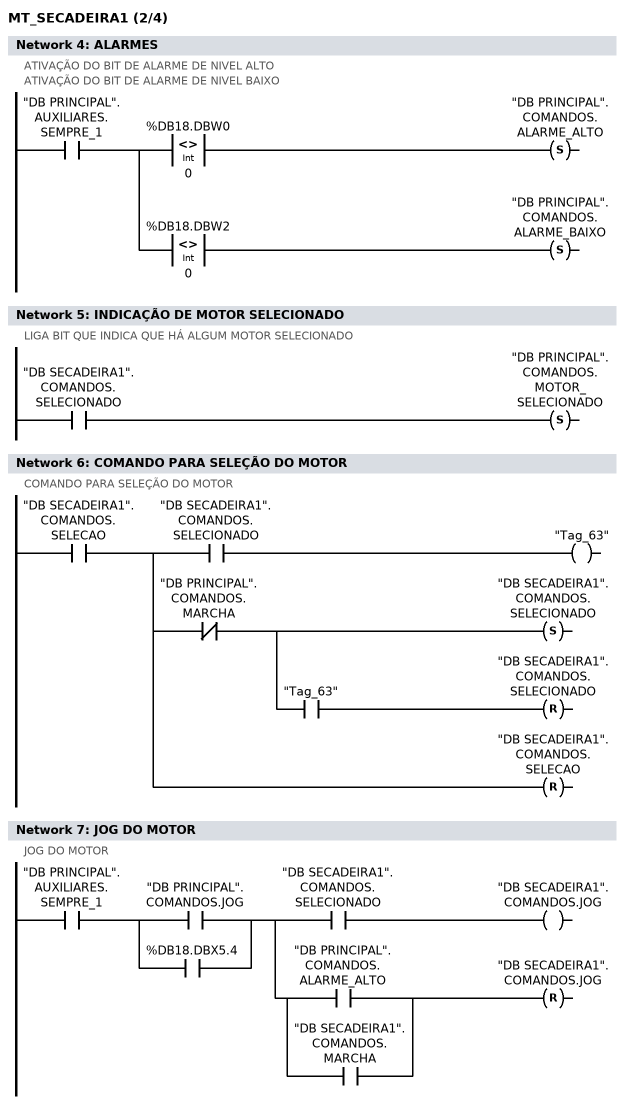
   RUNG wire#powerrail
      Contact( "DB PRINCIPAL".AUXILIARES.SEMPRE_1 )
      wire#w1
      { S7_Templates := "SrcType := Int" } NE_Contact(in1 := %DB18.DBW0, in2 := 0)
      S_Coil( "DB PRINCIPAL".COMANDOS.ALARME_ALTO )
   END_RUNG
   RUNG wire#w1
      { S7_Templates := "SrcType := Int" } NE_Contact(in1 := %DB18.DBW2, in2 := 0)
      S_Coil( "DB PRINCIPAL".COMANDOS.ALARME_BAIXO )
   END_RUNG
   // the same network as SCL:
   IF "DB PRINCIPAL".AUXILIARES.SEMPRE_1 AND (%DB18.DBW0 <> 0) THEN
       "DB PRINCIPAL".COMANDOS.ALARME_ALTO := TRUE;
   END_IF;
   IF "DB PRINCIPAL".AUXILIARES.SEMPRE_1 AND (%DB18.DBW2 <> 0) THEN
       "DB PRINCIPAL".COMANDOS.ALARME_BAIXO := TRUE;
   END_IF;
END_REGION

REGION Network 5: INDICAÇÃO DE MOTOR SELECIONADO
   // LIGA BIT QUE INDICA QUE HÁ ALGUM MOTOR SELECIONADO
   RUNG wire#powerrail
      Contact( "DB SECADEIRA1".COMANDOS.SELECIONADO )
      S_Coil( "DB PRINCIPAL".COMANDOS.MOTOR_SELECIONADO )
   END_RUNG
   // the same network as SCL:
   IF "DB SECADEIRA1".COMANDOS.SELECIONADO THEN "DB PRINCIPAL".COMANDOS.MOTOR_SELECIONADO := TRUE; END_IF;
END_REGION

REGION Network 6: COMANDO PARA SELEÇÃO DO MOTOR
   // COMANDO PARA SELEÇÃO DO MOTOR
   RUNG wire#powerrail
      Contact( "DB SECADEIRA1".COMANDOS.SELECAO )
      wire#w1
      Contact( "DB SECADEIRA1".COMANDOS.SELECIONADO )
      Coil( "Tag_63" )
   END_RUNG
   RUNG wire#w1
      I_Contact( "DB PRINCIPAL".COMANDOS.MARCHA )
      wire#w2
      S_Coil( "DB SECADEIRA1".COMANDOS.SELECIONADO )
   END_RUNG
   RUNG wire#w2
      Contact( "Tag_63" )
      R_Coil( "DB SECADEIRA1".COMANDOS.SELECIONADO )
   END_RUNG
   RUNG wire#w1
      R_Coil( "DB SECADEIRA1".COMANDOS.SELECAO )
   END_RUNG
   // the same network as SCL:
   "Tag_63" := "DB SECADEIRA1".COMANDOS.SELECAO AND "DB SECADEIRA1".COMANDOS.SELECIONADO;
   #_w1 := "DB SECADEIRA1".COMANDOS.SELECAO AND NOT "DB PRINCIPAL".COMANDOS.MARCHA;
   IF #_w1 THEN "DB SECADEIRA1".COMANDOS.SELECIONADO := TRUE; END_IF;
   IF #_w1 AND "Tag_63" THEN "DB SECADEIRA1".COMANDOS.SELECIONADO := FALSE; END_IF;
   IF "DB SECADEIRA1".COMANDOS.SELECAO THEN "DB SECADEIRA1".COMANDOS.SELECAO := FALSE; END_IF;
END_REGION

REGION Network 7: JOG DO MOTOR
   // JOG DO MOTOR
   RUNG wire#powerrail
      Contact( "DB PRINCIPAL".AUXILIARES.SEMPRE_1 )
      wire#w1
      Contact( "DB PRINCIPAL".COMANDOS.JOG )
      wire#w2
      Contact( "DB SECADEIRA1".COMANDOS.SELECIONADO )
      Coil( "DB SECADEIRA1".COMANDOS.JOG )
   END_RUNG
   RUNG wire#w1
      Contact( %DB18.DBX5.4 )
   END_RUNG wire#w2
   RUNG wire#w2
      Contact( "DB PRINCIPAL".COMANDOS.ALARME_ALTO )
      wire#w3
      R_Coil( "DB SECADEIRA1".COMANDOS.JOG )
   END_RUNG
   RUNG wire#w2
      Contact( "DB SECADEIRA1".COMANDOS.MARCHA )
   END_RUNG wire#w3
   // the same network as SCL:
   #_w1 := "DB PRINCIPAL".AUXILIARES.SEMPRE_1 AND ("DB PRINCIPAL".COMANDOS.JOG OR %DB18.DBX5.4);
   "DB SECADEIRA1".COMANDOS.JOG := #_w1 AND "DB SECADEIRA1".COMANDOS.SELECIONADO;
   IF #_w1 AND ("DB PRINCIPAL".COMANDOS.ALARME_ALTO OR "DB SECADEIRA1".COMANDOS.MARCHA) THEN
       "DB SECADEIRA1".COMANDOS.JOG := FALSE;
   END_IF;
END_REGION

REGION Network 8: COMANDO PARA LIBERAÇÃO DO MOTOR
   // COMANDO PARA LIBERAÇÃO DO MOTOR
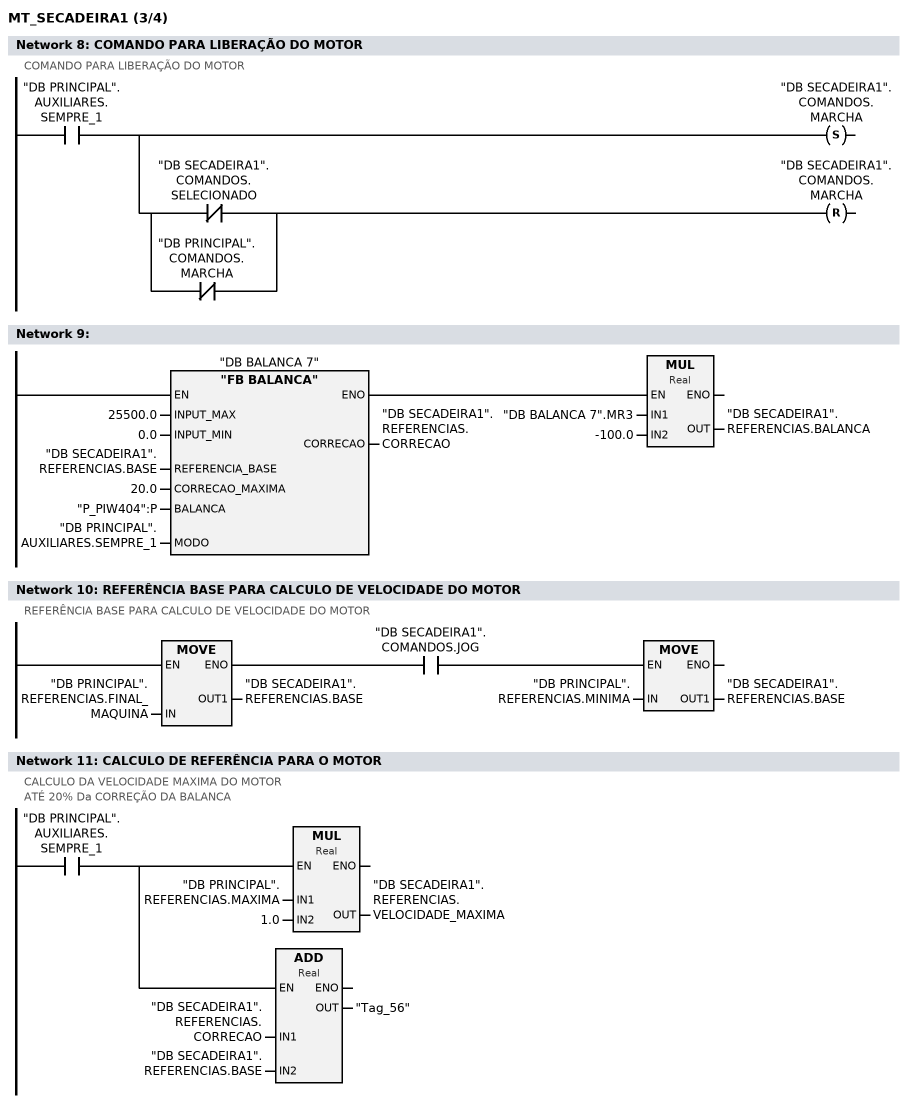
   RUNG wire#powerrail
      Contact( "DB PRINCIPAL".AUXILIARES.SEMPRE_1 )
      wire#w1
      S_Coil( "DB SECADEIRA1".COMANDOS.MARCHA )
   END_RUNG
   RUNG wire#w1
      I_Contact( "DB SECADEIRA1".COMANDOS.SELECIONADO )
      wire#w2
      R_Coil( "DB SECADEIRA1".COMANDOS.MARCHA )
   END_RUNG
   RUNG wire#w1
      I_Contact( "DB PRINCIPAL".COMANDOS.MARCHA )
   END_RUNG wire#w2
   // the same network as SCL:
   IF "DB PRINCIPAL".AUXILIARES.SEMPRE_1 THEN "DB SECADEIRA1".COMANDOS.MARCHA := TRUE; END_IF;
   IF "DB PRINCIPAL".AUXILIARES.SEMPRE_1 AND (NOT "DB SECADEIRA1".COMANDOS.SELECIONADO OR NOT "DB PRINCIPAL".COMANDOS.MARCHA) THEN
       "DB SECADEIRA1".COMANDOS.MARCHA := FALSE;
   END_IF;
END_REGION

REGION Network 9
   RUNG wire#powerrail
      "DB BALANCA 7"(INPUT_MAX := 25500.0, INPUT_MIN := 0.0, REFERENCIA_BASE := "DB SECADEIRA1".REFERENCIAS.BASE, CORRECAO_MAXIMA := 20.0, BALANCA := "P_PIW404":P, MODO := "DB PRINCIPAL".AUXILIARES.SEMPRE_1, CORRECAO => "DB SECADEIRA1".REFERENCIAS.CORRECAO)
      { S7_Templates := "SrcType := Real"; S7_GenerateENO := "TRUE" } Mul(in1 := "DB BALANCA 7".MR3, in2 := -100.0, out => "DB SECADEIRA1".REFERENCIAS.BALANCA)
   END_RUNG
   // the same network as SCL:
   "DB BALANCA 7"(INPUT_MAX := 25500.0,   // "FB BALANCA"
                  INPUT_MIN := 0.0,
                  REFERENCIA_BASE := "DB SECADEIRA1".REFERENCIAS.BASE,
                  CORRECAO_MAXIMA := 20.0,
                  BALANCA := "P_PIW404":P,
                  MODO := "DB PRINCIPAL".AUXILIARES.SEMPRE_1,
                  CORRECAO => "DB SECADEIRA1".REFERENCIAS.CORRECAO,
                  ENO => #_w1);
   IF #_w1 THEN "DB SECADEIRA1".REFERENCIAS.BALANCA := "DB BALANCA 7".MR3 * (-100.0); END_IF;
END_REGION

REGION Network 10: REFERÊNCIA BASE PARA CALCULO DE VELOCIDADE DO MOTOR
   // REFERÊNCIA BASE PARA CALCULO DE VELOCIDADE DO MOTOR
   RUNG wire#powerrail
      { S7_GenerateENO := "TRUE" } Move(in := "DB PRINCIPAL".REFERENCIAS.FINAL_MAQUINA, out1 => "DB SECADEIRA1".REFERENCIAS.BASE)
      Contact( "DB SECADEIRA1".COMANDOS.JOG )
      { S7_GenerateENO := "TRUE" } Move(in := "DB PRINCIPAL".REFERENCIAS.MINIMA, out1 => "DB SECADEIRA1".REFERENCIAS.BASE)
   END_RUNG
   // the same network as SCL:
   // ENO of a box is taken as its EN; it also drops when the box reports an error
   "DB SECADEIRA1".REFERENCIAS.BASE := "DB PRINCIPAL".REFERENCIAS.FINAL_MAQUINA;
   IF "DB SECADEIRA1".COMANDOS.JOG THEN
       "DB SECADEIRA1".REFERENCIAS.BASE := "DB PRINCIPAL".REFERENCIAS.MINIMA;
   END_IF;
END_REGION

REGION Network 11: CALCULO DE REFERÊNCIA PARA O MOTOR
   // CALCULO DA VELOCIDADE MAXIMA DO MOTOR
   // ATÉ 20% Da CORREÇÃO DA BALANCA
   RUNG wire#powerrail
      Contact( "DB PRINCIPAL".AUXILIARES.SEMPRE_1 )
      wire#w1
      { S7_Templates := "SrcType := Real"; S7_GenerateENO := "TRUE" } Mul(in1 := "DB PRINCIPAL".REFERENCIAS.MAXIMA, in2 := 1.0, out => "DB SECADEIRA1".REFERENCIAS.VELOCIDADE_MAXIMA)
   END_RUNG
   RUNG wire#w1
      { S7_Templates := "SrcType := Real"; S7_GenerateENO := "TRUE" } Add(in1 := "DB SECADEIRA1".REFERENCIAS.CORRECAO, in2 := "DB SECADEIRA1".REFERENCIAS.BASE, out => "Tag_56")
   END_RUNG
   // the same network as SCL:
   IF "DB PRINCIPAL".AUXILIARES.SEMPRE_1 THEN
       "DB SECADEIRA1".REFERENCIAS.VELOCIDADE_MAXIMA := "DB PRINCIPAL".REFERENCIAS.MAXIMA * 1.0;
       "Tag_56" := "DB SECADEIRA1".REFERENCIAS.CORRECAO + "DB SECADEIRA1".REFERENCIAS.BASE;
   END_IF;
END_REGION

REGION Network 12: ACC/DEC DA REFERÊNCIA DO MOTOR
   // ACC/DEC DA REFERÊNCIA DO MOTOR
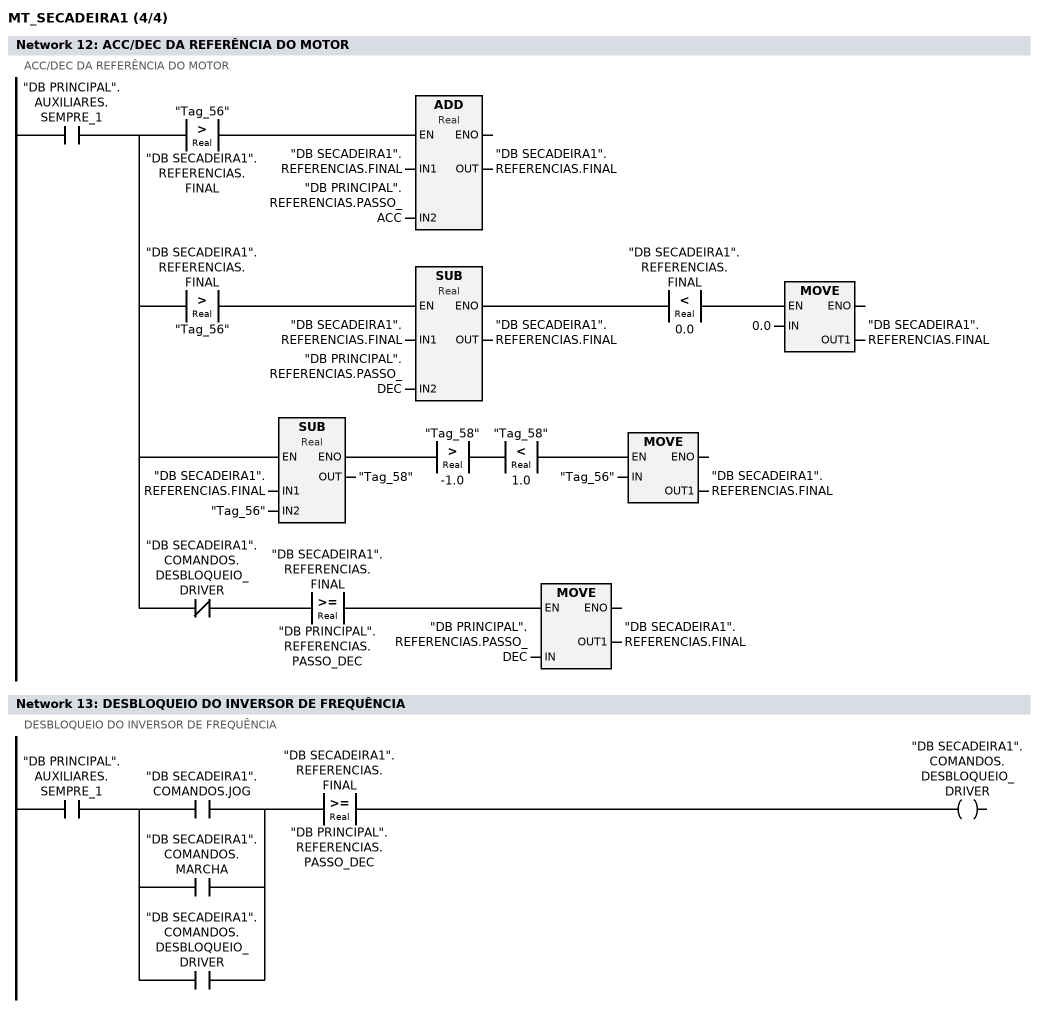
   RUNG wire#powerrail
      Contact( "DB PRINCIPAL".AUXILIARES.SEMPRE_1 )
      wire#w1
      { S7_Templates := "SrcType := Real" } GT_Contact(in1 := "Tag_56", in2 := "DB SECADEIRA1".REFERENCIAS.FINAL)
      { S7_Templates := "SrcType := Real"; S7_GenerateENO := "TRUE" } Add(in1 := "DB SECADEIRA1".REFERENCIAS.FINAL, in2 := "DB PRINCIPAL".REFERENCIAS.PASSO_ACC, out => "DB SECADEIRA1".REFERENCIAS.FINAL)
   END_RUNG
   RUNG wire#w1
      { S7_Templates := "SrcType := Real" } GT_Contact(in1 := "DB SECADEIRA1".REFERENCIAS.FINAL, in2 := "Tag_56")
      { S7_Templates := "SrcType := Real"; S7_GenerateENO := "TRUE" } Sub(in1 := "DB SECADEIRA1".REFERENCIAS.FINAL, in2 := "DB PRINCIPAL".REFERENCIAS.PASSO_DEC, out => "DB SECADEIRA1".REFERENCIAS.FINAL)
      { S7_Templates := "SrcType := Real" } LT_Contact(in1 := "DB SECADEIRA1".REFERENCIAS.FINAL, in2 := 0.0)
      { S7_GenerateENO := "TRUE" } Move(in := 0.0, out1 => "DB SECADEIRA1".REFERENCIAS.FINAL)
   END_RUNG
   RUNG wire#w1
      { S7_Templates := "SrcType := Real"; S7_GenerateENO := "TRUE" } Sub(in1 := "DB SECADEIRA1".REFERENCIAS.FINAL, in2 := "Tag_56", out => "Tag_58")
      { S7_Templates := "SrcType := Real" } GT_Contact(in1 := "Tag_58", in2 := -1.0)
      { S7_Templates := "SrcType := Real" } LT_Contact(in1 := "Tag_58", in2 := 1.0)
      { S7_GenerateENO := "TRUE" } Move(in := "Tag_56", out1 => "DB SECADEIRA1".REFERENCIAS.FINAL)
   END_RUNG
   RUNG wire#w1
      I_Contact( "DB SECADEIRA1".COMANDOS.DESBLOQUEIO_DRIVER )
      { S7_Templates := "SrcType := Real" } GE_Contact(in1 := "DB SECADEIRA1".REFERENCIAS.FINAL, in2 := "DB PRINCIPAL".REFERENCIAS.PASSO_DEC)
      { S7_GenerateENO := "TRUE" } Move(in := "DB PRINCIPAL".REFERENCIAS.PASSO_DEC, out1 => "DB SECADEIRA1".REFERENCIAS.FINAL)
   END_RUNG
   // the same network as SCL:
   // ENO of a box is taken as its EN; it also drops when the box reports an error
   IF "DB PRINCIPAL".AUXILIARES.SEMPRE_1 AND ("Tag_56" > "DB SECADEIRA1".REFERENCIAS.FINAL) THEN
       "DB SECADEIRA1".REFERENCIAS.FINAL := "DB SECADEIRA1".REFERENCIAS.FINAL + "DB PRINCIPAL".REFERENCIAS.PASSO_ACC;
   END_IF;
   #_w1 := "DB PRINCIPAL".AUXILIARES.SEMPRE_1 AND ("DB SECADEIRA1".REFERENCIAS.FINAL > "Tag_56");
   IF #_w1 THEN
       "DB SECADEIRA1".REFERENCIAS.FINAL := "DB SECADEIRA1".REFERENCIAS.FINAL - "DB PRINCIPAL".REFERENCIAS.PASSO_DEC;
   END_IF;
   IF #_w1 AND ("DB SECADEIRA1".REFERENCIAS.FINAL < 0.0) THEN
       "DB SECADEIRA1".REFERENCIAS.FINAL := 0.0;
   END_IF;
   IF "DB PRINCIPAL".AUXILIARES.SEMPRE_1 THEN
       "Tag_58" := "DB SECADEIRA1".REFERENCIAS.FINAL - "Tag_56";
   END_IF;
   IF "DB PRINCIPAL".AUXILIARES.SEMPRE_1 AND ("Tag_58" > (-1.0)) AND ("Tag_58" < 1.0) THEN
       "DB SECADEIRA1".REFERENCIAS.FINAL := "Tag_56";
   END_IF;
   IF "DB PRINCIPAL".AUXILIARES.SEMPRE_1 AND NOT "DB SECADEIRA1".COMANDOS.DESBLOQUEIO_DRIVER AND ("DB SECADEIRA1".REFERENCIAS.FINAL >= "DB PRINCIPAL".REFERENCIAS.PASSO_DEC) THEN
       "DB SECADEIRA1".REFERENCIAS.FINAL := "DB PRINCIPAL".REFERENCIAS.PASSO_DEC;
   END_IF;
END_REGION

REGION Network 13: DESBLOQUEIO DO INVERSOR DE FREQUÊNCIA
   // DESBLOQUEIO DO INVERSOR DE FREQUÊNCIA
   RUNG wire#powerrail
      Contact( "DB PRINCIPAL".AUXILIARES.SEMPRE_1 )
      wire#w1
      Contact( "DB SECADEIRA1".COMANDOS.JOG )
      wire#w2
      { S7_Templates := "SrcType := Real" } GE_Contact(in1 := "DB SECADEIRA1".REFERENCIAS.FINAL, in2 := "DB PRINCIPAL".REFERENCIAS.PASSO_DEC)
      Coil( "DB SECADEIRA1".COMANDOS.DESBLOQUEIO_DRIVER )
   END_RUNG
   RUNG wire#w1
      Contact( "DB SECADEIRA1".COMANDOS.MARCHA )
   END_RUNG wire#w2
   RUNG wire#w1
      Contact( "DB SECADEIRA1".COMANDOS.DESBLOQUEIO_DRIVER )
   END_RUNG wire#w2
   // the same network as SCL:
   "DB SECADEIRA1".COMANDOS.DESBLOQUEIO_DRIVER := "DB PRINCIPAL".AUXILIARES.SEMPRE_1 AND ("DB SECADEIRA1".COMANDOS.JOG OR "DB SECADEIRA1".COMANDOS.MARCHA OR "DB SECADEIRA1".COMANDOS.DESBLOQUEIO_DRIVER) AND ("DB SECADEIRA1".REFERENCIAS.FINAL >= "DB PRINCIPAL".REFERENCIAS.PASSO_DEC);
END_REGION

REGION Network 14 (STL): STATUS / CONTROLE - INVERSOR DE FREQUÊNCIA
   // DANFOSS FC300 PROFIBUS - TEX24626INV001
   // STATUS DO INVERSOR DE FREQUÊNCIA
         L     "Tag_27":P;
         T     "Tag_1";
         AN    "Tag_59";
         =     "DB SECADEIRA1".COMANDOS.STATUS_DRIVER;

   // CONTROLE DO INVERSOR DE FREQUÊNCIA
         L     1150;
         T     "Tag_1";
         A     "DB SECADEIRA1".COMANDOS.DESBLOQUEIO_DRIVER;
         =     "Tag_60";
         A     "T2";
         AN    "DB SECADEIRA1".COMANDOS.STATUS_DRIVER;
         =     "Tag_61";
         L     "Tag_1";
         T     "Tag_28":P;

   // REFERÊNCIA PARA O INVERSOR DE FREQUÊNCIA
         L     "DB SECADEIRA1".REFERENCIAS.FINAL;
         L     16384.0;
         *R;

         L     "DB SECADEIRA1".REFERENCIAS.VELOCIDADE_MAXIMA;
         /R;
         RND;
         T     "Tag_62";
         L     "Tag_62";
         T     "Tag_29":P;
END_REGION

REGION Network 15 (STL): INVERSOR RESERVA
         A     "DB PRINCIPAL".AUXILIARES.SEMPRE_1;
         =     %L24.0;
         A     %L24.0;
         A(;
         L     "DB PRINCIPAL".AUXILIARES1.INVERSOR_RESERVA1;
         L     9;
         ==I;
         );
         =     %L24.1;
         A     %L24.1;
         JNB   M00c;
         L     "DB SECADEIRA1".REFERENCIAS.FINAL;
         L     3.456;
         *R;
         T     #AUX_R;
         RND;
         T     "P_QW100":P;
   M00c: NOP   0;
         A     %L24.1;
         A     "I130";
         S     "DB PRINCIPAL".ALARME.INV_RESERVA1;
         A     %L24.1;
         A     "DB SECADEIRA1".COMANDOS.DESBLOQUEIO_DRIVER;
         S     "Q134";
         A     %L24.1;
         AN    "DB SECADEIRA1".COMANDOS.DESBLOQUEIO_DRIVER;
         R     "Q134";
         A     %L24.0;
         A(;
         L     "DB PRINCIPAL".AUXILIARES1.INVERSOR_RESERVA2;
         L     9;
         ==I;
         );
         =     %L24.1;
         A     %L24.1;
         JNB   M00d;
         L     "DB SECADEIRA1".REFERENCIAS.FINAL;
         L     3.456;
         *R;
         T     #AUX_R;
         RND;
         T     "P_QW102":P;
   M00d: NOP   0;
         A     %L24.1;
         A     "I132";
         S     "DB PRINCIPAL".ALARME.INV_RESERVA2;
         A     %L24.1;
         A     "DB SECADEIRA1".COMANDOS.DESBLOQUEIO_DRIVER;
         S     "Q135";
         A     %L24.1;
         AN    "DB SECADEIRA1".COMANDOS.DESBLOQUEIO_DRIVER;
         R     "Q135";
END_REGION
END_FUNCTION

FUNCTION "MT_FOULARD" : Void   // FC19, LAD
TITLE = MÓDULO DE CONTROLE DO FOULARD
{ S7_Optimized_Access := 'FALSE' }
AUTHOR : THALLES
FAMILY : TRAÇÃO
NAME : LINHA1
VERSION : 0.1
// DATA BLOCK DE CONTROLE // DB19
// Automation Pack Automação Indl. e Com. Ltda.
// Cliente: Texima S/A Ind. de Máquinas
// Cliente Final: Cia. Fiação e Tecidos Santo Antonio.
// Máquina: LINHA 1 DENIN - O.S.: 24.626
   VAR_TEMP
      AUX_R : Real;
   END_VAR
   VAR_TEMP   // added for the SCL form of the ladder/FBD networks
      _w1 : Bool;
   END_VAR
BEGIN

REGION Network 1: ALARMES
   // RESET DOS ALARMES
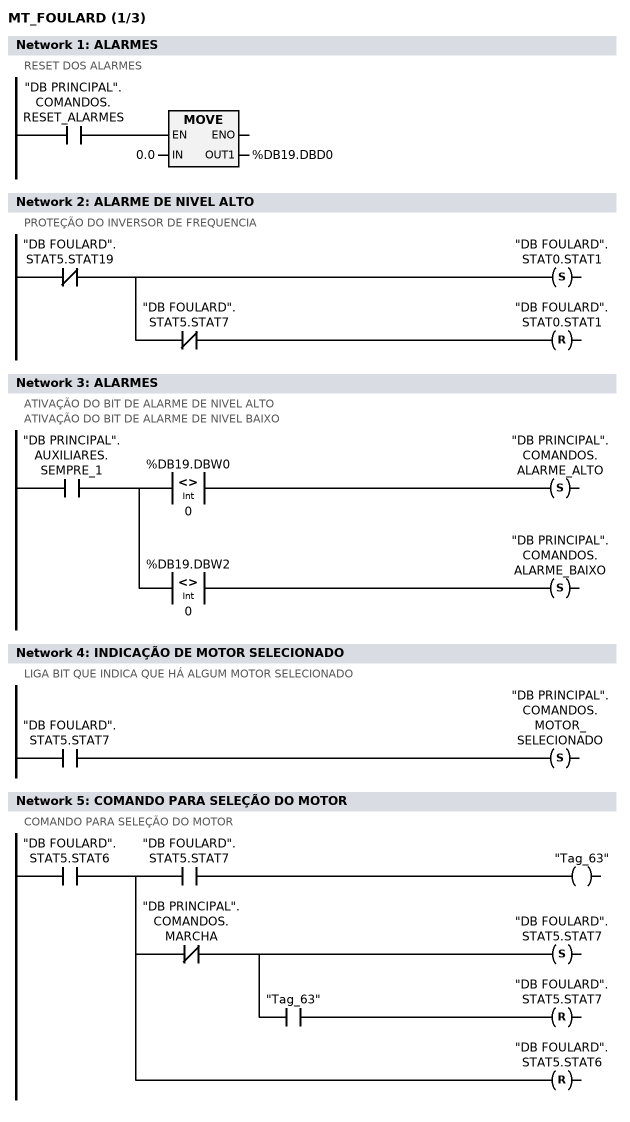
   RUNG wire#powerrail
      Contact( "DB PRINCIPAL".COMANDOS.RESET_ALARMES )
      { S7_GenerateENO := "TRUE" } Move(in := 0.0, out1 => %DB19.DBD0)
   END_RUNG
   // the same network as SCL:
   IF "DB PRINCIPAL".COMANDOS.RESET_ALARMES THEN %DB19.DBD0 := 0.0; END_IF;
END_REGION

REGION Network 2: ALARME DE NIVEL ALTO
   // PROTEÇÃO DO INVERSOR DE FREQUENCIA
   RUNG wire#powerrail
      I_Contact( "DB FOULARD".STAT5.STAT19 )
      wire#w1
      S_Coil( "DB FOULARD".STAT0.STAT1 )
   END_RUNG
   RUNG wire#w1
      I_Contact( "DB FOULARD".STAT5.STAT7 )
      R_Coil( "DB FOULARD".STAT0.STAT1 )
   END_RUNG
   // the same network as SCL:
   #_w1 := NOT "DB FOULARD".STAT5.STAT19;
   IF #_w1 THEN "DB FOULARD".STAT0.STAT1 := TRUE; END_IF;
   IF #_w1 AND NOT "DB FOULARD".STAT5.STAT7 THEN "DB FOULARD".STAT0.STAT1 := FALSE; END_IF;
END_REGION

REGION Network 3: ALARMES
   // ATIVAÇÃO DO BIT DE ALARME DE NIVEL ALTO
   // ATIVAÇÃO DO BIT DE ALARME DE NIVEL BAIXO
   RUNG wire#powerrail
      Contact( "DB PRINCIPAL".AUXILIARES.SEMPRE_1 )
      wire#w1
      { S7_Templates := "SrcType := Int" } NE_Contact(in1 := %DB19.DBW0, in2 := 0)
      S_Coil( "DB PRINCIPAL".COMANDOS.ALARME_ALTO )
   END_RUNG
   RUNG wire#w1
      { S7_Templates := "SrcType := Int" } NE_Contact(in1 := %DB19.DBW2, in2 := 0)
      S_Coil( "DB PRINCIPAL".COMANDOS.ALARME_BAIXO )
   END_RUNG
   // the same network as SCL:
   IF "DB PRINCIPAL".AUXILIARES.SEMPRE_1 AND (%DB19.DBW0 <> 0) THEN
       "DB PRINCIPAL".COMANDOS.ALARME_ALTO := TRUE;
   END_IF;
   IF "DB PRINCIPAL".AUXILIARES.SEMPRE_1 AND (%DB19.DBW2 <> 0) THEN
       "DB PRINCIPAL".COMANDOS.ALARME_BAIXO := TRUE;
   END_IF;
END_REGION

REGION Network 4: INDICAÇÃO DE MOTOR SELECIONADO
   // LIGA BIT QUE INDICA QUE HÁ ALGUM MOTOR SELECIONADO
   RUNG wire#powerrail
      Contact( "DB FOULARD".STAT5.STAT7 )
      S_Coil( "DB PRINCIPAL".COMANDOS.MOTOR_SELECIONADO )
   END_RUNG
   // the same network as SCL:
   IF "DB FOULARD".STAT5.STAT7 THEN "DB PRINCIPAL".COMANDOS.MOTOR_SELECIONADO := TRUE; END_IF;
END_REGION

REGION Network 5: COMANDO PARA SELEÇÃO DO MOTOR
   // COMANDO PARA SELEÇÃO DO MOTOR
   RUNG wire#powerrail
      Contact( "DB FOULARD".STAT5.STAT6 )
      wire#w1
      Contact( "DB FOULARD".STAT5.STAT7 )
      Coil( "Tag_63" )
   END_RUNG
   RUNG wire#w1
      I_Contact( "DB PRINCIPAL".COMANDOS.MARCHA )
      wire#w2
      S_Coil( "DB FOULARD".STAT5.STAT7 )
   END_RUNG
   RUNG wire#w2
      Contact( "Tag_63" )
      R_Coil( "DB FOULARD".STAT5.STAT7 )
   END_RUNG
   RUNG wire#w1
      R_Coil( "DB FOULARD".STAT5.STAT6 )
   END_RUNG
   // the same network as SCL:
   "Tag_63" := "DB FOULARD".STAT5.STAT6 AND "DB FOULARD".STAT5.STAT7;
   #_w1 := "DB FOULARD".STAT5.STAT6 AND NOT "DB PRINCIPAL".COMANDOS.MARCHA;
   IF #_w1 THEN "DB FOULARD".STAT5.STAT7 := TRUE; END_IF;
   IF #_w1 AND "Tag_63" THEN "DB FOULARD".STAT5.STAT7 := FALSE; END_IF;
   IF "DB FOULARD".STAT5.STAT6 THEN "DB FOULARD".STAT5.STAT6 := FALSE; END_IF;
END_REGION

REGION Network 6: JOG DO MOTOR
   // JOG DO MOTOR
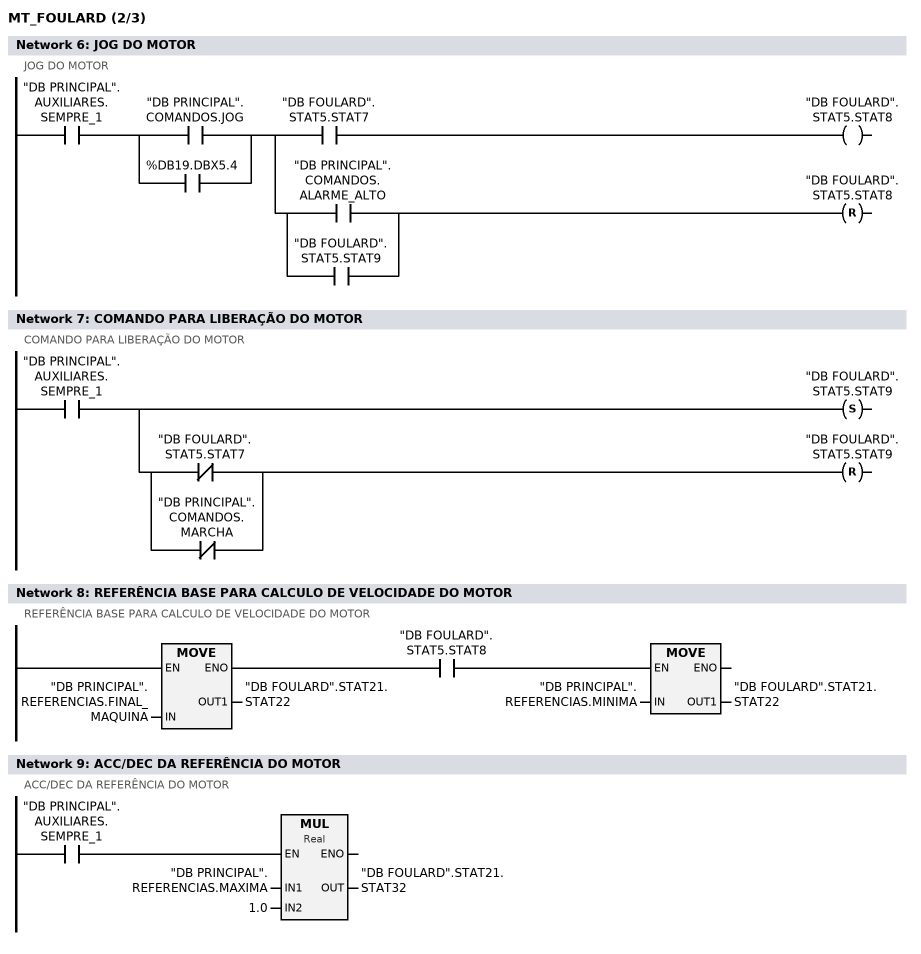
   RUNG wire#powerrail
      Contact( "DB PRINCIPAL".AUXILIARES.SEMPRE_1 )
      wire#w1
      Contact( "DB PRINCIPAL".COMANDOS.JOG )
      wire#w2
      Contact( "DB FOULARD".STAT5.STAT7 )
      Coil( "DB FOULARD".STAT5.STAT8 )
   END_RUNG
   RUNG wire#w1
      Contact( %DB19.DBX5.4 )
   END_RUNG wire#w2
   RUNG wire#w2
      Contact( "DB PRINCIPAL".COMANDOS.ALARME_ALTO )
      wire#w3
      R_Coil( "DB FOULARD".STAT5.STAT8 )
   END_RUNG
   RUNG wire#w2
      Contact( "DB FOULARD".STAT5.STAT9 )
   END_RUNG wire#w3
   // the same network as SCL:
   #_w1 := "DB PRINCIPAL".AUXILIARES.SEMPRE_1 AND ("DB PRINCIPAL".COMANDOS.JOG OR %DB19.DBX5.4);
   "DB FOULARD".STAT5.STAT8 := #_w1 AND "DB FOULARD".STAT5.STAT7;
   IF #_w1 AND ("DB PRINCIPAL".COMANDOS.ALARME_ALTO OR "DB FOULARD".STAT5.STAT9) THEN
       "DB FOULARD".STAT5.STAT8 := FALSE;
   END_IF;
END_REGION

REGION Network 7: COMANDO PARA LIBERAÇÃO DO MOTOR
   // COMANDO PARA LIBERAÇÃO DO MOTOR
   RUNG wire#powerrail
      Contact( "DB PRINCIPAL".AUXILIARES.SEMPRE_1 )
      wire#w1
      S_Coil( "DB FOULARD".STAT5.STAT9 )
   END_RUNG
   RUNG wire#w1
      I_Contact( "DB FOULARD".STAT5.STAT7 )
      wire#w2
      R_Coil( "DB FOULARD".STAT5.STAT9 )
   END_RUNG
   RUNG wire#w1
      I_Contact( "DB PRINCIPAL".COMANDOS.MARCHA )
   END_RUNG wire#w2
   // the same network as SCL:
   IF "DB PRINCIPAL".AUXILIARES.SEMPRE_1 THEN "DB FOULARD".STAT5.STAT9 := TRUE; END_IF;
   IF "DB PRINCIPAL".AUXILIARES.SEMPRE_1 AND (NOT "DB FOULARD".STAT5.STAT7 OR NOT "DB PRINCIPAL".COMANDOS.MARCHA) THEN
       "DB FOULARD".STAT5.STAT9 := FALSE;
   END_IF;
END_REGION

REGION Network 8: REFERÊNCIA BASE PARA CALCULO DE VELOCIDADE DO MOTOR
   // REFERÊNCIA BASE PARA CALCULO DE VELOCIDADE DO MOTOR
   RUNG wire#powerrail
      { S7_GenerateENO := "TRUE" } Move(in := "DB PRINCIPAL".REFERENCIAS.FINAL_MAQUINA, out1 => "DB FOULARD".STAT21.STAT22)
      Contact( "DB FOULARD".STAT5.STAT8 )
      { S7_GenerateENO := "TRUE" } Move(in := "DB PRINCIPAL".REFERENCIAS.MINIMA, out1 => "DB FOULARD".STAT21.STAT22)
   END_RUNG
   // the same network as SCL:
   // ENO of a box is taken as its EN; it also drops when the box reports an error
   "DB FOULARD".STAT21.STAT22 := "DB PRINCIPAL".REFERENCIAS.FINAL_MAQUINA;
   IF "DB FOULARD".STAT5.STAT8 THEN "DB FOULARD".STAT21.STAT22 := "DB PRINCIPAL".REFERENCIAS.MINIMA; END_IF;
END_REGION

REGION Network 9: ACC/DEC DA REFERÊNCIA DO MOTOR
   // ACC/DEC DA REFERÊNCIA DO MOTOR
   RUNG wire#powerrail
      Contact( "DB PRINCIPAL".AUXILIARES.SEMPRE_1 )
      { S7_Templates := "SrcType := Real"; S7_GenerateENO := "TRUE" } Mul(in1 := "DB PRINCIPAL".REFERENCIAS.MAXIMA, in2 := 1.0, out => "DB FOULARD".STAT21.STAT32)
   END_RUNG
   // the same network as SCL:
   IF "DB PRINCIPAL".AUXILIARES.SEMPRE_1 THEN
       "DB FOULARD".STAT21.STAT32 := "DB PRINCIPAL".REFERENCIAS.MAXIMA * 1.0;
   END_IF;
END_REGION

REGION Network 10: DESBLOQUEIO DO INVERSOR DE FREQUÊNCIA
   // DESBLOQUEIO DO INVERSOR DE FREQUÊNCIA
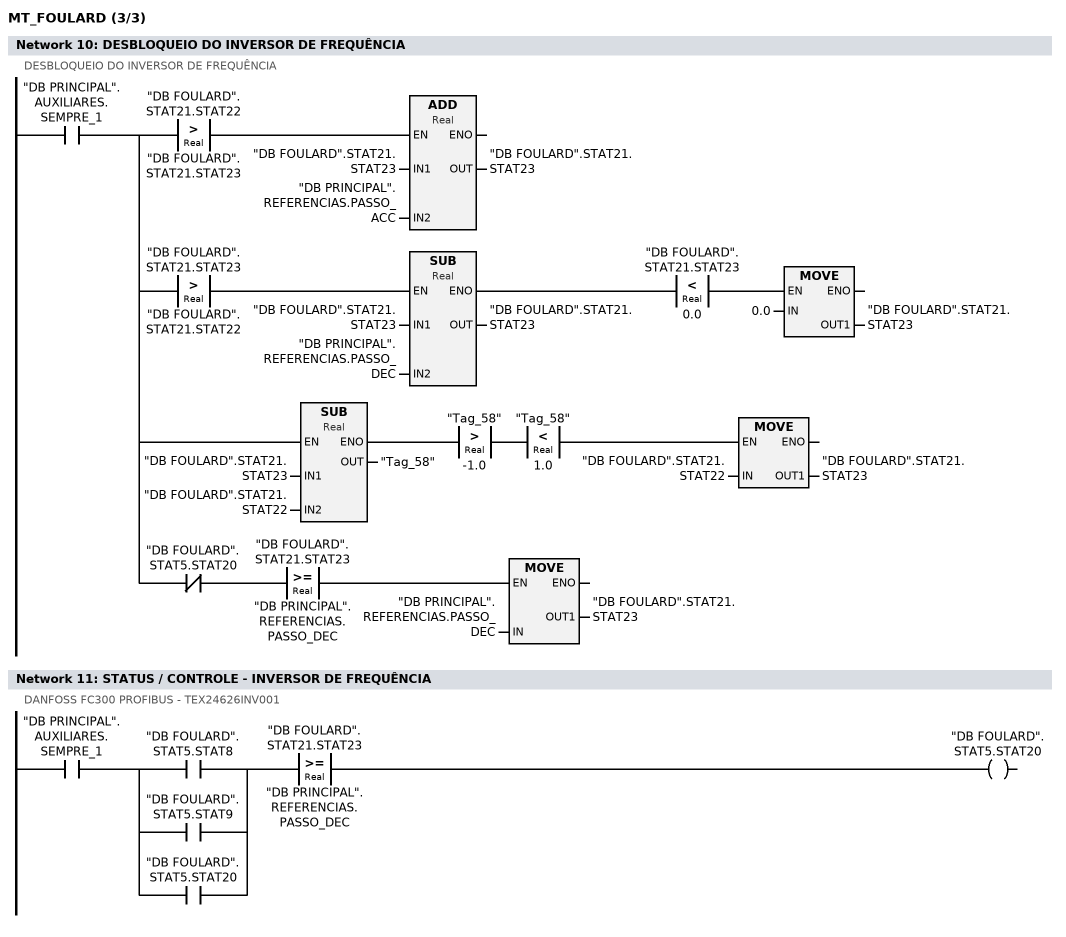
   RUNG wire#powerrail
      Contact( "DB PRINCIPAL".AUXILIARES.SEMPRE_1 )
      wire#w1
      { S7_Templates := "SrcType := Real" } GT_Contact(in1 := "DB FOULARD".STAT21.STAT22, in2 := "DB FOULARD".STAT21.STAT23)
      { S7_Templates := "SrcType := Real"; S7_GenerateENO := "TRUE" } Add(in1 := "DB FOULARD".STAT21.STAT23, in2 := "DB PRINCIPAL".REFERENCIAS.PASSO_ACC, out => "DB FOULARD".STAT21.STAT23)
   END_RUNG
   RUNG wire#w1
      { S7_Templates := "SrcType := Real" } GT_Contact(in1 := "DB FOULARD".STAT21.STAT23, in2 := "DB FOULARD".STAT21.STAT22)
      { S7_Templates := "SrcType := Real"; S7_GenerateENO := "TRUE" } Sub(in1 := "DB FOULARD".STAT21.STAT23, in2 := "DB PRINCIPAL".REFERENCIAS.PASSO_DEC, out => "DB FOULARD".STAT21.STAT23)
      { S7_Templates := "SrcType := Real" } LT_Contact(in1 := "DB FOULARD".STAT21.STAT23, in2 := 0.0)
      { S7_GenerateENO := "TRUE" } Move(in := 0.0, out1 => "DB FOULARD".STAT21.STAT23)
   END_RUNG
   RUNG wire#w1
      { S7_Templates := "SrcType := Real"; S7_GenerateENO := "TRUE" } Sub(in1 := "DB FOULARD".STAT21.STAT23, in2 := "DB FOULARD".STAT21.STAT22, out => "Tag_58")
      { S7_Templates := "SrcType := Real" } GT_Contact(in1 := "Tag_58", in2 := -1.0)
      { S7_Templates := "SrcType := Real" } LT_Contact(in1 := "Tag_58", in2 := 1.0)
      { S7_GenerateENO := "TRUE" } Move(in := "DB FOULARD".STAT21.STAT22, out1 => "DB FOULARD".STAT21.STAT23)
   END_RUNG
   RUNG wire#w1
      I_Contact( "DB FOULARD".STAT5.STAT20 )
      { S7_Templates := "SrcType := Real" } GE_Contact(in1 := "DB FOULARD".STAT21.STAT23, in2 := "DB PRINCIPAL".REFERENCIAS.PASSO_DEC)
      { S7_GenerateENO := "TRUE" } Move(in := "DB PRINCIPAL".REFERENCIAS.PASSO_DEC, out1 => "DB FOULARD".STAT21.STAT23)
   END_RUNG
   // the same network as SCL:
   // ENO of a box is taken as its EN; it also drops when the box reports an error
   IF "DB PRINCIPAL".AUXILIARES.SEMPRE_1 AND ("DB FOULARD".STAT21.STAT22 > "DB FOULARD".STAT21.STAT23) THEN
       "DB FOULARD".STAT21.STAT23 := "DB FOULARD".STAT21.STAT23 + "DB PRINCIPAL".REFERENCIAS.PASSO_ACC;
   END_IF;
   #_w1 := "DB PRINCIPAL".AUXILIARES.SEMPRE_1 AND ("DB FOULARD".STAT21.STAT23 > "DB FOULARD".STAT21.STAT22);
   IF #_w1 THEN
       "DB FOULARD".STAT21.STAT23 := "DB FOULARD".STAT21.STAT23 - "DB PRINCIPAL".REFERENCIAS.PASSO_DEC;
   END_IF;
   IF #_w1 AND ("DB FOULARD".STAT21.STAT23 < 0.0) THEN "DB FOULARD".STAT21.STAT23 := 0.0; END_IF;
   IF "DB PRINCIPAL".AUXILIARES.SEMPRE_1 THEN
       "Tag_58" := "DB FOULARD".STAT21.STAT23 - "DB FOULARD".STAT21.STAT22;
   END_IF;
   IF "DB PRINCIPAL".AUXILIARES.SEMPRE_1 AND ("Tag_58" > (-1.0)) AND ("Tag_58" < 1.0) THEN
       "DB FOULARD".STAT21.STAT23 := "DB FOULARD".STAT21.STAT22;
   END_IF;
   IF "DB PRINCIPAL".AUXILIARES.SEMPRE_1 AND NOT "DB FOULARD".STAT5.STAT20 AND ("DB FOULARD".STAT21.STAT23 >= "DB PRINCIPAL".REFERENCIAS.PASSO_DEC) THEN
       "DB FOULARD".STAT21.STAT23 := "DB PRINCIPAL".REFERENCIAS.PASSO_DEC;
   END_IF;
END_REGION

REGION Network 11: STATUS / CONTROLE - INVERSOR DE FREQUÊNCIA
   // DANFOSS FC300 PROFIBUS - TEX24626INV001
   RUNG wire#powerrail
      Contact( "DB PRINCIPAL".AUXILIARES.SEMPRE_1 )
      wire#w1
      Contact( "DB FOULARD".STAT5.STAT8 )
      wire#w2
      { S7_Templates := "SrcType := Real" } GE_Contact(in1 := "DB FOULARD".STAT21.STAT23, in2 := "DB PRINCIPAL".REFERENCIAS.PASSO_DEC)
      Coil( "DB FOULARD".STAT5.STAT20 )
   END_RUNG
   RUNG wire#w1
      Contact( "DB FOULARD".STAT5.STAT9 )
   END_RUNG wire#w2
   RUNG wire#w1
      Contact( "DB FOULARD".STAT5.STAT20 )
   END_RUNG wire#w2
   // the same network as SCL:
   "DB FOULARD".STAT5.STAT20 := "DB PRINCIPAL".AUXILIARES.SEMPRE_1 AND ("DB FOULARD".STAT5.STAT8 OR "DB FOULARD".STAT5.STAT9 OR "DB FOULARD".STAT5.STAT20) AND ("DB FOULARD".STAT21.STAT23 >= "DB PRINCIPAL".REFERENCIAS.PASSO_DEC);
END_REGION

REGION Network 12 (STL): INVERSOR RESERVA
         L     "Tag_30":P;
         T     "Tag_1";
         AN    "Tag_59";
         =     "DB FOULARD".STAT5.STAT19;
         L     1150;
         T     "Tag_1";
         A     "DB FOULARD".STAT5.STAT20;
         =     "Tag_60";
         A     "T2";
         AN    "DB FOULARD".STAT5.STAT19;
         =     "Tag_61";
         L     "Tag_1";
         T     "Tag_31":P;
         L     "DB FOULARD".STAT21.STAT23;
         L     16384.0;
         *R;
         L     "DB FOULARD".STAT21.STAT32;
         /R;
         RND;
         T     "Tag_62";
         L     "Tag_62";
         T     "Tag_32":P;
END_REGION

REGION Network 13 (STL)
         A     "DB PRINCIPAL".AUXILIARES.SEMPRE_1;
         =     %L24.0;
         A     %L24.0;
         A(;
         L     "DB PRINCIPAL".AUXILIARES1.INVERSOR_RESERVA1;
         L     10;
         ==I;
         );
         =     %L24.1;
         A     %L24.1;
         JNB   M003;
         L     "DB FOULARD".STAT21.STAT23;
         L     3.456;
         *R;
         T     #AUX_R;
         RND;
         T     "P_QW100":P;
   M003: NOP   0;
         A     %L24.1;
         A     "I130";
         S     "DB PRINCIPAL".ALARME.INV_RESERVA1;
         A     %L24.1;
         A     "DB FOULARD".STAT5.STAT20;
         S     "Q134";
         A     %L24.1;
         AN    "DB FOULARD".STAT5.STAT20;
         R     "Q134";
         A     %L24.0;
         A(;
         L     "DB PRINCIPAL".AUXILIARES1.INVERSOR_RESERVA2;
         L     10;
         ==I;
         );
         =     %L24.1;
         A     %L24.1;
         JNB   M004;
         L     "DB FOULARD".STAT21.STAT23;
         L     3.456;
         *R;
         T     #AUX_R;
         RND;
         T     "P_QW102":P;
   M004: NOP   0;
         A     %L24.1;
         A     "I132";
         S     "DB PRINCIPAL".ALARME.INV_RESERVA2;
         A     %L24.1;
         A     "DB FOULARD".STAT5.STAT20;
         S     "Q135";
         A     %L24.1;
         AN    "DB FOULARD".STAT5.STAT20;
         R     "Q135";
END_REGION
END_FUNCTION

FUNCTION "MT_ESTICADOR" : Void   // FC20, LAD
TITLE = MÓDULO DE CONTROLE DO ESTICADOR
{ S7_Optimized_Access := 'FALSE' }
AUTHOR : THALLES
FAMILY : TRAÇÃO
NAME : LINHA1
VERSION : 0.1
// DATA BLOCK DE CONTROLE // DB20
// Automation Pack Automação Indl. e Com. Ltda.
// Cliente: Texima S/A Ind. de Máquinas
// Cliente Final: Cia. Fiação e Tecidos Santo Antonio.
// Máquina: LINHA 1 DENIN - O.S.: 24.626
   VAR_TEMP
      AUX_R : Real;
   END_VAR
   VAR_TEMP   // added for the SCL form of the ladder/FBD networks
      _w1 : Bool;
   END_VAR
BEGIN

REGION Network 1: ALARMES
   // RESET DOS ALARMES
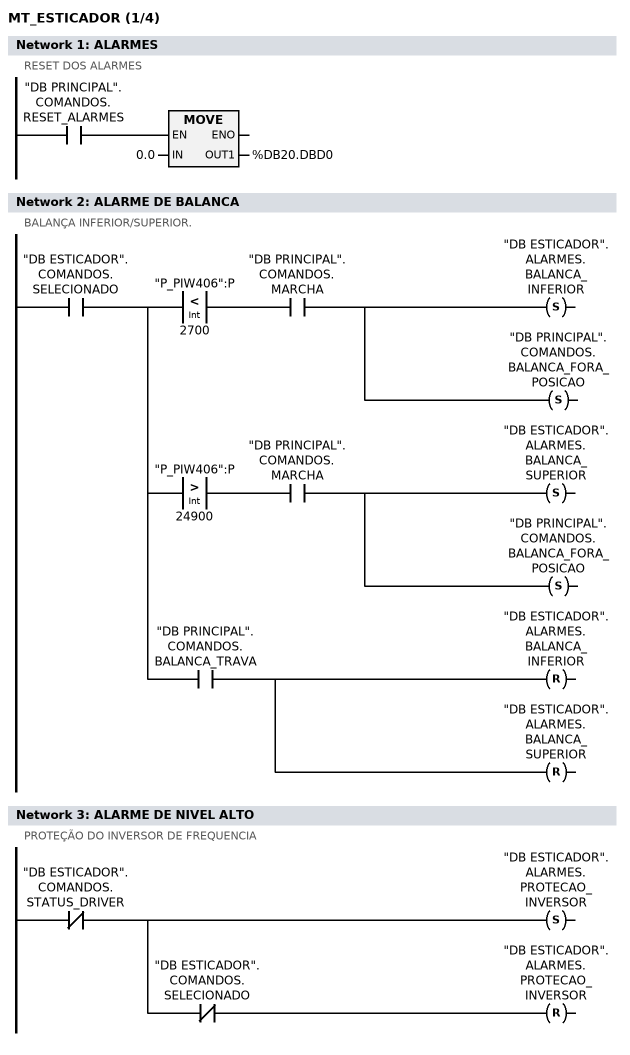
   RUNG wire#powerrail
      Contact( "DB PRINCIPAL".COMANDOS.RESET_ALARMES )
      { S7_GenerateENO := "TRUE" } Move(in := 0.0, out1 => %DB20.DBD0)
   END_RUNG
   // the same network as SCL:
   IF "DB PRINCIPAL".COMANDOS.RESET_ALARMES THEN %DB20.DBD0 := 0.0; END_IF;
END_REGION

REGION Network 2: ALARME DE BALANCA
   // BALANÇA INFERIOR/SUPERIOR.
   RUNG wire#powerrail
      Contact( "DB ESTICADOR".COMANDOS.SELECIONADO )
      wire#w1
      { S7_Templates := "SrcType := Int" } LT_Contact(in1 := "P_PIW406":P, in2 := 2700)
      Contact( "DB PRINCIPAL".COMANDOS.MARCHA )
      wire#w2
      S_Coil( "DB ESTICADOR".ALARMES.BALANCA_INFERIOR )
   END_RUNG
   RUNG wire#w2
      S_Coil( "DB PRINCIPAL".COMANDOS.BALANCA_FORA_POSICAO )
   END_RUNG
   RUNG wire#w1
      { S7_Templates := "SrcType := Int" } GT_Contact(in1 := "P_PIW406":P, in2 := 24900)
      Contact( "DB PRINCIPAL".COMANDOS.MARCHA )
      wire#w3
      S_Coil( "DB ESTICADOR".ALARMES.BALANCA_SUPERIOR )
   END_RUNG
   RUNG wire#w3
      S_Coil( "DB PRINCIPAL".COMANDOS.BALANCA_FORA_POSICAO )
   END_RUNG
   RUNG wire#w1
      Contact( "DB PRINCIPAL".COMANDOS.BALANCA_TRAVA )
      wire#w4
      R_Coil( "DB ESTICADOR".ALARMES.BALANCA_INFERIOR )
   END_RUNG
   RUNG wire#w4
      R_Coil( "DB ESTICADOR".ALARMES.BALANCA_SUPERIOR )
   END_RUNG
   // the same network as SCL:
   IF "DB ESTICADOR".COMANDOS.SELECIONADO AND ("P_PIW406":P < 2700) AND "DB PRINCIPAL".COMANDOS.MARCHA THEN
       "DB ESTICADOR".ALARMES.BALANCA_INFERIOR := TRUE;
       "DB PRINCIPAL".COMANDOS.BALANCA_FORA_POSICAO := TRUE;
   END_IF;
   IF "DB ESTICADOR".COMANDOS.SELECIONADO AND ("P_PIW406":P > 24900) AND "DB PRINCIPAL".COMANDOS.MARCHA THEN
       "DB ESTICADOR".ALARMES.BALANCA_SUPERIOR := TRUE;
       "DB PRINCIPAL".COMANDOS.BALANCA_FORA_POSICAO := TRUE;
   END_IF;
   IF "DB ESTICADOR".COMANDOS.SELECIONADO AND "DB PRINCIPAL".COMANDOS.BALANCA_TRAVA THEN
       "DB ESTICADOR".ALARMES.BALANCA_INFERIOR := FALSE;
       "DB ESTICADOR".ALARMES.BALANCA_SUPERIOR := FALSE;
   END_IF;
END_REGION

REGION Network 3: ALARME DE NIVEL ALTO
   // PROTEÇÃO DO INVERSOR DE FREQUENCIA
   RUNG wire#powerrail
      I_Contact( "DB ESTICADOR".COMANDOS.STATUS_DRIVER )
      wire#w1
      S_Coil( "DB ESTICADOR".ALARMES.PROTECAO_INVERSOR )
   END_RUNG
   RUNG wire#w1
      I_Contact( "DB ESTICADOR".COMANDOS.SELECIONADO )
      R_Coil( "DB ESTICADOR".ALARMES.PROTECAO_INVERSOR )
   END_RUNG
   // the same network as SCL:
   #_w1 := NOT "DB ESTICADOR".COMANDOS.STATUS_DRIVER;
   IF #_w1 THEN "DB ESTICADOR".ALARMES.PROTECAO_INVERSOR := TRUE; END_IF;
   IF #_w1 AND NOT "DB ESTICADOR".COMANDOS.SELECIONADO THEN
       "DB ESTICADOR".ALARMES.PROTECAO_INVERSOR := FALSE;
   END_IF;
END_REGION

REGION Network 4: ALARMES
   // ATIVAÇÃO DO BIT DE ALARME DE NIVEL ALTO
   // ATIVAÇÃO DO BIT DE ALARME DE NIVEL BAIXO
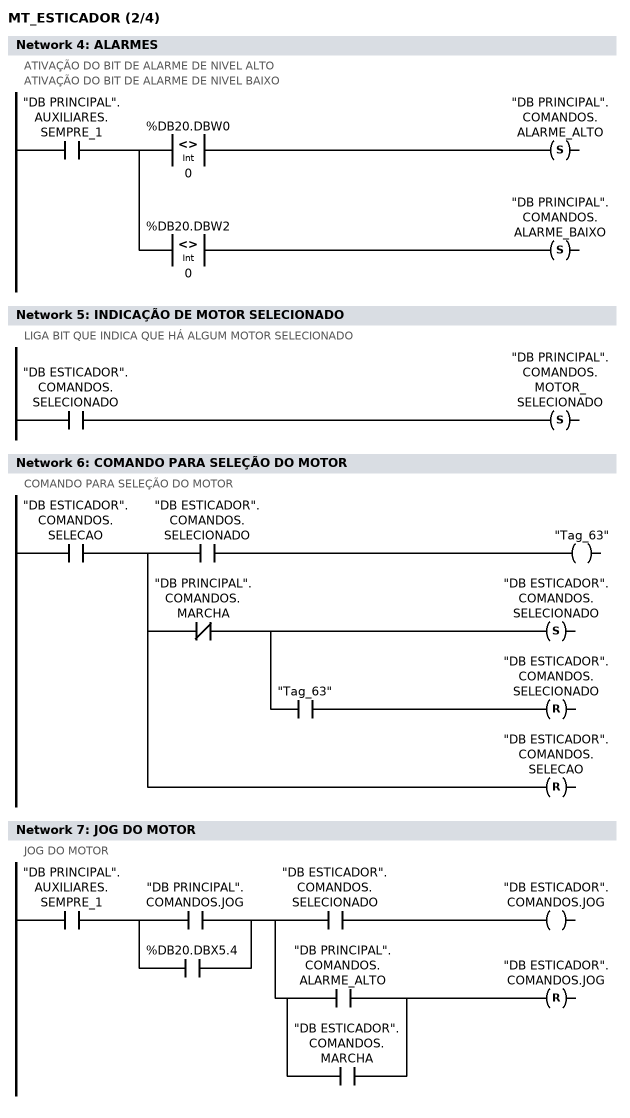
   RUNG wire#powerrail
      Contact( "DB PRINCIPAL".AUXILIARES.SEMPRE_1 )
      wire#w1
      { S7_Templates := "SrcType := Int" } NE_Contact(in1 := %DB20.DBW0, in2 := 0)
      S_Coil( "DB PRINCIPAL".COMANDOS.ALARME_ALTO )
   END_RUNG
   RUNG wire#w1
      { S7_Templates := "SrcType := Int" } NE_Contact(in1 := %DB20.DBW2, in2 := 0)
      S_Coil( "DB PRINCIPAL".COMANDOS.ALARME_BAIXO )
   END_RUNG
   // the same network as SCL:
   IF "DB PRINCIPAL".AUXILIARES.SEMPRE_1 AND (%DB20.DBW0 <> 0) THEN
       "DB PRINCIPAL".COMANDOS.ALARME_ALTO := TRUE;
   END_IF;
   IF "DB PRINCIPAL".AUXILIARES.SEMPRE_1 AND (%DB20.DBW2 <> 0) THEN
       "DB PRINCIPAL".COMANDOS.ALARME_BAIXO := TRUE;
   END_IF;
END_REGION

REGION Network 5: INDICAÇÃO DE MOTOR SELECIONADO
   // LIGA BIT QUE INDICA QUE HÁ ALGUM MOTOR SELECIONADO
   RUNG wire#powerrail
      Contact( "DB ESTICADOR".COMANDOS.SELECIONADO )
      S_Coil( "DB PRINCIPAL".COMANDOS.MOTOR_SELECIONADO )
   END_RUNG
   // the same network as SCL:
   IF "DB ESTICADOR".COMANDOS.SELECIONADO THEN "DB PRINCIPAL".COMANDOS.MOTOR_SELECIONADO := TRUE; END_IF;
END_REGION

REGION Network 6: COMANDO PARA SELEÇÃO DO MOTOR
   // COMANDO PARA SELEÇÃO DO MOTOR
   RUNG wire#powerrail
      Contact( "DB ESTICADOR".COMANDOS.SELECAO )
      wire#w1
      Contact( "DB ESTICADOR".COMANDOS.SELECIONADO )
      Coil( "Tag_63" )
   END_RUNG
   RUNG wire#w1
      I_Contact( "DB PRINCIPAL".COMANDOS.MARCHA )
      wire#w2
      S_Coil( "DB ESTICADOR".COMANDOS.SELECIONADO )
   END_RUNG
   RUNG wire#w2
      Contact( "Tag_63" )
      R_Coil( "DB ESTICADOR".COMANDOS.SELECIONADO )
   END_RUNG
   RUNG wire#w1
      R_Coil( "DB ESTICADOR".COMANDOS.SELECAO )
   END_RUNG
   // the same network as SCL:
   "Tag_63" := "DB ESTICADOR".COMANDOS.SELECAO AND "DB ESTICADOR".COMANDOS.SELECIONADO;
   #_w1 := "DB ESTICADOR".COMANDOS.SELECAO AND NOT "DB PRINCIPAL".COMANDOS.MARCHA;
   IF #_w1 THEN "DB ESTICADOR".COMANDOS.SELECIONADO := TRUE; END_IF;
   IF #_w1 AND "Tag_63" THEN "DB ESTICADOR".COMANDOS.SELECIONADO := FALSE; END_IF;
   IF "DB ESTICADOR".COMANDOS.SELECAO THEN "DB ESTICADOR".COMANDOS.SELECAO := FALSE; END_IF;
END_REGION

REGION Network 7: JOG DO MOTOR
   // JOG DO MOTOR
   RUNG wire#powerrail
      Contact( "DB PRINCIPAL".AUXILIARES.SEMPRE_1 )
      wire#w1
      Contact( "DB PRINCIPAL".COMANDOS.JOG )
      wire#w2
      Contact( "DB ESTICADOR".COMANDOS.SELECIONADO )
      Coil( "DB ESTICADOR".COMANDOS.JOG )
   END_RUNG
   RUNG wire#w1
      Contact( %DB20.DBX5.4 )
   END_RUNG wire#w2
   RUNG wire#w2
      Contact( "DB PRINCIPAL".COMANDOS.ALARME_ALTO )
      wire#w3
      R_Coil( "DB ESTICADOR".COMANDOS.JOG )
   END_RUNG
   RUNG wire#w2
      Contact( "DB ESTICADOR".COMANDOS.MARCHA )
   END_RUNG wire#w3
   // the same network as SCL:
   #_w1 := "DB PRINCIPAL".AUXILIARES.SEMPRE_1 AND ("DB PRINCIPAL".COMANDOS.JOG OR %DB20.DBX5.4);
   "DB ESTICADOR".COMANDOS.JOG := #_w1 AND "DB ESTICADOR".COMANDOS.SELECIONADO;
   IF #_w1 AND ("DB PRINCIPAL".COMANDOS.ALARME_ALTO OR "DB ESTICADOR".COMANDOS.MARCHA) THEN
       "DB ESTICADOR".COMANDOS.JOG := FALSE;
   END_IF;
END_REGION

REGION Network 8: COMANDO PARA LIBERAÇÃO DO MOTOR
   // COMANDO PARA LIBERAÇÃO DO MOTOR
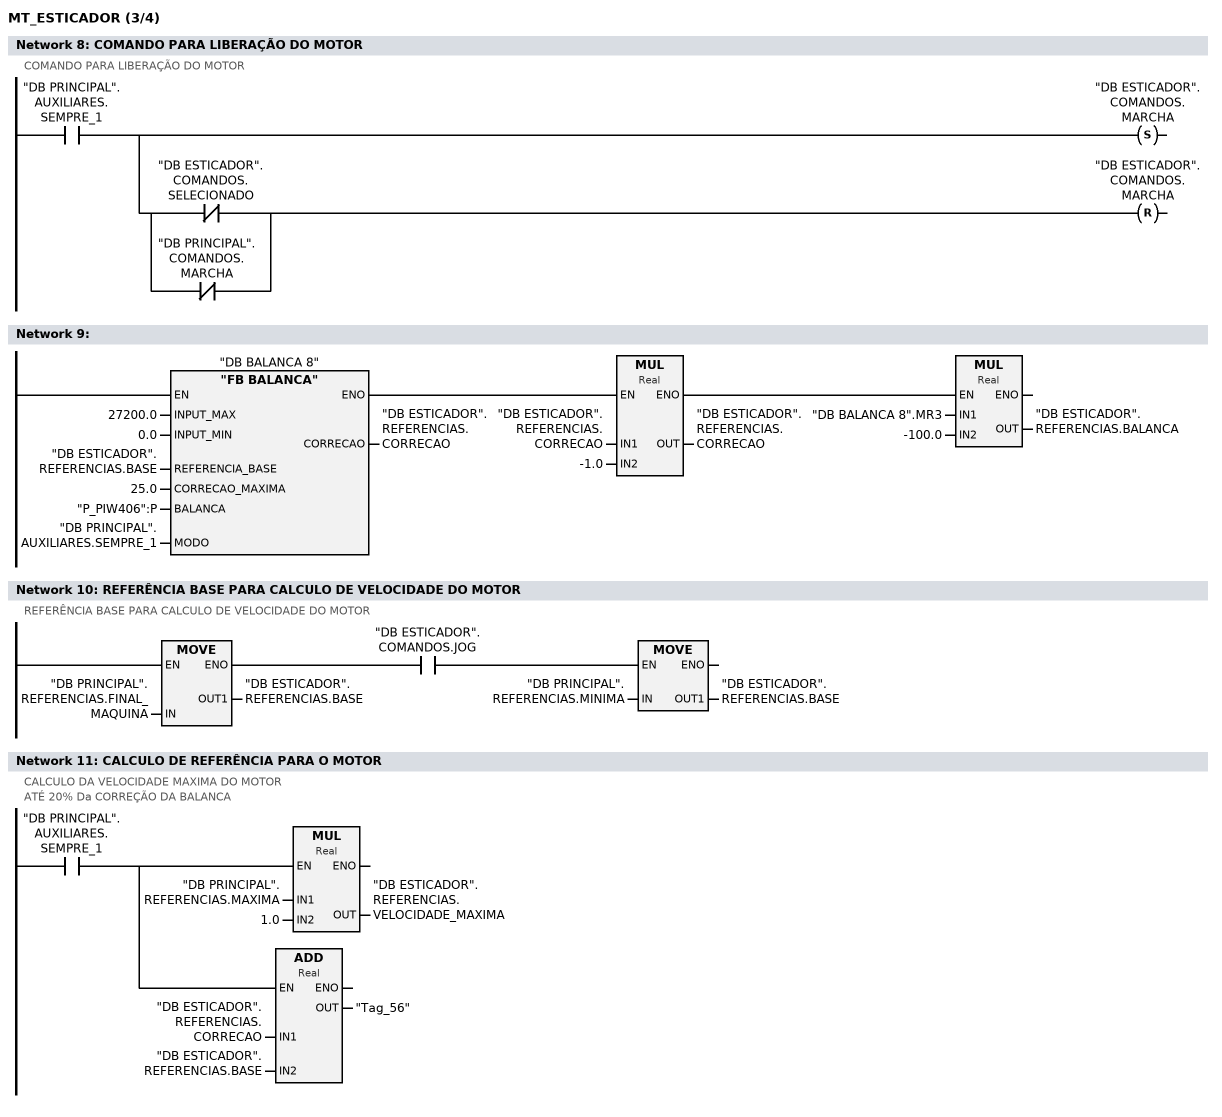
   RUNG wire#powerrail
      Contact( "DB PRINCIPAL".AUXILIARES.SEMPRE_1 )
      wire#w1
      S_Coil( "DB ESTICADOR".COMANDOS.MARCHA )
   END_RUNG
   RUNG wire#w1
      I_Contact( "DB ESTICADOR".COMANDOS.SELECIONADO )
      wire#w2
      R_Coil( "DB ESTICADOR".COMANDOS.MARCHA )
   END_RUNG
   RUNG wire#w1
      I_Contact( "DB PRINCIPAL".COMANDOS.MARCHA )
   END_RUNG wire#w2
   // the same network as SCL:
   IF "DB PRINCIPAL".AUXILIARES.SEMPRE_1 THEN "DB ESTICADOR".COMANDOS.MARCHA := TRUE; END_IF;
   IF "DB PRINCIPAL".AUXILIARES.SEMPRE_1 AND (NOT "DB ESTICADOR".COMANDOS.SELECIONADO OR NOT "DB PRINCIPAL".COMANDOS.MARCHA) THEN
       "DB ESTICADOR".COMANDOS.MARCHA := FALSE;
   END_IF;
END_REGION

REGION Network 9
   RUNG wire#powerrail
      "DB BALANCA 8"(INPUT_MAX := 27200.0, INPUT_MIN := 0.0, REFERENCIA_BASE := "DB ESTICADOR".REFERENCIAS.BASE, CORRECAO_MAXIMA := 25.0, BALANCA := "P_PIW406":P, MODO := "DB PRINCIPAL".AUXILIARES.SEMPRE_1, CORRECAO => "DB ESTICADOR".REFERENCIAS.CORRECAO)
      { S7_Templates := "SrcType := Real"; S7_GenerateENO := "TRUE" } Mul(in1 := "DB ESTICADOR".REFERENCIAS.CORRECAO, in2 := -1.0, out => "DB ESTICADOR".REFERENCIAS.CORRECAO)
      { S7_Templates := "SrcType := Real"; S7_GenerateENO := "TRUE" } Mul(in1 := "DB BALANCA 8".MR3, in2 := -100.0, out => "DB ESTICADOR".REFERENCIAS.BALANCA)
   END_RUNG
   // the same network as SCL:
   // ENO of a box is taken as its EN; it also drops when the box reports an error
   "DB BALANCA 8"(INPUT_MAX := 27200.0,   // "FB BALANCA"
                  INPUT_MIN := 0.0,
                  REFERENCIA_BASE := "DB ESTICADOR".REFERENCIAS.BASE,
                  CORRECAO_MAXIMA := 25.0,
                  BALANCA := "P_PIW406":P,
                  MODO := "DB PRINCIPAL".AUXILIARES.SEMPRE_1,
                  CORRECAO => "DB ESTICADOR".REFERENCIAS.CORRECAO,
                  ENO => #_w1);
   IF #_w1 THEN
       "DB ESTICADOR".REFERENCIAS.CORRECAO := "DB ESTICADOR".REFERENCIAS.CORRECAO * (-1.0);
       "DB ESTICADOR".REFERENCIAS.BALANCA := "DB BALANCA 8".MR3 * (-100.0);
   END_IF;
END_REGION

REGION Network 10: REFERÊNCIA BASE PARA CALCULO DE VELOCIDADE DO MOTOR
   // REFERÊNCIA BASE PARA CALCULO DE VELOCIDADE DO MOTOR
   RUNG wire#powerrail
      { S7_GenerateENO := "TRUE" } Move(in := "DB PRINCIPAL".REFERENCIAS.FINAL_MAQUINA, out1 => "DB ESTICADOR".REFERENCIAS.BASE)
      Contact( "DB ESTICADOR".COMANDOS.JOG )
      { S7_GenerateENO := "TRUE" } Move(in := "DB PRINCIPAL".REFERENCIAS.MINIMA, out1 => "DB ESTICADOR".REFERENCIAS.BASE)
   END_RUNG
   // the same network as SCL:
   // ENO of a box is taken as its EN; it also drops when the box reports an error
   "DB ESTICADOR".REFERENCIAS.BASE := "DB PRINCIPAL".REFERENCIAS.FINAL_MAQUINA;
   IF "DB ESTICADOR".COMANDOS.JOG THEN
       "DB ESTICADOR".REFERENCIAS.BASE := "DB PRINCIPAL".REFERENCIAS.MINIMA;
   END_IF;
END_REGION

REGION Network 11: CALCULO DE REFERÊNCIA PARA O MOTOR
   // CALCULO DA VELOCIDADE MAXIMA DO MOTOR
   // ATÉ 20% Da CORREÇÃO DA BALANCA
   RUNG wire#powerrail
      Contact( "DB PRINCIPAL".AUXILIARES.SEMPRE_1 )
      wire#w1
      { S7_Templates := "SrcType := Real"; S7_GenerateENO := "TRUE" } Mul(in1 := "DB PRINCIPAL".REFERENCIAS.MAXIMA, in2 := 1.0, out => "DB ESTICADOR".REFERENCIAS.VELOCIDADE_MAXIMA)
   END_RUNG
   RUNG wire#w1
      { S7_Templates := "SrcType := Real"; S7_GenerateENO := "TRUE" } Add(in1 := "DB ESTICADOR".REFERENCIAS.CORRECAO, in2 := "DB ESTICADOR".REFERENCIAS.BASE, out => "Tag_56")
   END_RUNG
   // the same network as SCL:
   IF "DB PRINCIPAL".AUXILIARES.SEMPRE_1 THEN
       "DB ESTICADOR".REFERENCIAS.VELOCIDADE_MAXIMA := "DB PRINCIPAL".REFERENCIAS.MAXIMA * 1.0;
       "Tag_56" := "DB ESTICADOR".REFERENCIAS.CORRECAO + "DB ESTICADOR".REFERENCIAS.BASE;
   END_IF;
END_REGION

REGION Network 12: ACC/DEC DA REFERÊNCIA DO MOTOR
   // ACC/DEC DA REFERÊNCIA DO MOTOR
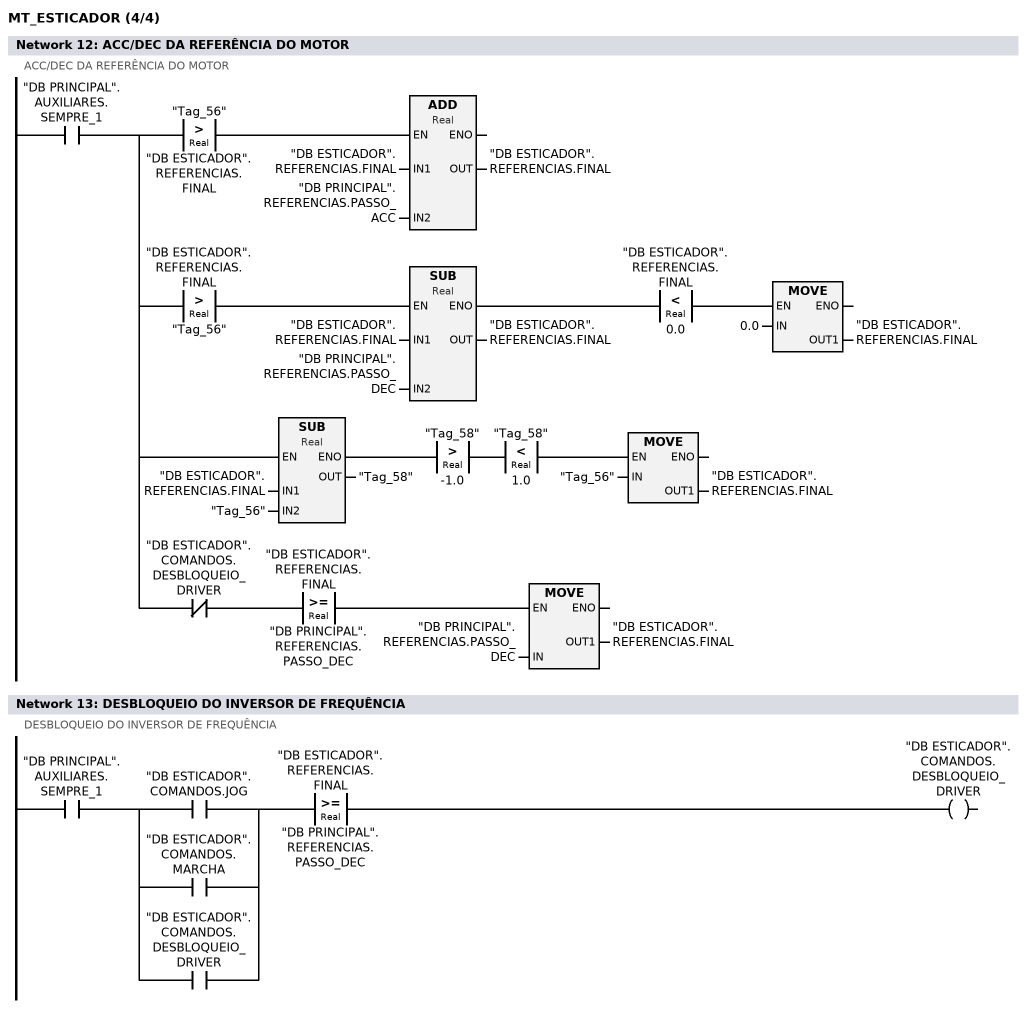
   RUNG wire#powerrail
      Contact( "DB PRINCIPAL".AUXILIARES.SEMPRE_1 )
      wire#w1
      { S7_Templates := "SrcType := Real" } GT_Contact(in1 := "Tag_56", in2 := "DB ESTICADOR".REFERENCIAS.FINAL)
      { S7_Templates := "SrcType := Real"; S7_GenerateENO := "TRUE" } Add(in1 := "DB ESTICADOR".REFERENCIAS.FINAL, in2 := "DB PRINCIPAL".REFERENCIAS.PASSO_ACC, out => "DB ESTICADOR".REFERENCIAS.FINAL)
   END_RUNG
   RUNG wire#w1
      { S7_Templates := "SrcType := Real" } GT_Contact(in1 := "DB ESTICADOR".REFERENCIAS.FINAL, in2 := "Tag_56")
      { S7_Templates := "SrcType := Real"; S7_GenerateENO := "TRUE" } Sub(in1 := "DB ESTICADOR".REFERENCIAS.FINAL, in2 := "DB PRINCIPAL".REFERENCIAS.PASSO_DEC, out => "DB ESTICADOR".REFERENCIAS.FINAL)
      { S7_Templates := "SrcType := Real" } LT_Contact(in1 := "DB ESTICADOR".REFERENCIAS.FINAL, in2 := 0.0)
      { S7_GenerateENO := "TRUE" } Move(in := 0.0, out1 => "DB ESTICADOR".REFERENCIAS.FINAL)
   END_RUNG
   RUNG wire#w1
      { S7_Templates := "SrcType := Real"; S7_GenerateENO := "TRUE" } Sub(in1 := "DB ESTICADOR".REFERENCIAS.FINAL, in2 := "Tag_56", out => "Tag_58")
      { S7_Templates := "SrcType := Real" } GT_Contact(in1 := "Tag_58", in2 := -1.0)
      { S7_Templates := "SrcType := Real" } LT_Contact(in1 := "Tag_58", in2 := 1.0)
      { S7_GenerateENO := "TRUE" } Move(in := "Tag_56", out1 => "DB ESTICADOR".REFERENCIAS.FINAL)
   END_RUNG
   RUNG wire#w1
      I_Contact( "DB ESTICADOR".COMANDOS.DESBLOQUEIO_DRIVER )
      { S7_Templates := "SrcType := Real" } GE_Contact(in1 := "DB ESTICADOR".REFERENCIAS.FINAL, in2 := "DB PRINCIPAL".REFERENCIAS.PASSO_DEC)
      { S7_GenerateENO := "TRUE" } Move(in := "DB PRINCIPAL".REFERENCIAS.PASSO_DEC, out1 => "DB ESTICADOR".REFERENCIAS.FINAL)
   END_RUNG
   // the same network as SCL:
   // ENO of a box is taken as its EN; it also drops when the box reports an error
   IF "DB PRINCIPAL".AUXILIARES.SEMPRE_1 AND ("Tag_56" > "DB ESTICADOR".REFERENCIAS.FINAL) THEN
       "DB ESTICADOR".REFERENCIAS.FINAL := "DB ESTICADOR".REFERENCIAS.FINAL + "DB PRINCIPAL".REFERENCIAS.PASSO_ACC;
   END_IF;
   #_w1 := "DB PRINCIPAL".AUXILIARES.SEMPRE_1 AND ("DB ESTICADOR".REFERENCIAS.FINAL > "Tag_56");
   IF #_w1 THEN
       "DB ESTICADOR".REFERENCIAS.FINAL := "DB ESTICADOR".REFERENCIAS.FINAL - "DB PRINCIPAL".REFERENCIAS.PASSO_DEC;
   END_IF;
   IF #_w1 AND ("DB ESTICADOR".REFERENCIAS.FINAL < 0.0) THEN "DB ESTICADOR".REFERENCIAS.FINAL := 0.0; END_IF;
   IF "DB PRINCIPAL".AUXILIARES.SEMPRE_1 THEN
       "Tag_58" := "DB ESTICADOR".REFERENCIAS.FINAL - "Tag_56";
   END_IF;
   IF "DB PRINCIPAL".AUXILIARES.SEMPRE_1 AND ("Tag_58" > (-1.0)) AND ("Tag_58" < 1.0) THEN
       "DB ESTICADOR".REFERENCIAS.FINAL := "Tag_56";
   END_IF;
   IF "DB PRINCIPAL".AUXILIARES.SEMPRE_1 AND NOT "DB ESTICADOR".COMANDOS.DESBLOQUEIO_DRIVER AND ("DB ESTICADOR".REFERENCIAS.FINAL >= "DB PRINCIPAL".REFERENCIAS.PASSO_DEC) THEN
       "DB ESTICADOR".REFERENCIAS.FINAL := "DB PRINCIPAL".REFERENCIAS.PASSO_DEC;
   END_IF;
END_REGION

REGION Network 13: DESBLOQUEIO DO INVERSOR DE FREQUÊNCIA
   // DESBLOQUEIO DO INVERSOR DE FREQUÊNCIA
   RUNG wire#powerrail
      Contact( "DB PRINCIPAL".AUXILIARES.SEMPRE_1 )
      wire#w1
      Contact( "DB ESTICADOR".COMANDOS.JOG )
      wire#w2
      { S7_Templates := "SrcType := Real" } GE_Contact(in1 := "DB ESTICADOR".REFERENCIAS.FINAL, in2 := "DB PRINCIPAL".REFERENCIAS.PASSO_DEC)
      Coil( "DB ESTICADOR".COMANDOS.DESBLOQUEIO_DRIVER )
   END_RUNG
   RUNG wire#w1
      Contact( "DB ESTICADOR".COMANDOS.MARCHA )
   END_RUNG wire#w2
   RUNG wire#w1
      Contact( "DB ESTICADOR".COMANDOS.DESBLOQUEIO_DRIVER )
   END_RUNG wire#w2
   // the same network as SCL:
   "DB ESTICADOR".COMANDOS.DESBLOQUEIO_DRIVER := "DB PRINCIPAL".AUXILIARES.SEMPRE_1 AND ("DB ESTICADOR".COMANDOS.JOG OR "DB ESTICADOR".COMANDOS.MARCHA OR "DB ESTICADOR".COMANDOS.DESBLOQUEIO_DRIVER) AND ("DB ESTICADOR".REFERENCIAS.FINAL >= "DB PRINCIPAL".REFERENCIAS.PASSO_DEC);
END_REGION

REGION Network 14 (STL): STATUS / CONTROLE - INVERSOR DE FREQUÊNCIA
   // DANFOSS FC300 PROFIBUS - TEX24626INV001
   // STATUS DO INVERSOR DE FREQUÊNCIA
         L     "Tag_33":P;
         T     "Tag_1";
         AN    "Tag_59";
         =     "DB ESTICADOR".COMANDOS.STATUS_DRIVER;

   // CONTROLE DO INVERSOR DE FREQUÊNCIA
         L     1150;
         T     "Tag_1";
         A     "DB ESTICADOR".COMANDOS.DESBLOQUEIO_DRIVER;
         =     "Tag_60";
         A     "T2";
         AN    "DB ESTICADOR".COMANDOS.STATUS_DRIVER;
         =     "Tag_61";
         L     "Tag_1";
         T     "Tag_34":P;

   // REFERÊNCIA PARA O INVERSOR DE FREQUÊNCIA
         L     "DB ESTICADOR".REFERENCIAS.FINAL;
         L     16384.0;
         *R;

         L     "DB ESTICADOR".REFERENCIAS.VELOCIDADE_MAXIMA;
         /R;
         RND;
         T     "Tag_62";
         L     "Tag_62";
         T     "Tag_35":P;
END_REGION

REGION Network 15 (STL): INVERSOR RESERVA
         A     "DB PRINCIPAL".AUXILIARES.SEMPRE_1;
         =     %L24.0;
         A     %L24.0;
         A(;
         L     "DB PRINCIPAL".AUXILIARES1.INVERSOR_RESERVA1;
         L     11;
         ==I;
         );
         =     %L24.1;
         A     %L24.1;
         JNB   M001;
         L     "DB ESTICADOR".REFERENCIAS.FINAL;
         L     3.456;
         *R;
         T     #AUX_R;
         RND;
         T     "P_QW100":P;
   M001: NOP   0;
         A     %L24.1;
         A     "I130";
         S     "DB PRINCIPAL".ALARME.INV_RESERVA1;
         A     %L24.1;
         A     "DB ESTICADOR".COMANDOS.DESBLOQUEIO_DRIVER;
         S     "Q134";
         A     %L24.1;
         AN    "DB ESTICADOR".COMANDOS.DESBLOQUEIO_DRIVER;
         R     "Q134";
         A     %L24.0;
         A(;
         L     "DB PRINCIPAL".AUXILIARES1.INVERSOR_RESERVA2;
         L     11;
         ==I;
         );
         =     %L24.1;
         A     %L24.1;
         JNB   M002;
         L     "DB ESTICADOR".REFERENCIAS.FINAL;
         L     3.456;
         *R;
         T     #AUX_R;
         RND;
         T     "P_QW102":P;
   M002: NOP   0;
         A     %L24.1;
         A     "I132";
         S     "DB PRINCIPAL".ALARME.INV_RESERVA2;
         A     %L24.1;
         A     "DB ESTICADOR".COMANDOS.DESBLOQUEIO_DRIVER;
         S     "Q135";
         A     %L24.1;
         AN    "DB ESTICADOR".COMANDOS.DESBLOQUEIO_DRIVER;
         R     "Q135";
END_REGION
END_FUNCTION

FUNCTION "MT_PUXADOR_SECADEIRA2" : Void   // FC21, LAD
TITLE = MÓDULO DE CONTROLE DO PUXADOR DA SECADEIRA 2
{ S7_Optimized_Access := 'FALSE' }
AUTHOR : THALLES
FAMILY : TRAÇÃO
NAME : LINHA1
VERSION : 0.1
// DATA BLOCK DE CONTROLE // DB21
// Automation Pack Automação Indl. e Com. Ltda.
// Cliente: Texima S/A Ind. de Máquinas
// Cliente Final: Cia. Fiação e Tecidos Santo Antonio.
// Máquina: LINHA 1 DENIN - O.S.: 24.626
   VAR_TEMP
      AUX_R : Real;
   END_VAR
   VAR_TEMP   // added for the SCL form of the ladder/FBD networks
      _w1 : Bool;
   END_VAR
BEGIN

REGION Network 1: ALARMES
   // RESET DOS ALARMES
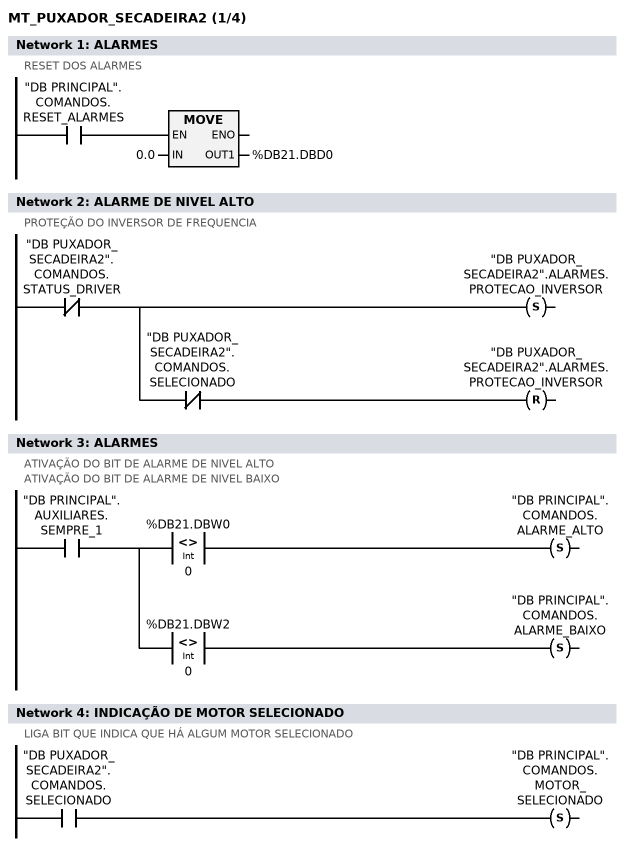
   RUNG wire#powerrail
      Contact( "DB PRINCIPAL".COMANDOS.RESET_ALARMES )
      { S7_GenerateENO := "TRUE" } Move(in := 0.0, out1 => %DB21.DBD0)
   END_RUNG
   // the same network as SCL:
   IF "DB PRINCIPAL".COMANDOS.RESET_ALARMES THEN %DB21.DBD0 := 0.0; END_IF;
END_REGION

REGION Network 2: ALARME DE NIVEL ALTO
   // PROTEÇÃO DO INVERSOR DE FREQUENCIA
   RUNG wire#powerrail
      I_Contact( "DB PUXADOR_SECADEIRA2".COMANDOS.STATUS_DRIVER )
      wire#w1
      S_Coil( "DB PUXADOR_SECADEIRA2".ALARMES.PROTECAO_INVERSOR )
   END_RUNG
   RUNG wire#w1
      I_Contact( "DB PUXADOR_SECADEIRA2".COMANDOS.SELECIONADO )
      R_Coil( "DB PUXADOR_SECADEIRA2".ALARMES.PROTECAO_INVERSOR )
   END_RUNG
   // the same network as SCL:
   #_w1 := NOT "DB PUXADOR_SECADEIRA2".COMANDOS.STATUS_DRIVER;
   IF #_w1 THEN "DB PUXADOR_SECADEIRA2".ALARMES.PROTECAO_INVERSOR := TRUE; END_IF;
   IF #_w1 AND NOT "DB PUXADOR_SECADEIRA2".COMANDOS.SELECIONADO THEN
       "DB PUXADOR_SECADEIRA2".ALARMES.PROTECAO_INVERSOR := FALSE;
   END_IF;
END_REGION

REGION Network 3: ALARMES
   // ATIVAÇÃO DO BIT DE ALARME DE NIVEL ALTO
   // ATIVAÇÃO DO BIT DE ALARME DE NIVEL BAIXO
   RUNG wire#powerrail
      Contact( "DB PRINCIPAL".AUXILIARES.SEMPRE_1 )
      wire#w1
      { S7_Templates := "SrcType := Int" } NE_Contact(in1 := %DB21.DBW0, in2 := 0)
      S_Coil( "DB PRINCIPAL".COMANDOS.ALARME_ALTO )
   END_RUNG
   RUNG wire#w1
      { S7_Templates := "SrcType := Int" } NE_Contact(in1 := %DB21.DBW2, in2 := 0)
      S_Coil( "DB PRINCIPAL".COMANDOS.ALARME_BAIXO )
   END_RUNG
   // the same network as SCL:
   IF "DB PRINCIPAL".AUXILIARES.SEMPRE_1 AND (%DB21.DBW0 <> 0) THEN
       "DB PRINCIPAL".COMANDOS.ALARME_ALTO := TRUE;
   END_IF;
   IF "DB PRINCIPAL".AUXILIARES.SEMPRE_1 AND (%DB21.DBW2 <> 0) THEN
       "DB PRINCIPAL".COMANDOS.ALARME_BAIXO := TRUE;
   END_IF;
END_REGION

REGION Network 4: INDICAÇÃO DE MOTOR SELECIONADO
   // LIGA BIT QUE INDICA QUE HÁ ALGUM MOTOR SELECIONADO
   RUNG wire#powerrail
      Contact( "DB PUXADOR_SECADEIRA2".COMANDOS.SELECIONADO )
      S_Coil( "DB PRINCIPAL".COMANDOS.MOTOR_SELECIONADO )
   END_RUNG
   // the same network as SCL:
   IF "DB PUXADOR_SECADEIRA2".COMANDOS.SELECIONADO THEN
       "DB PRINCIPAL".COMANDOS.MOTOR_SELECIONADO := TRUE;
   END_IF;
END_REGION

REGION Network 5: COMANDO PARA SELEÇÃO DO MOTOR
   // COMANDO PARA SELEÇÃO DO MOTOR
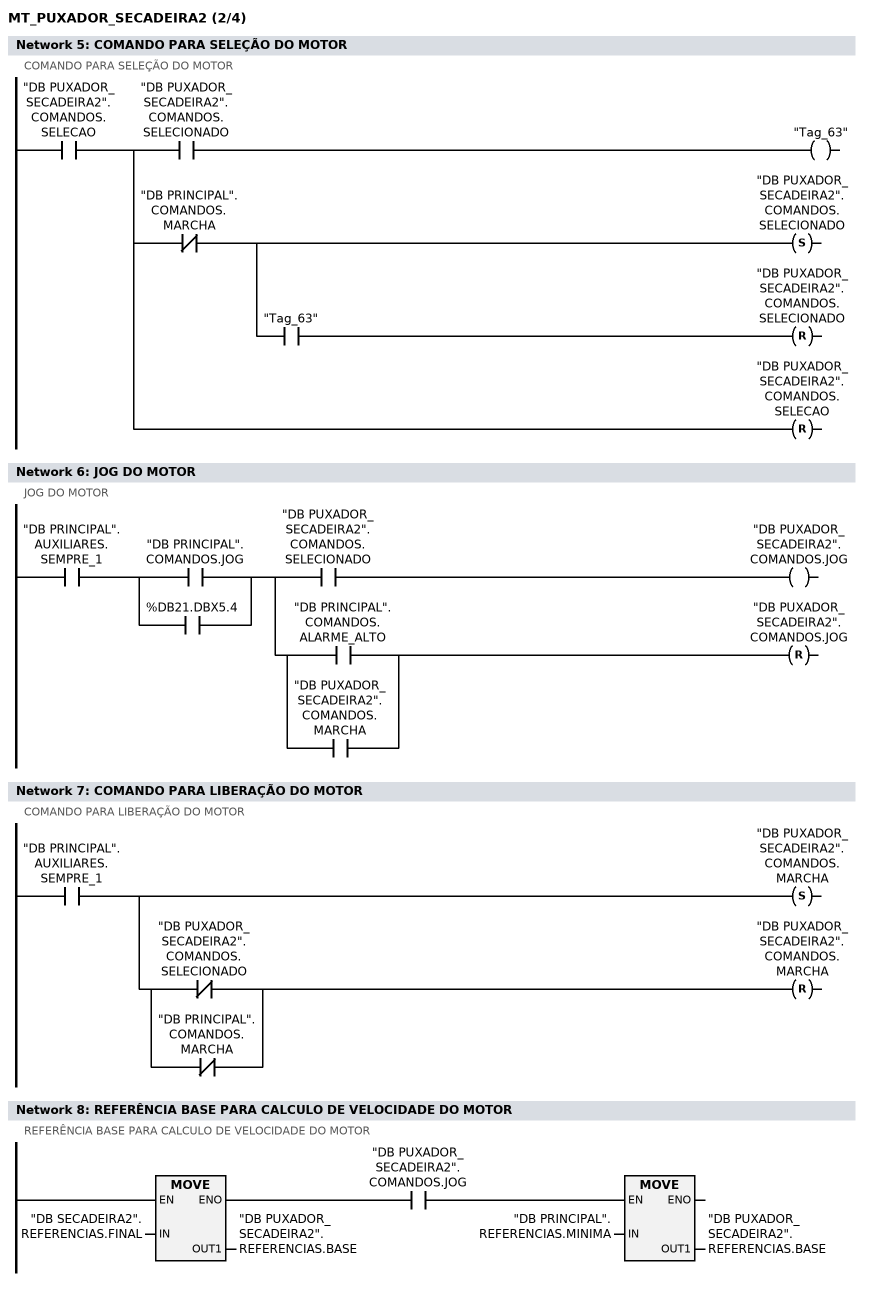
   RUNG wire#powerrail
      Contact( "DB PUXADOR_SECADEIRA2".COMANDOS.SELECAO )
      wire#w1
      Contact( "DB PUXADOR_SECADEIRA2".COMANDOS.SELECIONADO )
      Coil( "Tag_63" )
   END_RUNG
   RUNG wire#w1
      I_Contact( "DB PRINCIPAL".COMANDOS.MARCHA )
      wire#w2
      S_Coil( "DB PUXADOR_SECADEIRA2".COMANDOS.SELECIONADO )
   END_RUNG
   RUNG wire#w2
      Contact( "Tag_63" )
      R_Coil( "DB PUXADOR_SECADEIRA2".COMANDOS.SELECIONADO )
   END_RUNG
   RUNG wire#w1
      R_Coil( "DB PUXADOR_SECADEIRA2".COMANDOS.SELECAO )
   END_RUNG
   // the same network as SCL:
   "Tag_63" := "DB PUXADOR_SECADEIRA2".COMANDOS.SELECAO AND "DB PUXADOR_SECADEIRA2".COMANDOS.SELECIONADO;
   #_w1 := "DB PUXADOR_SECADEIRA2".COMANDOS.SELECAO AND NOT "DB PRINCIPAL".COMANDOS.MARCHA;
   IF #_w1 THEN "DB PUXADOR_SECADEIRA2".COMANDOS.SELECIONADO := TRUE; END_IF;
   IF #_w1 AND "Tag_63" THEN "DB PUXADOR_SECADEIRA2".COMANDOS.SELECIONADO := FALSE; END_IF;
   IF "DB PUXADOR_SECADEIRA2".COMANDOS.SELECAO THEN
       "DB PUXADOR_SECADEIRA2".COMANDOS.SELECAO := FALSE;
   END_IF;
END_REGION

REGION Network 6: JOG DO MOTOR
   // JOG DO MOTOR
   RUNG wire#powerrail
      Contact( "DB PRINCIPAL".AUXILIARES.SEMPRE_1 )
      wire#w1
      Contact( "DB PRINCIPAL".COMANDOS.JOG )
      wire#w2
      Contact( "DB PUXADOR_SECADEIRA2".COMANDOS.SELECIONADO )
      Coil( "DB PUXADOR_SECADEIRA2".COMANDOS.JOG )
   END_RUNG
   RUNG wire#w1
      Contact( %DB21.DBX5.4 )
   END_RUNG wire#w2
   RUNG wire#w2
      Contact( "DB PRINCIPAL".COMANDOS.ALARME_ALTO )
      wire#w3
      R_Coil( "DB PUXADOR_SECADEIRA2".COMANDOS.JOG )
   END_RUNG
   RUNG wire#w2
      Contact( "DB PUXADOR_SECADEIRA2".COMANDOS.MARCHA )
   END_RUNG wire#w3
   // the same network as SCL:
   #_w1 := "DB PRINCIPAL".AUXILIARES.SEMPRE_1 AND ("DB PRINCIPAL".COMANDOS.JOG OR %DB21.DBX5.4);
   "DB PUXADOR_SECADEIRA2".COMANDOS.JOG := #_w1 AND "DB PUXADOR_SECADEIRA2".COMANDOS.SELECIONADO;
   IF #_w1 AND ("DB PRINCIPAL".COMANDOS.ALARME_ALTO OR "DB PUXADOR_SECADEIRA2".COMANDOS.MARCHA) THEN
       "DB PUXADOR_SECADEIRA2".COMANDOS.JOG := FALSE;
   END_IF;
END_REGION

REGION Network 7: COMANDO PARA LIBERAÇÃO DO MOTOR
   // COMANDO PARA LIBERAÇÃO DO MOTOR
   RUNG wire#powerrail
      Contact( "DB PRINCIPAL".AUXILIARES.SEMPRE_1 )
      wire#w1
      S_Coil( "DB PUXADOR_SECADEIRA2".COMANDOS.MARCHA )
   END_RUNG
   RUNG wire#w1
      I_Contact( "DB PUXADOR_SECADEIRA2".COMANDOS.SELECIONADO )
      wire#w2
      R_Coil( "DB PUXADOR_SECADEIRA2".COMANDOS.MARCHA )
   END_RUNG
   RUNG wire#w1
      I_Contact( "DB PRINCIPAL".COMANDOS.MARCHA )
   END_RUNG wire#w2
   // the same network as SCL:
   IF "DB PRINCIPAL".AUXILIARES.SEMPRE_1 THEN "DB PUXADOR_SECADEIRA2".COMANDOS.MARCHA := TRUE; END_IF;
   IF "DB PRINCIPAL".AUXILIARES.SEMPRE_1 AND (NOT "DB PUXADOR_SECADEIRA2".COMANDOS.SELECIONADO OR NOT "DB PRINCIPAL".COMANDOS.MARCHA) THEN
       "DB PUXADOR_SECADEIRA2".COMANDOS.MARCHA := FALSE;
   END_IF;
END_REGION

REGION Network 8: REFERÊNCIA BASE PARA CALCULO DE VELOCIDADE DO MOTOR
   // REFERÊNCIA BASE PARA CALCULO DE VELOCIDADE DO MOTOR
   RUNG wire#powerrail
      { S7_GenerateENO := "TRUE" } Move(in := "DB SECADEIRA2".REFERENCIAS.FINAL, out1 => "DB PUXADOR_SECADEIRA2".REFERENCIAS.BASE)
      Contact( "DB PUXADOR_SECADEIRA2".COMANDOS.JOG )
      { S7_GenerateENO := "TRUE" } Move(in := "DB PRINCIPAL".REFERENCIAS.MINIMA, out1 => "DB PUXADOR_SECADEIRA2".REFERENCIAS.BASE)
   END_RUNG
   // the same network as SCL:
   // ENO of a box is taken as its EN; it also drops when the box reports an error
   "DB PUXADOR_SECADEIRA2".REFERENCIAS.BASE := "DB SECADEIRA2".REFERENCIAS.FINAL;
   IF "DB PUXADOR_SECADEIRA2".COMANDOS.JOG THEN
       "DB PUXADOR_SECADEIRA2".REFERENCIAS.BASE := "DB PRINCIPAL".REFERENCIAS.MINIMA;
   END_IF;
END_REGION

REGION Network 9: CALCULO DE REFERÊNCIA PARA O MOTOR
   // CALCULO DA VELOCIDADE MAXIMA DO MOTOR
   // ATÉ 20% DE TAXA DE AJUSTE
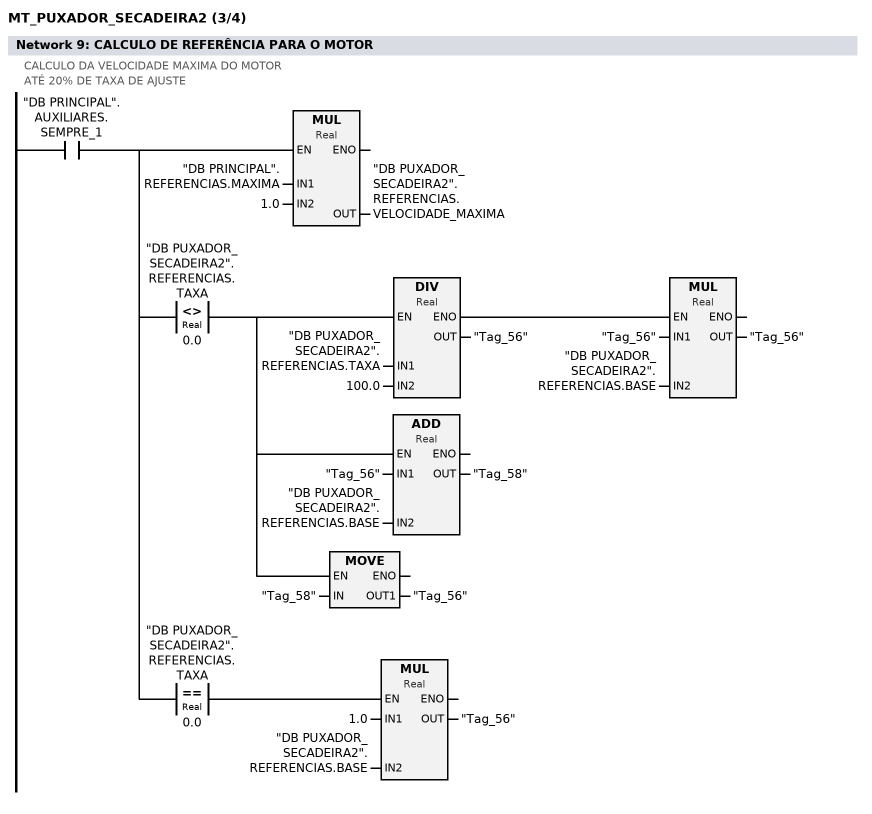
   RUNG wire#powerrail
      Contact( "DB PRINCIPAL".AUXILIARES.SEMPRE_1 )
      wire#w1
      { S7_Templates := "SrcType := Real"; S7_GenerateENO := "TRUE" } Mul(in1 := "DB PRINCIPAL".REFERENCIAS.MAXIMA, in2 := 1.0, out => "DB PUXADOR_SECADEIRA2".REFERENCIAS.VELOCIDADE_MAXIMA)
   END_RUNG
   RUNG wire#w1
      { S7_Templates := "SrcType := Real" } NE_Contact(in1 := "DB PUXADOR_SECADEIRA2".REFERENCIAS.TAXA, in2 := 0.0)
      wire#w2
      { S7_Templates := "SrcType := Real"; S7_GenerateENO := "TRUE" } Div(in1 := "DB PUXADOR_SECADEIRA2".REFERENCIAS.TAXA, in2 := 100.0, out => "Tag_56")
      { S7_Templates := "SrcType := Real"; S7_GenerateENO := "TRUE" } Mul(in1 := "Tag_56", in2 := "DB PUXADOR_SECADEIRA2".REFERENCIAS.BASE, out => "Tag_56")
   END_RUNG
   RUNG wire#w2
      { S7_Templates := "SrcType := Real"; S7_GenerateENO := "TRUE" } Add(in1 := "Tag_56", in2 := "DB PUXADOR_SECADEIRA2".REFERENCIAS.BASE, out => "Tag_58")
   END_RUNG
   RUNG wire#w2
      { S7_GenerateENO := "TRUE" } Move(in := "Tag_58", out1 => "Tag_56")
   END_RUNG
   RUNG wire#w1
      { S7_Templates := "SrcType := Real" } EQ_Contact(in1 := "DB PUXADOR_SECADEIRA2".REFERENCIAS.TAXA, in2 := 0.0)
      { S7_Templates := "SrcType := Real"; S7_GenerateENO := "TRUE" } Mul(in1 := 1.0, in2 := "DB PUXADOR_SECADEIRA2".REFERENCIAS.BASE, out => "Tag_56")
   END_RUNG
   // the same network as SCL:
   // ENO of a box is taken as its EN; it also drops when the box reports an error
   IF "DB PRINCIPAL".AUXILIARES.SEMPRE_1 THEN
       "DB PUXADOR_SECADEIRA2".REFERENCIAS.VELOCIDADE_MAXIMA := "DB PRINCIPAL".REFERENCIAS.MAXIMA * 1.0;
   END_IF;
   IF "DB PRINCIPAL".AUXILIARES.SEMPRE_1 AND ("DB PUXADOR_SECADEIRA2".REFERENCIAS.TAXA <> 0.0) THEN
       "Tag_56" := "DB PUXADOR_SECADEIRA2".REFERENCIAS.TAXA / 100.0;
       "Tag_56" := "Tag_56" * "DB PUXADOR_SECADEIRA2".REFERENCIAS.BASE;
       "Tag_58" := "Tag_56" + "DB PUXADOR_SECADEIRA2".REFERENCIAS.BASE;
       "Tag_56" := "Tag_58";
   END_IF;
   IF "DB PRINCIPAL".AUXILIARES.SEMPRE_1 AND ("DB PUXADOR_SECADEIRA2".REFERENCIAS.TAXA = 0.0) THEN
       "Tag_56" := 1.0 * "DB PUXADOR_SECADEIRA2".REFERENCIAS.BASE;
   END_IF;
END_REGION

REGION Network 10: ACC/DEC DA REFERÊNCIA DO MOTOR
   // ACC/DEC DA REFERÊNCIA DO MOTOR
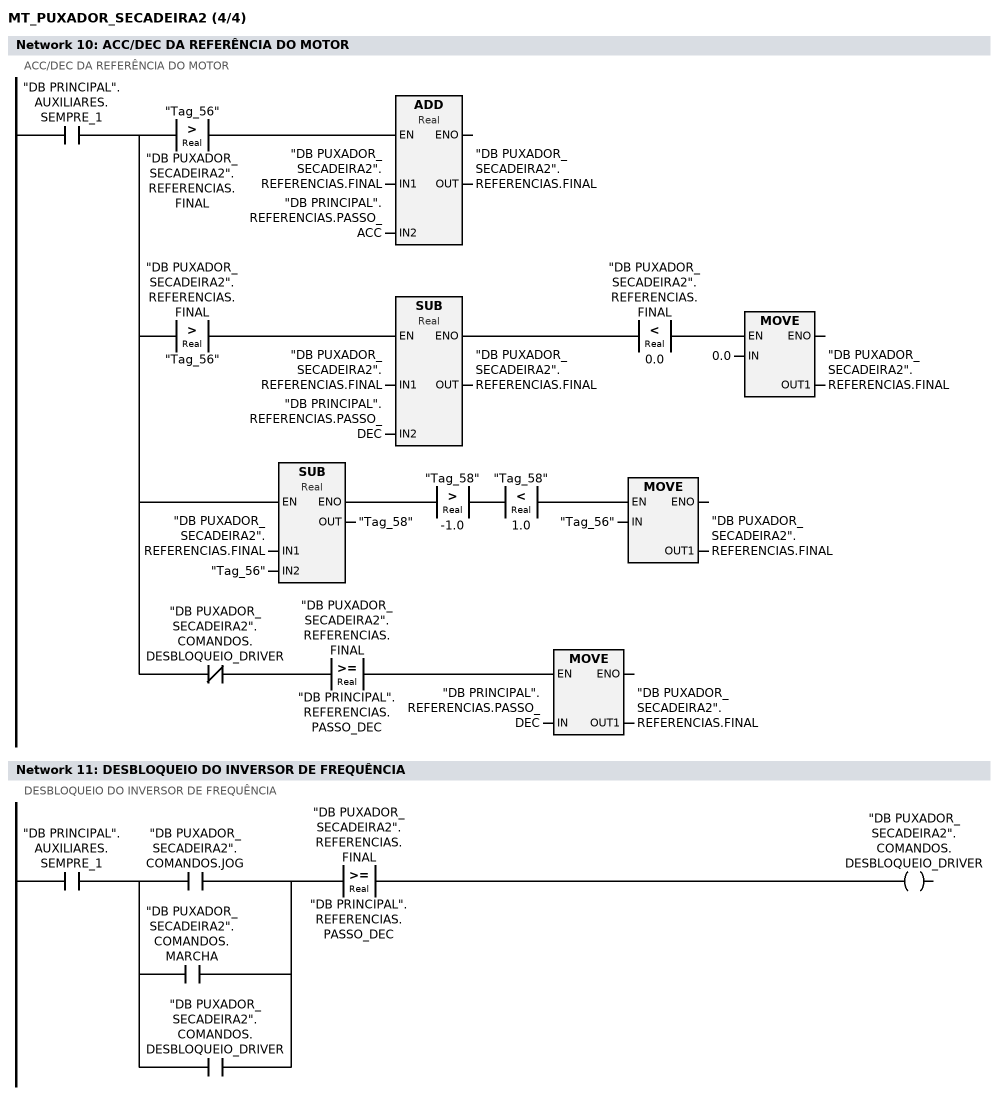
   RUNG wire#powerrail
      Contact( "DB PRINCIPAL".AUXILIARES.SEMPRE_1 )
      wire#w1
      { S7_Templates := "SrcType := Real" } GT_Contact(in1 := "Tag_56", in2 := "DB PUXADOR_SECADEIRA2".REFERENCIAS.FINAL)
      { S7_Templates := "SrcType := Real"; S7_GenerateENO := "TRUE" } Add(in1 := "DB PUXADOR_SECADEIRA2".REFERENCIAS.FINAL, in2 := "DB PRINCIPAL".REFERENCIAS.PASSO_ACC, out => "DB PUXADOR_SECADEIRA2".REFERENCIAS.FINAL)
   END_RUNG
   RUNG wire#w1
      { S7_Templates := "SrcType := Real" } GT_Contact(in1 := "DB PUXADOR_SECADEIRA2".REFERENCIAS.FINAL, in2 := "Tag_56")
      { S7_Templates := "SrcType := Real"; S7_GenerateENO := "TRUE" } Sub(in1 := "DB PUXADOR_SECADEIRA2".REFERENCIAS.FINAL, in2 := "DB PRINCIPAL".REFERENCIAS.PASSO_DEC, out => "DB PUXADOR_SECADEIRA2".REFERENCIAS.FINAL)
      { S7_Templates := "SrcType := Real" } LT_Contact(in1 := "DB PUXADOR_SECADEIRA2".REFERENCIAS.FINAL, in2 := 0.0)
      { S7_GenerateENO := "TRUE" } Move(in := 0.0, out1 => "DB PUXADOR_SECADEIRA2".REFERENCIAS.FINAL)
   END_RUNG
   RUNG wire#w1
      { S7_Templates := "SrcType := Real"; S7_GenerateENO := "TRUE" } Sub(in1 := "DB PUXADOR_SECADEIRA2".REFERENCIAS.FINAL, in2 := "Tag_56", out => "Tag_58")
      { S7_Templates := "SrcType := Real" } GT_Contact(in1 := "Tag_58", in2 := -1.0)
      { S7_Templates := "SrcType := Real" } LT_Contact(in1 := "Tag_58", in2 := 1.0)
      { S7_GenerateENO := "TRUE" } Move(in := "Tag_56", out1 => "DB PUXADOR_SECADEIRA2".REFERENCIAS.FINAL)
   END_RUNG
   RUNG wire#w1
      I_Contact( "DB PUXADOR_SECADEIRA2".COMANDOS.DESBLOQUEIO_DRIVER )
      { S7_Templates := "SrcType := Real" } GE_Contact(in1 := "DB PUXADOR_SECADEIRA2".REFERENCIAS.FINAL, in2 := "DB PRINCIPAL".REFERENCIAS.PASSO_DEC)
      { S7_GenerateENO := "TRUE" } Move(in := "DB PRINCIPAL".REFERENCIAS.PASSO_DEC, out1 => "DB PUXADOR_SECADEIRA2".REFERENCIAS.FINAL)
   END_RUNG
   // the same network as SCL:
   // ENO of a box is taken as its EN; it also drops when the box reports an error
   IF "DB PRINCIPAL".AUXILIARES.SEMPRE_1 AND ("Tag_56" > "DB PUXADOR_SECADEIRA2".REFERENCIAS.FINAL) THEN
       "DB PUXADOR_SECADEIRA2".REFERENCIAS.FINAL := "DB PUXADOR_SECADEIRA2".REFERENCIAS.FINAL + "DB PRINCIPAL".REFERENCIAS.PASSO_ACC;
   END_IF;
   #_w1 := "DB PRINCIPAL".AUXILIARES.SEMPRE_1 AND ("DB PUXADOR_SECADEIRA2".REFERENCIAS.FINAL > "Tag_56");
   IF #_w1 THEN
       "DB PUXADOR_SECADEIRA2".REFERENCIAS.FINAL := "DB PUXADOR_SECADEIRA2".REFERENCIAS.FINAL - "DB PRINCIPAL".REFERENCIAS.PASSO_DEC;
   END_IF;
   IF #_w1 AND ("DB PUXADOR_SECADEIRA2".REFERENCIAS.FINAL < 0.0) THEN
       "DB PUXADOR_SECADEIRA2".REFERENCIAS.FINAL := 0.0;
   END_IF;
   IF "DB PRINCIPAL".AUXILIARES.SEMPRE_1 THEN
       "Tag_58" := "DB PUXADOR_SECADEIRA2".REFERENCIAS.FINAL - "Tag_56";
   END_IF;
   IF "DB PRINCIPAL".AUXILIARES.SEMPRE_1 AND ("Tag_58" > (-1.0)) AND ("Tag_58" < 1.0) THEN
       "DB PUXADOR_SECADEIRA2".REFERENCIAS.FINAL := "Tag_56";
   END_IF;
   IF "DB PRINCIPAL".AUXILIARES.SEMPRE_1 AND NOT "DB PUXADOR_SECADEIRA2".COMANDOS.DESBLOQUEIO_DRIVER AND ("DB PUXADOR_SECADEIRA2".REFERENCIAS.FINAL >= "DB PRINCIPAL".REFERENCIAS.PASSO_DEC) THEN
       "DB PUXADOR_SECADEIRA2".REFERENCIAS.FINAL := "DB PRINCIPAL".REFERENCIAS.PASSO_DEC;
   END_IF;
END_REGION

REGION Network 11: DESBLOQUEIO DO INVERSOR DE FREQUÊNCIA
   // DESBLOQUEIO DO INVERSOR DE FREQUÊNCIA
   RUNG wire#powerrail
      Contact( "DB PRINCIPAL".AUXILIARES.SEMPRE_1 )
      wire#w1
      Contact( "DB PUXADOR_SECADEIRA2".COMANDOS.JOG )
      wire#w2
      { S7_Templates := "SrcType := Real" } GE_Contact(in1 := "DB PUXADOR_SECADEIRA2".REFERENCIAS.FINAL, in2 := "DB PRINCIPAL".REFERENCIAS.PASSO_DEC)
      Coil( "DB PUXADOR_SECADEIRA2".COMANDOS.DESBLOQUEIO_DRIVER )
   END_RUNG
   RUNG wire#w1
      Contact( "DB PUXADOR_SECADEIRA2".COMANDOS.MARCHA )
   END_RUNG wire#w2
   RUNG wire#w1
      Contact( "DB PUXADOR_SECADEIRA2".COMANDOS.DESBLOQUEIO_DRIVER )
   END_RUNG wire#w2
   // the same network as SCL:
   "DB PUXADOR_SECADEIRA2".COMANDOS.DESBLOQUEIO_DRIVER := "DB PRINCIPAL".AUXILIARES.SEMPRE_1 AND ("DB PUXADOR_SECADEIRA2".COMANDOS.JOG OR "DB PUXADOR_SECADEIRA2".COMANDOS.MARCHA OR "DB PUXADOR_SECADEIRA2".COMANDOS.DESBLOQUEIO_DRIVER) AND ("DB PUXADOR_SECADEIRA2".REFERENCIAS.FINAL >= "DB PRINCIPAL".REFERENCIAS.PASSO_DEC);
END_REGION

REGION Network 12 (STL): STATUS / CONTROLE - INVERSOR DE FREQUÊNCIA
   // DANFOSS FC300 PROFIBUS - TEX24626INV001
   // STATUS DO INVERSOR DE FREQUÊNCIA
   //     L     PIW 1220
         T     "Tag_1";
         AN    "Tag_59";
         =     "DB PUXADOR_SECADEIRA2".COMANDOS.STATUS_DRIVER;

   // CONTROLE DO INVERSOR DE FREQUÊNCIA
         L     1150;
         T     "Tag_1";
         A     "DB PUXADOR_SECADEIRA2".COMANDOS.DESBLOQUEIO_DRIVER;
         =     "Tag_60";
         A     "T2";
         AN    "DB PUXADOR_SECADEIRA2".COMANDOS.STATUS_DRIVER;
         =     "Tag_61";
         L     "Tag_1";
   //     T     PQW 1220

   // REFERÊNCIA PARA O INVERSOR DE FREQUÊNCIA
         L     "DB PUXADOR_SECADEIRA2".REFERENCIAS.FINAL;
         L     16384.0;
         *R;

         L     "DB PUXADOR_SECADEIRA2".REFERENCIAS.VELOCIDADE_MAXIMA;
         /R;
         RND;
         T     "Tag_62";
         L     "Tag_62";
   //     T     PQW 1222
END_REGION

REGION Network 13 (STL): INVERSOR RESERVA
         A     "DB PRINCIPAL".AUXILIARES.SEMPRE_1;
         =     %L24.0;
         A     %L24.0;
         A(;
         L     "DB PRINCIPAL".AUXILIARES1.INVERSOR_RESERVA1;
         L     12;
         ==I;
         );
         =     %L24.1;
         A     %L24.1;
         JNB   M00f;
         L     "DB PUXADOR_SECADEIRA2".REFERENCIAS.FINAL;
         L     3.456;
         *R;
         T     #AUX_R;
         RND;
         T     "P_QW100":P;
   M00f: NOP   0;
         A     %L24.1;
         A     "I130";
         S     "DB PRINCIPAL".ALARME.INV_RESERVA1;
         A     %L24.1;
         A     "DB PUXADOR_SECADEIRA2".COMANDOS.DESBLOQUEIO_DRIVER;
         S     "Q134";
         A     %L24.1;
         AN    "DB PUXADOR_SECADEIRA2".COMANDOS.DESBLOQUEIO_DRIVER;
         R     "Q134";
         A     %L24.0;
         A(;
         L     "DB PRINCIPAL".AUXILIARES1.INVERSOR_RESERVA2;
         L     12;
         ==I;
         );
         =     %L24.1;
         A     %L24.1;
         JNB   M010;
         L     "DB PUXADOR_SECADEIRA2".REFERENCIAS.FINAL;
         L     3.456;
         *R;
         T     #AUX_R;
         RND;
         T     "P_QW102":P;
   M010: NOP   0;
         A     %L24.1;
         A     "I132";
         S     "DB PRINCIPAL".ALARME.INV_RESERVA2;
         A     %L24.1;
         A     "DB PUXADOR_SECADEIRA2".COMANDOS.DESBLOQUEIO_DRIVER;
         S     "Q135";
         A     %L24.1;
         AN    "DB PUXADOR_SECADEIRA2".COMANDOS.DESBLOQUEIO_DRIVER;
         R     "Q135";
END_REGION
END_FUNCTION

FUNCTION "MT_SECADEIRA2" : Void   // FC22, LAD
TITLE = MÓDULO DE CONTROLE DA SECADEIRA 2
{ S7_Optimized_Access := 'FALSE' }
AUTHOR : THALLES
FAMILY : TRAÇÃO
NAME : LINHA1
VERSION : 0.1
// DATA BLOCK DE CONTROLE // DB22
// Automation Pack Automação Indl. e Com. Ltda.
// Cliente: Texima S/A Ind. de Máquinas
// Cliente Final: Cia. Fiação e Tecidos Santo Antonio.
// Máquina: LINHA 1 DENIN - O.S.: 24.626
   VAR_TEMP
      AUX_R : Real;
   END_VAR
   VAR_TEMP   // added for the SCL form of the ladder/FBD networks
      _w1 : Bool;
   END_VAR
BEGIN

REGION Network 1: ALARMES
   // RESET DOS ALARMES
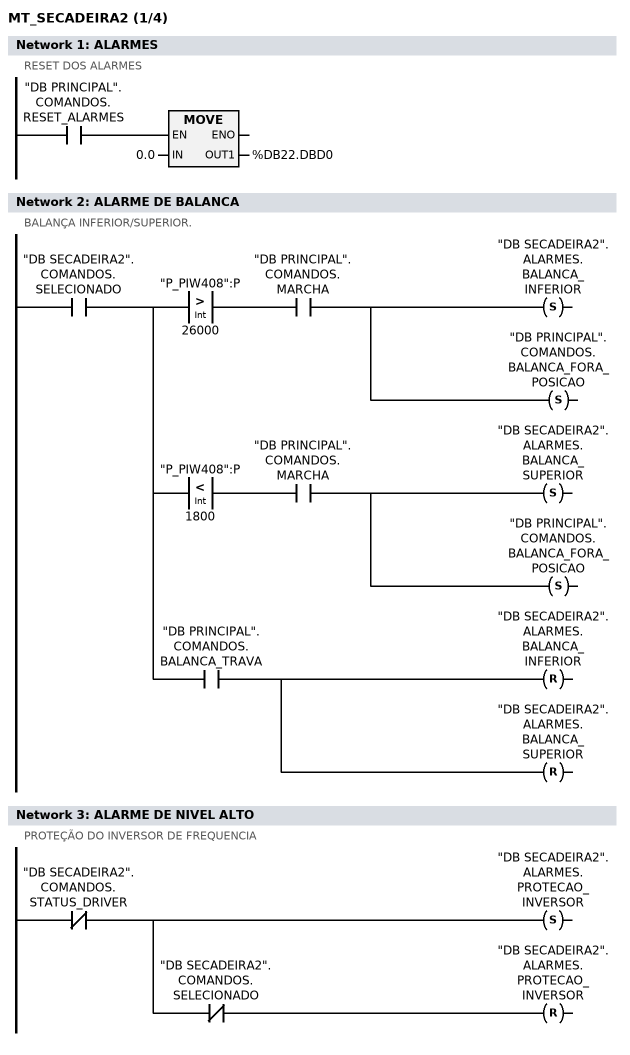
   RUNG wire#powerrail
      Contact( "DB PRINCIPAL".COMANDOS.RESET_ALARMES )
      { S7_GenerateENO := "TRUE" } Move(in := 0.0, out1 => %DB22.DBD0)
   END_RUNG
   // the same network as SCL:
   IF "DB PRINCIPAL".COMANDOS.RESET_ALARMES THEN %DB22.DBD0 := 0.0; END_IF;
END_REGION

REGION Network 2: ALARME DE BALANCA
   // BALANÇA INFERIOR/SUPERIOR.
   RUNG wire#powerrail
      Contact( "DB SECADEIRA2".COMANDOS.SELECIONADO )
      wire#w1
      { S7_Templates := "SrcType := Int" } GT_Contact(in1 := "P_PIW408":P, in2 := 26000)
      Contact( "DB PRINCIPAL".COMANDOS.MARCHA )
      wire#w2
      S_Coil( "DB SECADEIRA2".ALARMES.BALANCA_INFERIOR )
   END_RUNG
   RUNG wire#w2
      S_Coil( "DB PRINCIPAL".COMANDOS.BALANCA_FORA_POSICAO )
   END_RUNG
   RUNG wire#w1
      { S7_Templates := "SrcType := Int" } LT_Contact(in1 := "P_PIW408":P, in2 := 1800)
      Contact( "DB PRINCIPAL".COMANDOS.MARCHA )
      wire#w3
      S_Coil( "DB SECADEIRA2".ALARMES.BALANCA_SUPERIOR )
   END_RUNG
   RUNG wire#w3
      S_Coil( "DB PRINCIPAL".COMANDOS.BALANCA_FORA_POSICAO )
   END_RUNG
   RUNG wire#w1
      Contact( "DB PRINCIPAL".COMANDOS.BALANCA_TRAVA )
      wire#w4
      R_Coil( "DB SECADEIRA2".ALARMES.BALANCA_INFERIOR )
   END_RUNG
   RUNG wire#w4
      R_Coil( "DB SECADEIRA2".ALARMES.BALANCA_SUPERIOR )
   END_RUNG
   // the same network as SCL:
   IF "DB SECADEIRA2".COMANDOS.SELECIONADO AND ("P_PIW408":P > 26000) AND "DB PRINCIPAL".COMANDOS.MARCHA THEN
       "DB SECADEIRA2".ALARMES.BALANCA_INFERIOR := TRUE;
       "DB PRINCIPAL".COMANDOS.BALANCA_FORA_POSICAO := TRUE;
   END_IF;
   IF "DB SECADEIRA2".COMANDOS.SELECIONADO AND ("P_PIW408":P < 1800) AND "DB PRINCIPAL".COMANDOS.MARCHA THEN
       "DB SECADEIRA2".ALARMES.BALANCA_SUPERIOR := TRUE;
       "DB PRINCIPAL".COMANDOS.BALANCA_FORA_POSICAO := TRUE;
   END_IF;
   IF "DB SECADEIRA2".COMANDOS.SELECIONADO AND "DB PRINCIPAL".COMANDOS.BALANCA_TRAVA THEN
       "DB SECADEIRA2".ALARMES.BALANCA_INFERIOR := FALSE;
       "DB SECADEIRA2".ALARMES.BALANCA_SUPERIOR := FALSE;
   END_IF;
END_REGION

REGION Network 3: ALARME DE NIVEL ALTO
   // PROTEÇÃO DO INVERSOR DE FREQUENCIA
   RUNG wire#powerrail
      I_Contact( "DB SECADEIRA2".COMANDOS.STATUS_DRIVER )
      wire#w1
      S_Coil( "DB SECADEIRA2".ALARMES.PROTECAO_INVERSOR )
   END_RUNG
   RUNG wire#w1
      I_Contact( "DB SECADEIRA2".COMANDOS.SELECIONADO )
      R_Coil( "DB SECADEIRA2".ALARMES.PROTECAO_INVERSOR )
   END_RUNG
   // the same network as SCL:
   #_w1 := NOT "DB SECADEIRA2".COMANDOS.STATUS_DRIVER;
   IF #_w1 THEN "DB SECADEIRA2".ALARMES.PROTECAO_INVERSOR := TRUE; END_IF;
   IF #_w1 AND NOT "DB SECADEIRA2".COMANDOS.SELECIONADO THEN
       "DB SECADEIRA2".ALARMES.PROTECAO_INVERSOR := FALSE;
   END_IF;
END_REGION

REGION Network 4: ALARMES
   // ATIVAÇÃO DO BIT DE ALARME DE NIVEL ALTO
   // ATIVAÇÃO DO BIT DE ALARME DE NIVEL BAIXO
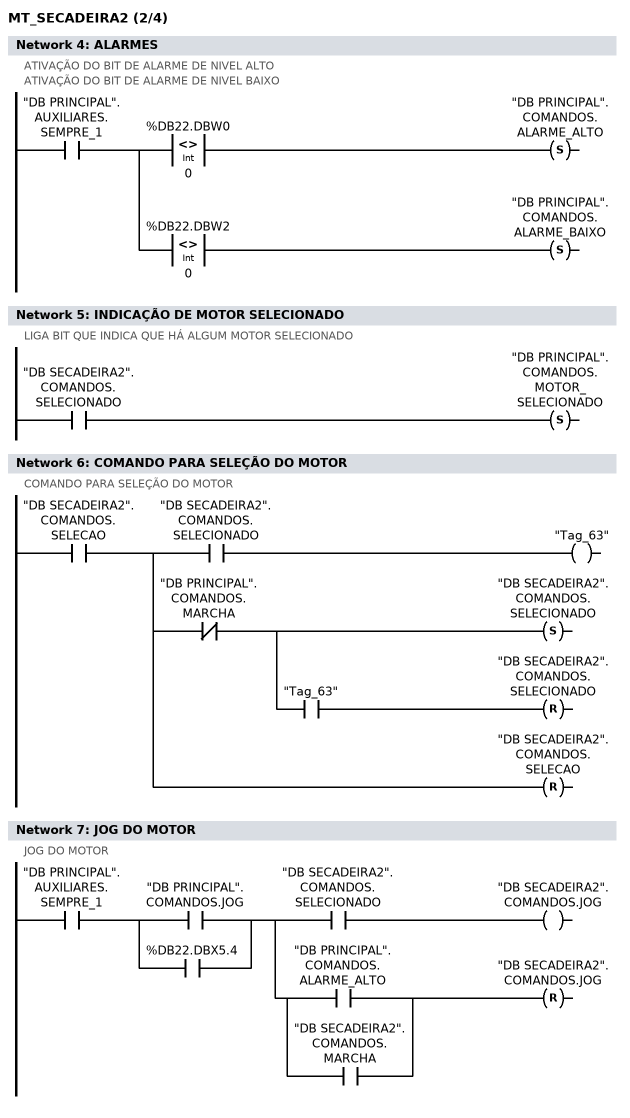
   RUNG wire#powerrail
      Contact( "DB PRINCIPAL".AUXILIARES.SEMPRE_1 )
      wire#w1
      { S7_Templates := "SrcType := Int" } NE_Contact(in1 := %DB22.DBW0, in2 := 0)
      S_Coil( "DB PRINCIPAL".COMANDOS.ALARME_ALTO )
   END_RUNG
   RUNG wire#w1
      { S7_Templates := "SrcType := Int" } NE_Contact(in1 := %DB22.DBW2, in2 := 0)
      S_Coil( "DB PRINCIPAL".COMANDOS.ALARME_BAIXO )
   END_RUNG
   // the same network as SCL:
   IF "DB PRINCIPAL".AUXILIARES.SEMPRE_1 AND (%DB22.DBW0 <> 0) THEN
       "DB PRINCIPAL".COMANDOS.ALARME_ALTO := TRUE;
   END_IF;
   IF "DB PRINCIPAL".AUXILIARES.SEMPRE_1 AND (%DB22.DBW2 <> 0) THEN
       "DB PRINCIPAL".COMANDOS.ALARME_BAIXO := TRUE;
   END_IF;
END_REGION

REGION Network 5: INDICAÇÃO DE MOTOR SELECIONADO
   // LIGA BIT QUE INDICA QUE HÁ ALGUM MOTOR SELECIONADO
   RUNG wire#powerrail
      Contact( "DB SECADEIRA2".COMANDOS.SELECIONADO )
      S_Coil( "DB PRINCIPAL".COMANDOS.MOTOR_SELECIONADO )
   END_RUNG
   // the same network as SCL:
   IF "DB SECADEIRA2".COMANDOS.SELECIONADO THEN "DB PRINCIPAL".COMANDOS.MOTOR_SELECIONADO := TRUE; END_IF;
END_REGION

REGION Network 6: COMANDO PARA SELEÇÃO DO MOTOR
   // COMANDO PARA SELEÇÃO DO MOTOR
   RUNG wire#powerrail
      Contact( "DB SECADEIRA2".COMANDOS.SELECAO )
      wire#w1
      Contact( "DB SECADEIRA2".COMANDOS.SELECIONADO )
      Coil( "Tag_63" )
   END_RUNG
   RUNG wire#w1
      I_Contact( "DB PRINCIPAL".COMANDOS.MARCHA )
      wire#w2
      S_Coil( "DB SECADEIRA2".COMANDOS.SELECIONADO )
   END_RUNG
   RUNG wire#w2
      Contact( "Tag_63" )
      R_Coil( "DB SECADEIRA2".COMANDOS.SELECIONADO )
   END_RUNG
   RUNG wire#w1
      R_Coil( "DB SECADEIRA2".COMANDOS.SELECAO )
   END_RUNG
   // the same network as SCL:
   "Tag_63" := "DB SECADEIRA2".COMANDOS.SELECAO AND "DB SECADEIRA2".COMANDOS.SELECIONADO;
   #_w1 := "DB SECADEIRA2".COMANDOS.SELECAO AND NOT "DB PRINCIPAL".COMANDOS.MARCHA;
   IF #_w1 THEN "DB SECADEIRA2".COMANDOS.SELECIONADO := TRUE; END_IF;
   IF #_w1 AND "Tag_63" THEN "DB SECADEIRA2".COMANDOS.SELECIONADO := FALSE; END_IF;
   IF "DB SECADEIRA2".COMANDOS.SELECAO THEN "DB SECADEIRA2".COMANDOS.SELECAO := FALSE; END_IF;
END_REGION

REGION Network 7: JOG DO MOTOR
   // JOG DO MOTOR
   RUNG wire#powerrail
      Contact( "DB PRINCIPAL".AUXILIARES.SEMPRE_1 )
      wire#w1
      Contact( "DB PRINCIPAL".COMANDOS.JOG )
      wire#w2
      Contact( "DB SECADEIRA2".COMANDOS.SELECIONADO )
      Coil( "DB SECADEIRA2".COMANDOS.JOG )
   END_RUNG
   RUNG wire#w1
      Contact( %DB22.DBX5.4 )
   END_RUNG wire#w2
   RUNG wire#w2
      Contact( "DB PRINCIPAL".COMANDOS.ALARME_ALTO )
      wire#w3
      R_Coil( "DB SECADEIRA2".COMANDOS.JOG )
   END_RUNG
   RUNG wire#w2
      Contact( "DB SECADEIRA2".COMANDOS.MARCHA )
   END_RUNG wire#w3
   // the same network as SCL:
   #_w1 := "DB PRINCIPAL".AUXILIARES.SEMPRE_1 AND ("DB PRINCIPAL".COMANDOS.JOG OR %DB22.DBX5.4);
   "DB SECADEIRA2".COMANDOS.JOG := #_w1 AND "DB SECADEIRA2".COMANDOS.SELECIONADO;
   IF #_w1 AND ("DB PRINCIPAL".COMANDOS.ALARME_ALTO OR "DB SECADEIRA2".COMANDOS.MARCHA) THEN
       "DB SECADEIRA2".COMANDOS.JOG := FALSE;
   END_IF;
END_REGION

REGION Network 8: COMANDO PARA LIBERAÇÃO DO MOTOR
   // COMANDO PARA LIBERAÇÃO DO MOTOR
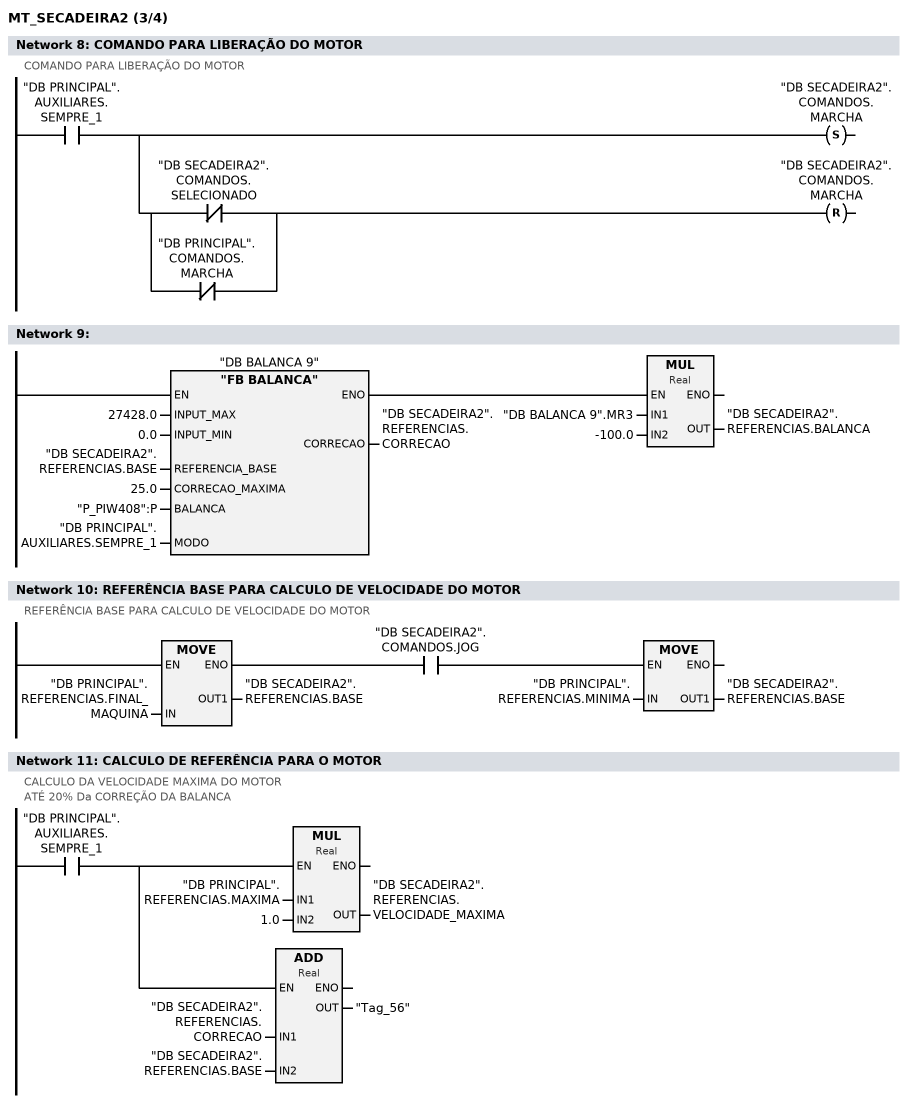
   RUNG wire#powerrail
      Contact( "DB PRINCIPAL".AUXILIARES.SEMPRE_1 )
      wire#w1
      S_Coil( "DB SECADEIRA2".COMANDOS.MARCHA )
   END_RUNG
   RUNG wire#w1
      I_Contact( "DB SECADEIRA2".COMANDOS.SELECIONADO )
      wire#w2
      R_Coil( "DB SECADEIRA2".COMANDOS.MARCHA )
   END_RUNG
   RUNG wire#w1
      I_Contact( "DB PRINCIPAL".COMANDOS.MARCHA )
   END_RUNG wire#w2
   // the same network as SCL:
   IF "DB PRINCIPAL".AUXILIARES.SEMPRE_1 THEN "DB SECADEIRA2".COMANDOS.MARCHA := TRUE; END_IF;
   IF "DB PRINCIPAL".AUXILIARES.SEMPRE_1 AND (NOT "DB SECADEIRA2".COMANDOS.SELECIONADO OR NOT "DB PRINCIPAL".COMANDOS.MARCHA) THEN
       "DB SECADEIRA2".COMANDOS.MARCHA := FALSE;
   END_IF;
END_REGION

REGION Network 9
   RUNG wire#powerrail
      "DB BALANCA 9"(INPUT_MAX := 27428.0, INPUT_MIN := 0.0, REFERENCIA_BASE := "DB SECADEIRA2".REFERENCIAS.BASE, CORRECAO_MAXIMA := 25.0, BALANCA := "P_PIW408":P, MODO := "DB PRINCIPAL".AUXILIARES.SEMPRE_1, CORRECAO => "DB SECADEIRA2".REFERENCIAS.CORRECAO)
      { S7_Templates := "SrcType := Real"; S7_GenerateENO := "TRUE" } Mul(in1 := "DB BALANCA 9".MR3, in2 := -100.0, out => "DB SECADEIRA2".REFERENCIAS.BALANCA)
   END_RUNG
   // the same network as SCL:
   "DB BALANCA 9"(INPUT_MAX := 27428.0,   // "FB BALANCA"
                  INPUT_MIN := 0.0,
                  REFERENCIA_BASE := "DB SECADEIRA2".REFERENCIAS.BASE,
                  CORRECAO_MAXIMA := 25.0,
                  BALANCA := "P_PIW408":P,
                  MODO := "DB PRINCIPAL".AUXILIARES.SEMPRE_1,
                  CORRECAO => "DB SECADEIRA2".REFERENCIAS.CORRECAO,
                  ENO => #_w1);
   IF #_w1 THEN "DB SECADEIRA2".REFERENCIAS.BALANCA := "DB BALANCA 9".MR3 * (-100.0); END_IF;
END_REGION

REGION Network 10: REFERÊNCIA BASE PARA CALCULO DE VELOCIDADE DO MOTOR
   // REFERÊNCIA BASE PARA CALCULO DE VELOCIDADE DO MOTOR
   RUNG wire#powerrail
      { S7_GenerateENO := "TRUE" } Move(in := "DB PRINCIPAL".REFERENCIAS.FINAL_MAQUINA, out1 => "DB SECADEIRA2".REFERENCIAS.BASE)
      Contact( "DB SECADEIRA2".COMANDOS.JOG )
      { S7_GenerateENO := "TRUE" } Move(in := "DB PRINCIPAL".REFERENCIAS.MINIMA, out1 => "DB SECADEIRA2".REFERENCIAS.BASE)
   END_RUNG
   // the same network as SCL:
   // ENO of a box is taken as its EN; it also drops when the box reports an error
   "DB SECADEIRA2".REFERENCIAS.BASE := "DB PRINCIPAL".REFERENCIAS.FINAL_MAQUINA;
   IF "DB SECADEIRA2".COMANDOS.JOG THEN
       "DB SECADEIRA2".REFERENCIAS.BASE := "DB PRINCIPAL".REFERENCIAS.MINIMA;
   END_IF;
END_REGION

REGION Network 11: CALCULO DE REFERÊNCIA PARA O MOTOR
   // CALCULO DA VELOCIDADE MAXIMA DO MOTOR
   // ATÉ 20% Da CORREÇÃO DA BALANCA
   RUNG wire#powerrail
      Contact( "DB PRINCIPAL".AUXILIARES.SEMPRE_1 )
      wire#w1
      { S7_Templates := "SrcType := Real"; S7_GenerateENO := "TRUE" } Mul(in1 := "DB PRINCIPAL".REFERENCIAS.MAXIMA, in2 := 1.0, out => "DB SECADEIRA2".REFERENCIAS.VELOCIDADE_MAXIMA)
   END_RUNG
   RUNG wire#w1
      { S7_Templates := "SrcType := Real"; S7_GenerateENO := "TRUE" } Add(in1 := "DB SECADEIRA2".REFERENCIAS.CORRECAO, in2 := "DB SECADEIRA2".REFERENCIAS.BASE, out => "Tag_56")
   END_RUNG
   // the same network as SCL:
   IF "DB PRINCIPAL".AUXILIARES.SEMPRE_1 THEN
       "DB SECADEIRA2".REFERENCIAS.VELOCIDADE_MAXIMA := "DB PRINCIPAL".REFERENCIAS.MAXIMA * 1.0;
       "Tag_56" := "DB SECADEIRA2".REFERENCIAS.CORRECAO + "DB SECADEIRA2".REFERENCIAS.BASE;
   END_IF;
END_REGION

REGION Network 12: ACC/DEC DA REFERÊNCIA DO MOTOR
   // ACC/DEC DA REFERÊNCIA DO MOTOR
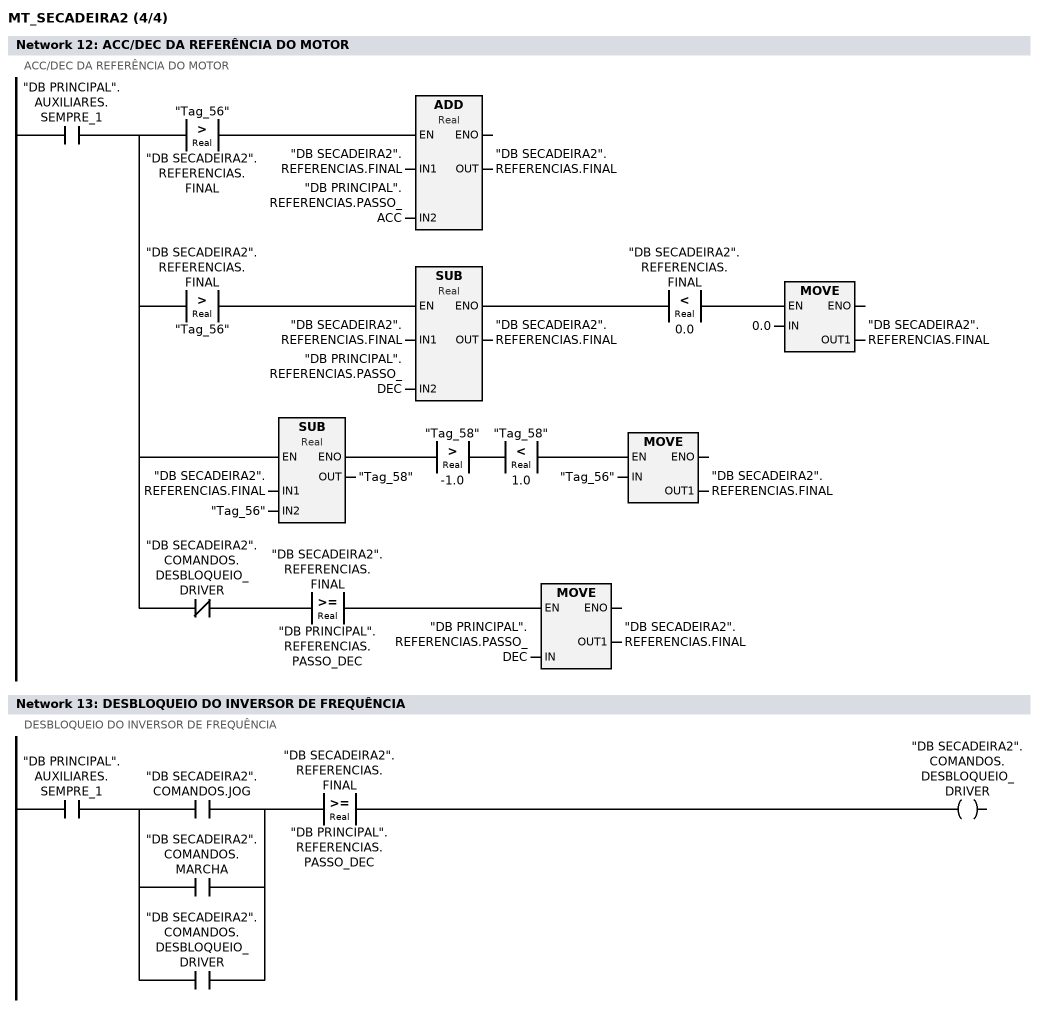
   RUNG wire#powerrail
      Contact( "DB PRINCIPAL".AUXILIARES.SEMPRE_1 )
      wire#w1
      { S7_Templates := "SrcType := Real" } GT_Contact(in1 := "Tag_56", in2 := "DB SECADEIRA2".REFERENCIAS.FINAL)
      { S7_Templates := "SrcType := Real"; S7_GenerateENO := "TRUE" } Add(in1 := "DB SECADEIRA2".REFERENCIAS.FINAL, in2 := "DB PRINCIPAL".REFERENCIAS.PASSO_ACC, out => "DB SECADEIRA2".REFERENCIAS.FINAL)
   END_RUNG
   RUNG wire#w1
      { S7_Templates := "SrcType := Real" } GT_Contact(in1 := "DB SECADEIRA2".REFERENCIAS.FINAL, in2 := "Tag_56")
      { S7_Templates := "SrcType := Real"; S7_GenerateENO := "TRUE" } Sub(in1 := "DB SECADEIRA2".REFERENCIAS.FINAL, in2 := "DB PRINCIPAL".REFERENCIAS.PASSO_DEC, out => "DB SECADEIRA2".REFERENCIAS.FINAL)
      { S7_Templates := "SrcType := Real" } LT_Contact(in1 := "DB SECADEIRA2".REFERENCIAS.FINAL, in2 := 0.0)
      { S7_GenerateENO := "TRUE" } Move(in := 0.0, out1 => "DB SECADEIRA2".REFERENCIAS.FINAL)
   END_RUNG
   RUNG wire#w1
      { S7_Templates := "SrcType := Real"; S7_GenerateENO := "TRUE" } Sub(in1 := "DB SECADEIRA2".REFERENCIAS.FINAL, in2 := "Tag_56", out => "Tag_58")
      { S7_Templates := "SrcType := Real" } GT_Contact(in1 := "Tag_58", in2 := -1.0)
      { S7_Templates := "SrcType := Real" } LT_Contact(in1 := "Tag_58", in2 := 1.0)
      { S7_GenerateENO := "TRUE" } Move(in := "Tag_56", out1 => "DB SECADEIRA2".REFERENCIAS.FINAL)
   END_RUNG
   RUNG wire#w1
      I_Contact( "DB SECADEIRA2".COMANDOS.DESBLOQUEIO_DRIVER )
      { S7_Templates := "SrcType := Real" } GE_Contact(in1 := "DB SECADEIRA2".REFERENCIAS.FINAL, in2 := "DB PRINCIPAL".REFERENCIAS.PASSO_DEC)
      { S7_GenerateENO := "TRUE" } Move(in := "DB PRINCIPAL".REFERENCIAS.PASSO_DEC, out1 => "DB SECADEIRA2".REFERENCIAS.FINAL)
   END_RUNG
   // the same network as SCL:
   // ENO of a box is taken as its EN; it also drops when the box reports an error
   IF "DB PRINCIPAL".AUXILIARES.SEMPRE_1 AND ("Tag_56" > "DB SECADEIRA2".REFERENCIAS.FINAL) THEN
       "DB SECADEIRA2".REFERENCIAS.FINAL := "DB SECADEIRA2".REFERENCIAS.FINAL + "DB PRINCIPAL".REFERENCIAS.PASSO_ACC;
   END_IF;
   #_w1 := "DB PRINCIPAL".AUXILIARES.SEMPRE_1 AND ("DB SECADEIRA2".REFERENCIAS.FINAL > "Tag_56");
   IF #_w1 THEN
       "DB SECADEIRA2".REFERENCIAS.FINAL := "DB SECADEIRA2".REFERENCIAS.FINAL - "DB PRINCIPAL".REFERENCIAS.PASSO_DEC;
   END_IF;
   IF #_w1 AND ("DB SECADEIRA2".REFERENCIAS.FINAL < 0.0) THEN
       "DB SECADEIRA2".REFERENCIAS.FINAL := 0.0;
   END_IF;
   IF "DB PRINCIPAL".AUXILIARES.SEMPRE_1 THEN
       "Tag_58" := "DB SECADEIRA2".REFERENCIAS.FINAL - "Tag_56";
   END_IF;
   IF "DB PRINCIPAL".AUXILIARES.SEMPRE_1 AND ("Tag_58" > (-1.0)) AND ("Tag_58" < 1.0) THEN
       "DB SECADEIRA2".REFERENCIAS.FINAL := "Tag_56";
   END_IF;
   IF "DB PRINCIPAL".AUXILIARES.SEMPRE_1 AND NOT "DB SECADEIRA2".COMANDOS.DESBLOQUEIO_DRIVER AND ("DB SECADEIRA2".REFERENCIAS.FINAL >= "DB PRINCIPAL".REFERENCIAS.PASSO_DEC) THEN
       "DB SECADEIRA2".REFERENCIAS.FINAL := "DB PRINCIPAL".REFERENCIAS.PASSO_DEC;
   END_IF;
END_REGION

REGION Network 13: DESBLOQUEIO DO INVERSOR DE FREQUÊNCIA
   // DESBLOQUEIO DO INVERSOR DE FREQUÊNCIA
   RUNG wire#powerrail
      Contact( "DB PRINCIPAL".AUXILIARES.SEMPRE_1 )
      wire#w1
      Contact( "DB SECADEIRA2".COMANDOS.JOG )
      wire#w2
      { S7_Templates := "SrcType := Real" } GE_Contact(in1 := "DB SECADEIRA2".REFERENCIAS.FINAL, in2 := "DB PRINCIPAL".REFERENCIAS.PASSO_DEC)
      Coil( "DB SECADEIRA2".COMANDOS.DESBLOQUEIO_DRIVER )
   END_RUNG
   RUNG wire#w1
      Contact( "DB SECADEIRA2".COMANDOS.MARCHA )
   END_RUNG wire#w2
   RUNG wire#w1
      Contact( "DB SECADEIRA2".COMANDOS.DESBLOQUEIO_DRIVER )
   END_RUNG wire#w2
   // the same network as SCL:
   "DB SECADEIRA2".COMANDOS.DESBLOQUEIO_DRIVER := "DB PRINCIPAL".AUXILIARES.SEMPRE_1 AND ("DB SECADEIRA2".COMANDOS.JOG OR "DB SECADEIRA2".COMANDOS.MARCHA OR "DB SECADEIRA2".COMANDOS.DESBLOQUEIO_DRIVER) AND ("DB SECADEIRA2".REFERENCIAS.FINAL >= "DB PRINCIPAL".REFERENCIAS.PASSO_DEC);
END_REGION

REGION Network 14 (STL): STATUS / CONTROLE - INVERSOR DE FREQUÊNCIA
   // DANFOSS FC300 PROFIBUS - TEX24626INV001
   // STATUS DO INVERSOR DE FREQUÊNCIA
         L     "Tag_36":P;
         T     "Tag_1";
         AN    "Tag_59";
         =     "DB SECADEIRA2".COMANDOS.STATUS_DRIVER;

   // CONTROLE DO INVERSOR DE FREQUÊNCIA
         L     1150;
         T     "Tag_1";
         A     "DB SECADEIRA2".COMANDOS.DESBLOQUEIO_DRIVER;
         =     "Tag_60";
         A     "T2";
         AN    "DB SECADEIRA2".COMANDOS.STATUS_DRIVER;
         =     "Tag_61";
         L     "Tag_1";
         T     "Tag_37":P;

   // REFERÊNCIA PARA O INVERSOR DE FREQUÊNCIA
         L     "DB SECADEIRA2".REFERENCIAS.FINAL;
         L     16384.0;
         *R;

         L     "DB SECADEIRA2".REFERENCIAS.VELOCIDADE_MAXIMA;
         /R;
         RND;
         T     "Tag_62";
         L     "Tag_62";
         T     "Tag_38":P;
END_REGION

REGION Network 15 (STL): INVERSOR RESERVA
         A     "DB PRINCIPAL".AUXILIARES.SEMPRE_1;
         =     %L24.0;
         A     %L24.0;
         A(;
         L     "DB PRINCIPAL".AUXILIARES1.INVERSOR_RESERVA1;
         L     13;
         ==I;
         );
         =     %L24.1;
         A     %L24.1;
         JNB   M001;
         L     "DB SECADEIRA2".REFERENCIAS.FINAL;
         L     3.456;
         *R;
         T     #AUX_R;
         RND;
         T     "P_QW100":P;
   M001: NOP   0;
         A     %L24.1;
         A     "I130";
         S     "DB PRINCIPAL".ALARME.INV_RESERVA1;
         A     %L24.1;
         A     "DB SECADEIRA2".COMANDOS.DESBLOQUEIO_DRIVER;
         S     "Q134";
         A     %L24.1;
         AN    "DB SECADEIRA2".COMANDOS.DESBLOQUEIO_DRIVER;
         R     "Q134";
         A     %L24.0;
         A(;
         L     "DB PRINCIPAL".AUXILIARES1.INVERSOR_RESERVA2;
         L     13;
         ==I;
         );
         =     %L24.1;
         A     %L24.1;
         JNB   M002;
         L     "DB SECADEIRA2".REFERENCIAS.FINAL;
         L     3.456;
         *R;
         T     #AUX_R;
         RND;
         T     "P_QW102":P;
   M002: NOP   0;
         A     %L24.1;
         A     "I132";
         S     "DB PRINCIPAL".ALARME.INV_RESERVA2;
         A     %L24.1;
         A     "DB SECADEIRA2".COMANDOS.DESBLOQUEIO_DRIVER;
         S     "Q135";
         A     %L24.1;
         AN    "DB SECADEIRA2".COMANDOS.DESBLOQUEIO_DRIVER;
         R     "Q135";
END_REGION
END_FUNCTION

FUNCTION "MT_SECADEIRA3" : Void   // FC23, LAD
TITLE = MÓDULO DE CONTROLE DA SECADEIRA 3
{ S7_Optimized_Access := 'FALSE' }
AUTHOR : THALLES
FAMILY : TRAÇÃO
NAME : LINHA1
VERSION : 0.1
// DATA BLOCK DE CONTROLE // DB23
// Automation Pack Automação Indl. e Com. Ltda.
// Cliente: Texima S/A Ind. de Máquinas
// Cliente Final: Cia. Fiação e Tecidos Santo Antonio.
// Máquina: LINHA 1 DENIN - O.S.: 24.626
   VAR_TEMP
      AUX_R : Real;
   END_VAR
   VAR_TEMP   // added for the SCL form of the ladder/FBD networks
      _w1 : Bool;
   END_VAR
BEGIN

REGION Network 1: ALARMES
   // RESET DOS ALARMES
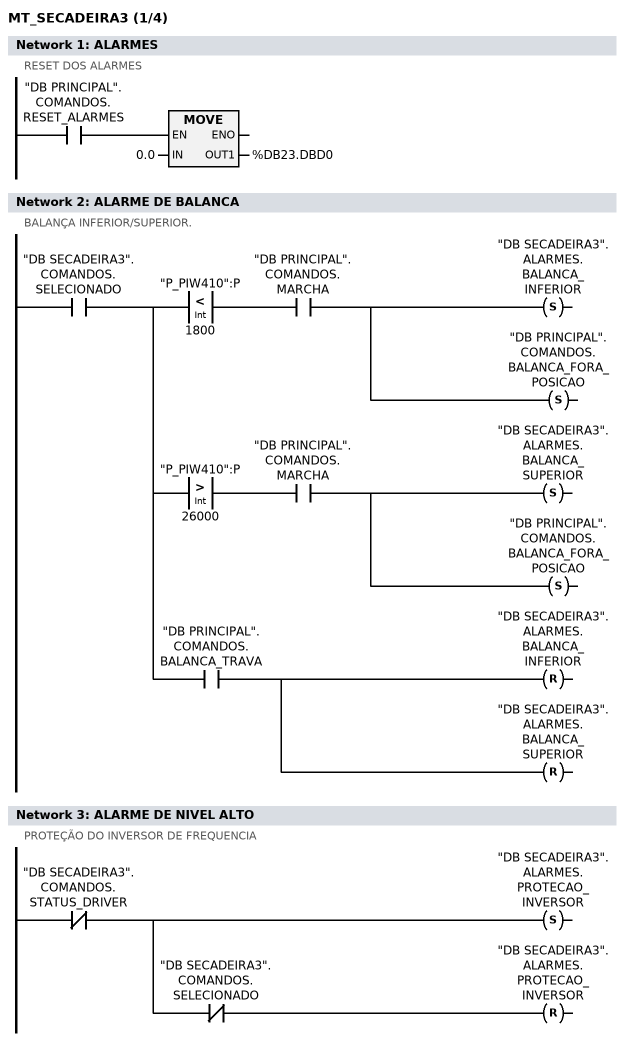
   RUNG wire#powerrail
      Contact( "DB PRINCIPAL".COMANDOS.RESET_ALARMES )
      { S7_GenerateENO := "TRUE" } Move(in := 0.0, out1 => %DB23.DBD0)
   END_RUNG
   // the same network as SCL:
   IF "DB PRINCIPAL".COMANDOS.RESET_ALARMES THEN %DB23.DBD0 := 0.0; END_IF;
END_REGION

REGION Network 2: ALARME DE BALANCA
   // BALANÇA INFERIOR/SUPERIOR.
   RUNG wire#powerrail
      Contact( "DB SECADEIRA3".COMANDOS.SELECIONADO )
      wire#w1
      { S7_Templates := "SrcType := Int" } LT_Contact(in1 := "P_PIW410":P, in2 := 1800)
      Contact( "DB PRINCIPAL".COMANDOS.MARCHA )
      wire#w2
      S_Coil( "DB SECADEIRA3".ALARMES.BALANCA_INFERIOR )
   END_RUNG
   RUNG wire#w2
      S_Coil( "DB PRINCIPAL".COMANDOS.BALANCA_FORA_POSICAO )
   END_RUNG
   RUNG wire#w1
      { S7_Templates := "SrcType := Int" } GT_Contact(in1 := "P_PIW410":P, in2 := 26000)
      Contact( "DB PRINCIPAL".COMANDOS.MARCHA )
      wire#w3
      S_Coil( "DB SECADEIRA3".ALARMES.BALANCA_SUPERIOR )
   END_RUNG
   RUNG wire#w3
      S_Coil( "DB PRINCIPAL".COMANDOS.BALANCA_FORA_POSICAO )
   END_RUNG
   RUNG wire#w1
      Contact( "DB PRINCIPAL".COMANDOS.BALANCA_TRAVA )
      wire#w4
      R_Coil( "DB SECADEIRA3".ALARMES.BALANCA_INFERIOR )
   END_RUNG
   RUNG wire#w4
      R_Coil( "DB SECADEIRA3".ALARMES.BALANCA_SUPERIOR )
   END_RUNG
   // the same network as SCL:
   IF "DB SECADEIRA3".COMANDOS.SELECIONADO AND ("P_PIW410":P < 1800) AND "DB PRINCIPAL".COMANDOS.MARCHA THEN
       "DB SECADEIRA3".ALARMES.BALANCA_INFERIOR := TRUE;
       "DB PRINCIPAL".COMANDOS.BALANCA_FORA_POSICAO := TRUE;
   END_IF;
   IF "DB SECADEIRA3".COMANDOS.SELECIONADO AND ("P_PIW410":P > 26000) AND "DB PRINCIPAL".COMANDOS.MARCHA THEN
       "DB SECADEIRA3".ALARMES.BALANCA_SUPERIOR := TRUE;
       "DB PRINCIPAL".COMANDOS.BALANCA_FORA_POSICAO := TRUE;
   END_IF;
   IF "DB SECADEIRA3".COMANDOS.SELECIONADO AND "DB PRINCIPAL".COMANDOS.BALANCA_TRAVA THEN
       "DB SECADEIRA3".ALARMES.BALANCA_INFERIOR := FALSE;
       "DB SECADEIRA3".ALARMES.BALANCA_SUPERIOR := FALSE;
   END_IF;
END_REGION

REGION Network 3: ALARME DE NIVEL ALTO
   // PROTEÇÃO DO INVERSOR DE FREQUENCIA
   RUNG wire#powerrail
      I_Contact( "DB SECADEIRA3".COMANDOS.STATUS_DRIVER )
      wire#w1
      S_Coil( "DB SECADEIRA3".ALARMES.PROTECAO_INVERSOR )
   END_RUNG
   RUNG wire#w1
      I_Contact( "DB SECADEIRA3".COMANDOS.SELECIONADO )
      R_Coil( "DB SECADEIRA3".ALARMES.PROTECAO_INVERSOR )
   END_RUNG
   // the same network as SCL:
   #_w1 := NOT "DB SECADEIRA3".COMANDOS.STATUS_DRIVER;
   IF #_w1 THEN "DB SECADEIRA3".ALARMES.PROTECAO_INVERSOR := TRUE; END_IF;
   IF #_w1 AND NOT "DB SECADEIRA3".COMANDOS.SELECIONADO THEN
       "DB SECADEIRA3".ALARMES.PROTECAO_INVERSOR := FALSE;
   END_IF;
END_REGION

REGION Network 4: ALARMES
   // ATIVAÇÃO DO BIT DE ALARME DE NIVEL ALTO
   // ATIVAÇÃO DO BIT DE ALARME DE NIVEL BAIXO
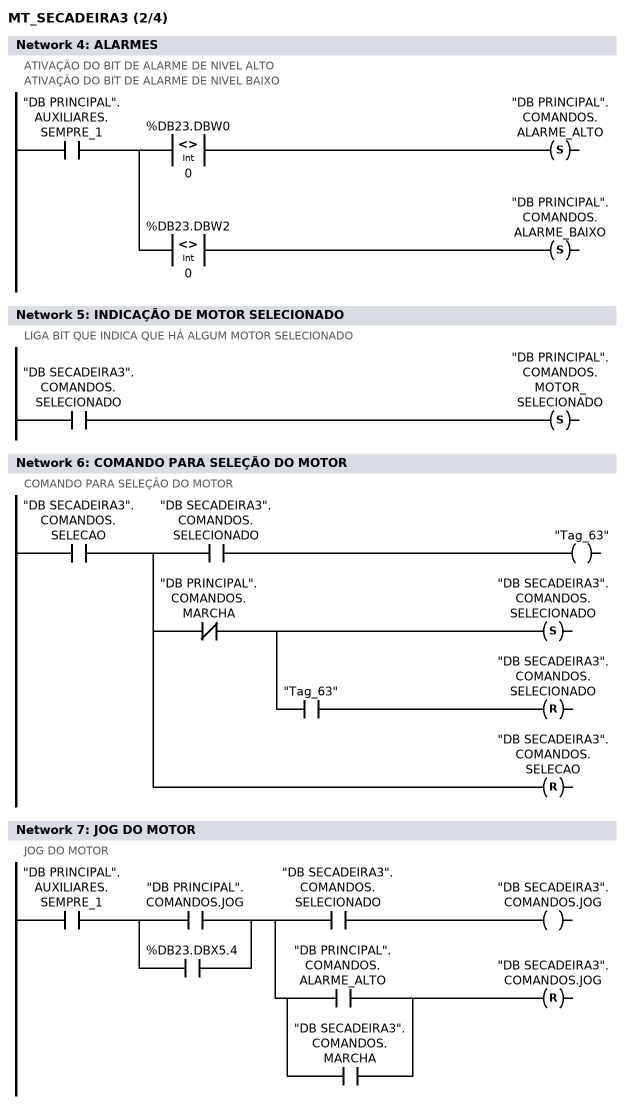
   RUNG wire#powerrail
      Contact( "DB PRINCIPAL".AUXILIARES.SEMPRE_1 )
      wire#w1
      { S7_Templates := "SrcType := Int" } NE_Contact(in1 := %DB23.DBW0, in2 := 0)
      S_Coil( "DB PRINCIPAL".COMANDOS.ALARME_ALTO )
   END_RUNG
   RUNG wire#w1
      { S7_Templates := "SrcType := Int" } NE_Contact(in1 := %DB23.DBW2, in2 := 0)
      S_Coil( "DB PRINCIPAL".COMANDOS.ALARME_BAIXO )
   END_RUNG
   // the same network as SCL:
   IF "DB PRINCIPAL".AUXILIARES.SEMPRE_1 AND (%DB23.DBW0 <> 0) THEN
       "DB PRINCIPAL".COMANDOS.ALARME_ALTO := TRUE;
   END_IF;
   IF "DB PRINCIPAL".AUXILIARES.SEMPRE_1 AND (%DB23.DBW2 <> 0) THEN
       "DB PRINCIPAL".COMANDOS.ALARME_BAIXO := TRUE;
   END_IF;
END_REGION

REGION Network 5: INDICAÇÃO DE MOTOR SELECIONADO
   // LIGA BIT QUE INDICA QUE HÁ ALGUM MOTOR SELECIONADO
   RUNG wire#powerrail
      Contact( "DB SECADEIRA3".COMANDOS.SELECIONADO )
      S_Coil( "DB PRINCIPAL".COMANDOS.MOTOR_SELECIONADO )
   END_RUNG
   // the same network as SCL:
   IF "DB SECADEIRA3".COMANDOS.SELECIONADO THEN "DB PRINCIPAL".COMANDOS.MOTOR_SELECIONADO := TRUE; END_IF;
END_REGION

REGION Network 6: COMANDO PARA SELEÇÃO DO MOTOR
   // COMANDO PARA SELEÇÃO DO MOTOR
   RUNG wire#powerrail
      Contact( "DB SECADEIRA3".COMANDOS.SELECAO )
      wire#w1
      Contact( "DB SECADEIRA3".COMANDOS.SELECIONADO )
      Coil( "Tag_63" )
   END_RUNG
   RUNG wire#w1
      I_Contact( "DB PRINCIPAL".COMANDOS.MARCHA )
      wire#w2
      S_Coil( "DB SECADEIRA3".COMANDOS.SELECIONADO )
   END_RUNG
   RUNG wire#w2
      Contact( "Tag_63" )
      R_Coil( "DB SECADEIRA3".COMANDOS.SELECIONADO )
   END_RUNG
   RUNG wire#w1
      R_Coil( "DB SECADEIRA3".COMANDOS.SELECAO )
   END_RUNG
   // the same network as SCL:
   "Tag_63" := "DB SECADEIRA3".COMANDOS.SELECAO AND "DB SECADEIRA3".COMANDOS.SELECIONADO;
   #_w1 := "DB SECADEIRA3".COMANDOS.SELECAO AND NOT "DB PRINCIPAL".COMANDOS.MARCHA;
   IF #_w1 THEN "DB SECADEIRA3".COMANDOS.SELECIONADO := TRUE; END_IF;
   IF #_w1 AND "Tag_63" THEN "DB SECADEIRA3".COMANDOS.SELECIONADO := FALSE; END_IF;
   IF "DB SECADEIRA3".COMANDOS.SELECAO THEN "DB SECADEIRA3".COMANDOS.SELECAO := FALSE; END_IF;
END_REGION

REGION Network 7: JOG DO MOTOR
   // JOG DO MOTOR
   RUNG wire#powerrail
      Contact( "DB PRINCIPAL".AUXILIARES.SEMPRE_1 )
      wire#w1
      Contact( "DB PRINCIPAL".COMANDOS.JOG )
      wire#w2
      Contact( "DB SECADEIRA3".COMANDOS.SELECIONADO )
      Coil( "DB SECADEIRA3".COMANDOS.JOG )
   END_RUNG
   RUNG wire#w1
      Contact( %DB23.DBX5.4 )
   END_RUNG wire#w2
   RUNG wire#w2
      Contact( "DB PRINCIPAL".COMANDOS.ALARME_ALTO )
      wire#w3
      R_Coil( "DB SECADEIRA3".COMANDOS.JOG )
   END_RUNG
   RUNG wire#w2
      Contact( "DB SECADEIRA3".COMANDOS.MARCHA )
   END_RUNG wire#w3
   // the same network as SCL:
   #_w1 := "DB PRINCIPAL".AUXILIARES.SEMPRE_1 AND ("DB PRINCIPAL".COMANDOS.JOG OR %DB23.DBX5.4);
   "DB SECADEIRA3".COMANDOS.JOG := #_w1 AND "DB SECADEIRA3".COMANDOS.SELECIONADO;
   IF #_w1 AND ("DB PRINCIPAL".COMANDOS.ALARME_ALTO OR "DB SECADEIRA3".COMANDOS.MARCHA) THEN
       "DB SECADEIRA3".COMANDOS.JOG := FALSE;
   END_IF;
END_REGION

REGION Network 8: COMANDO PARA LIBERAÇÃO DO MOTOR
   // COMANDO PARA LIBERAÇÃO DO MOTOR
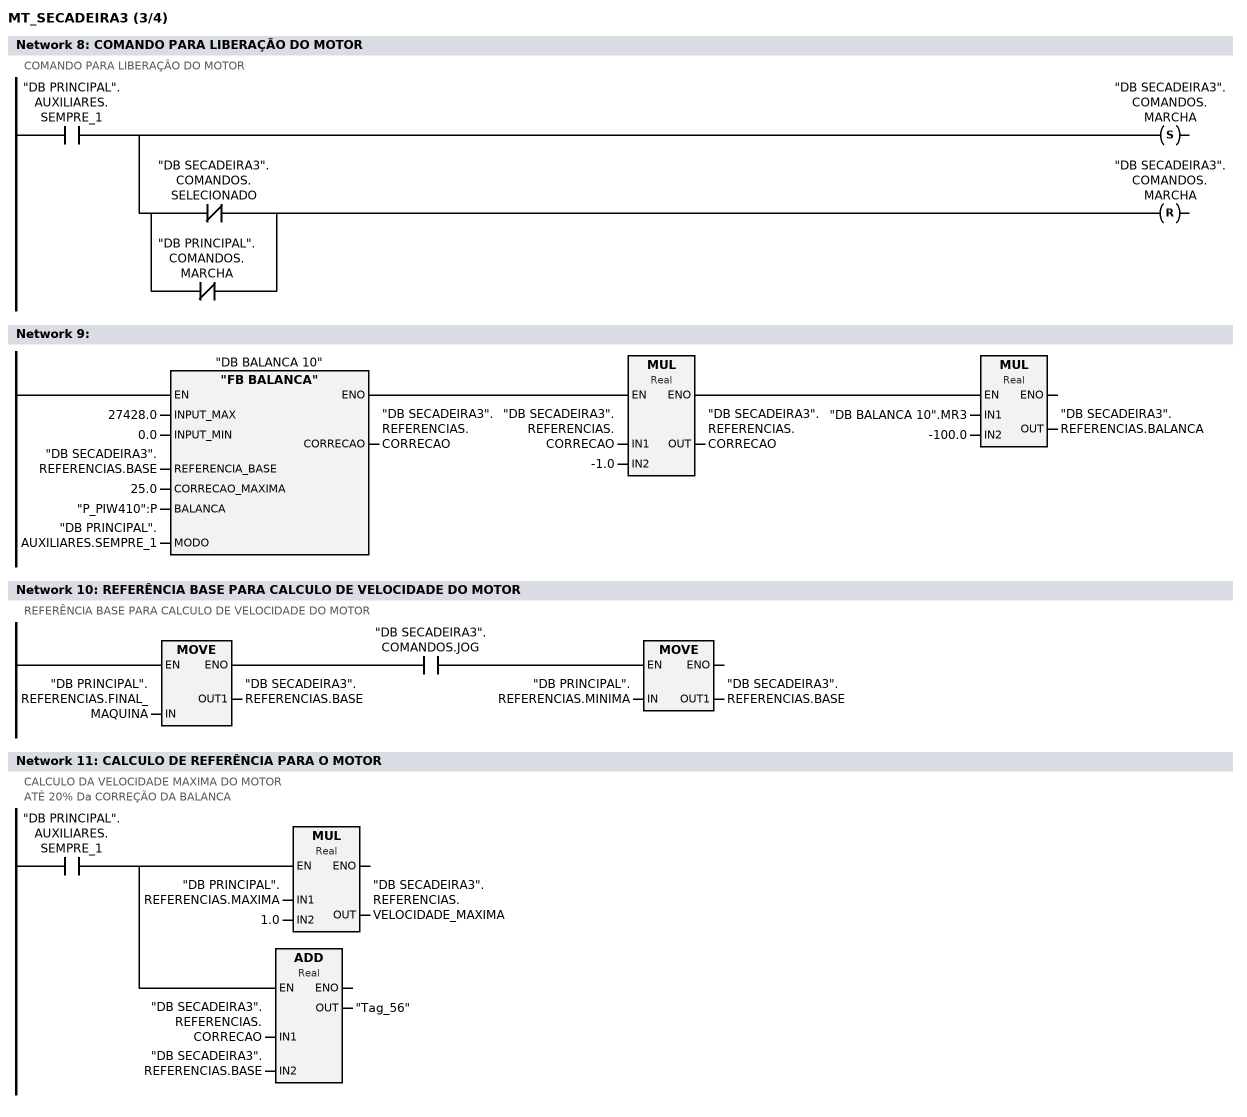
   RUNG wire#powerrail
      Contact( "DB PRINCIPAL".AUXILIARES.SEMPRE_1 )
      wire#w1
      S_Coil( "DB SECADEIRA3".COMANDOS.MARCHA )
   END_RUNG
   RUNG wire#w1
      I_Contact( "DB SECADEIRA3".COMANDOS.SELECIONADO )
      wire#w2
      R_Coil( "DB SECADEIRA3".COMANDOS.MARCHA )
   END_RUNG
   RUNG wire#w1
      I_Contact( "DB PRINCIPAL".COMANDOS.MARCHA )
   END_RUNG wire#w2
   // the same network as SCL:
   IF "DB PRINCIPAL".AUXILIARES.SEMPRE_1 THEN "DB SECADEIRA3".COMANDOS.MARCHA := TRUE; END_IF;
   IF "DB PRINCIPAL".AUXILIARES.SEMPRE_1 AND (NOT "DB SECADEIRA3".COMANDOS.SELECIONADO OR NOT "DB PRINCIPAL".COMANDOS.MARCHA) THEN
       "DB SECADEIRA3".COMANDOS.MARCHA := FALSE;
   END_IF;
END_REGION

REGION Network 9
   RUNG wire#powerrail
      "DB BALANCA 10"(INPUT_MAX := 27428.0, INPUT_MIN := 0.0, REFERENCIA_BASE := "DB SECADEIRA3".REFERENCIAS.BASE, CORRECAO_MAXIMA := 25.0, BALANCA := "P_PIW410":P, MODO := "DB PRINCIPAL".AUXILIARES.SEMPRE_1, CORRECAO => "DB SECADEIRA3".REFERENCIAS.CORRECAO)
      { S7_Templates := "SrcType := Real"; S7_GenerateENO := "TRUE" } Mul(in1 := "DB SECADEIRA3".REFERENCIAS.CORRECAO, in2 := -1.0, out => "DB SECADEIRA3".REFERENCIAS.CORRECAO)
      { S7_Templates := "SrcType := Real"; S7_GenerateENO := "TRUE" } Mul(in1 := "DB BALANCA 10".MR3, in2 := -100.0, out => "DB SECADEIRA3".REFERENCIAS.BALANCA)
   END_RUNG
   // the same network as SCL:
   // ENO of a box is taken as its EN; it also drops when the box reports an error
   "DB BALANCA 10"(INPUT_MAX := 27428.0,   // "FB BALANCA"
                   INPUT_MIN := 0.0,
                   REFERENCIA_BASE := "DB SECADEIRA3".REFERENCIAS.BASE,
                   CORRECAO_MAXIMA := 25.0,
                   BALANCA := "P_PIW410":P,
                   MODO := "DB PRINCIPAL".AUXILIARES.SEMPRE_1,
                   CORRECAO => "DB SECADEIRA3".REFERENCIAS.CORRECAO,
                   ENO => #_w1);
   IF #_w1 THEN
       "DB SECADEIRA3".REFERENCIAS.CORRECAO := "DB SECADEIRA3".REFERENCIAS.CORRECAO * (-1.0);
       "DB SECADEIRA3".REFERENCIAS.BALANCA := "DB BALANCA 10".MR3 * (-100.0);
   END_IF;
END_REGION

REGION Network 10: REFERÊNCIA BASE PARA CALCULO DE VELOCIDADE DO MOTOR
   // REFERÊNCIA BASE PARA CALCULO DE VELOCIDADE DO MOTOR
   RUNG wire#powerrail
      { S7_GenerateENO := "TRUE" } Move(in := "DB PRINCIPAL".REFERENCIAS.FINAL_MAQUINA, out1 => "DB SECADEIRA3".REFERENCIAS.BASE)
      Contact( "DB SECADEIRA3".COMANDOS.JOG )
      { S7_GenerateENO := "TRUE" } Move(in := "DB PRINCIPAL".REFERENCIAS.MINIMA, out1 => "DB SECADEIRA3".REFERENCIAS.BASE)
   END_RUNG
   // the same network as SCL:
   // ENO of a box is taken as its EN; it also drops when the box reports an error
   "DB SECADEIRA3".REFERENCIAS.BASE := "DB PRINCIPAL".REFERENCIAS.FINAL_MAQUINA;
   IF "DB SECADEIRA3".COMANDOS.JOG THEN
       "DB SECADEIRA3".REFERENCIAS.BASE := "DB PRINCIPAL".REFERENCIAS.MINIMA;
   END_IF;
END_REGION

REGION Network 11: CALCULO DE REFERÊNCIA PARA O MOTOR
   // CALCULO DA VELOCIDADE MAXIMA DO MOTOR
   // ATÉ 20% Da CORREÇÃO DA BALANCA
   RUNG wire#powerrail
      Contact( "DB PRINCIPAL".AUXILIARES.SEMPRE_1 )
      wire#w1
      { S7_Templates := "SrcType := Real"; S7_GenerateENO := "TRUE" } Mul(in1 := "DB PRINCIPAL".REFERENCIAS.MAXIMA, in2 := 1.0, out => "DB SECADEIRA3".REFERENCIAS.VELOCIDADE_MAXIMA)
   END_RUNG
   RUNG wire#w1
      { S7_Templates := "SrcType := Real"; S7_GenerateENO := "TRUE" } Add(in1 := "DB SECADEIRA3".REFERENCIAS.CORRECAO, in2 := "DB SECADEIRA3".REFERENCIAS.BASE, out => "Tag_56")
   END_RUNG
   // the same network as SCL:
   IF "DB PRINCIPAL".AUXILIARES.SEMPRE_1 THEN
       "DB SECADEIRA3".REFERENCIAS.VELOCIDADE_MAXIMA := "DB PRINCIPAL".REFERENCIAS.MAXIMA * 1.0;
       "Tag_56" := "DB SECADEIRA3".REFERENCIAS.CORRECAO + "DB SECADEIRA3".REFERENCIAS.BASE;
   END_IF;
END_REGION

REGION Network 12: ACC/DEC DA REFERÊNCIA DO MOTOR
   // ACC/DEC DA REFERÊNCIA DO MOTOR
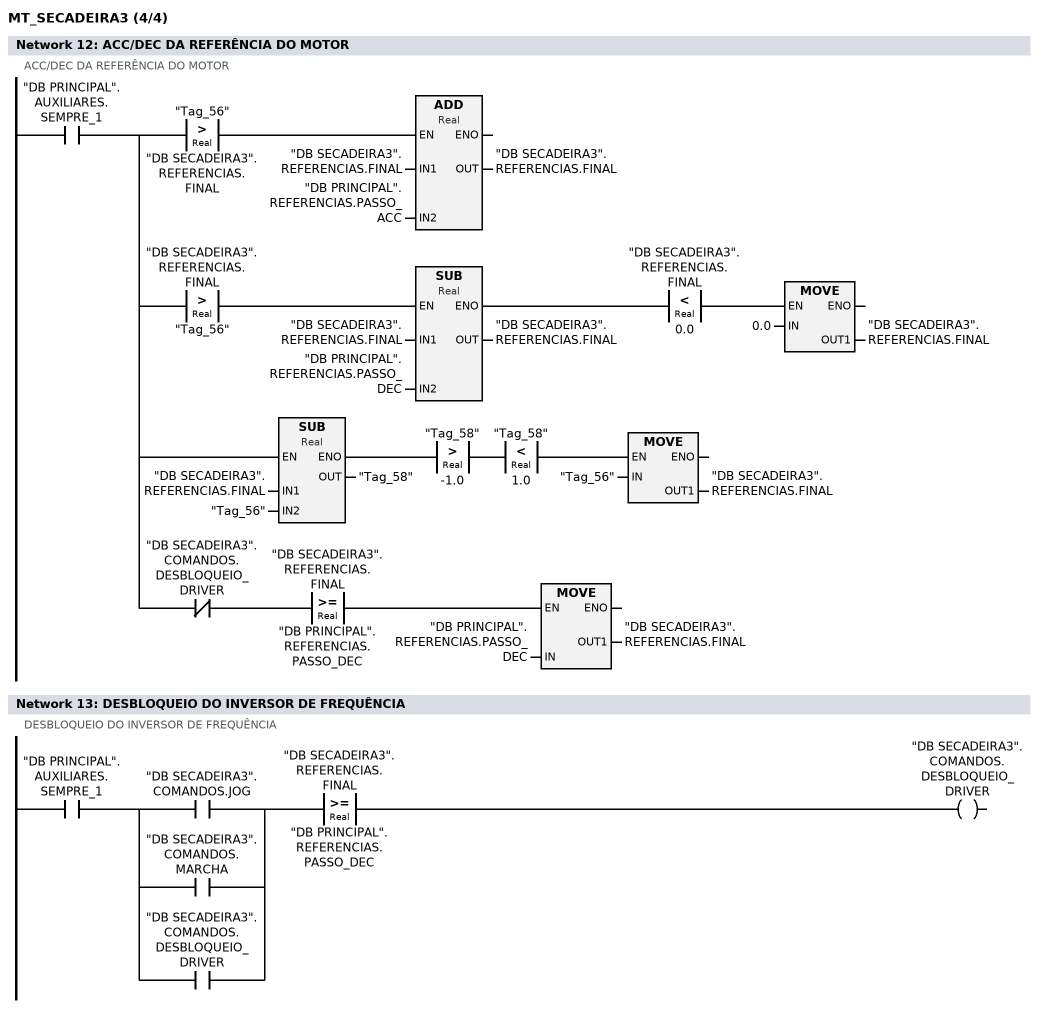
   RUNG wire#powerrail
      Contact( "DB PRINCIPAL".AUXILIARES.SEMPRE_1 )
      wire#w1
      { S7_Templates := "SrcType := Real" } GT_Contact(in1 := "Tag_56", in2 := "DB SECADEIRA3".REFERENCIAS.FINAL)
      { S7_Templates := "SrcType := Real"; S7_GenerateENO := "TRUE" } Add(in1 := "DB SECADEIRA3".REFERENCIAS.FINAL, in2 := "DB PRINCIPAL".REFERENCIAS.PASSO_ACC, out => "DB SECADEIRA3".REFERENCIAS.FINAL)
   END_RUNG
   RUNG wire#w1
      { S7_Templates := "SrcType := Real" } GT_Contact(in1 := "DB SECADEIRA3".REFERENCIAS.FINAL, in2 := "Tag_56")
      { S7_Templates := "SrcType := Real"; S7_GenerateENO := "TRUE" } Sub(in1 := "DB SECADEIRA3".REFERENCIAS.FINAL, in2 := "DB PRINCIPAL".REFERENCIAS.PASSO_DEC, out => "DB SECADEIRA3".REFERENCIAS.FINAL)
      { S7_Templates := "SrcType := Real" } LT_Contact(in1 := "DB SECADEIRA3".REFERENCIAS.FINAL, in2 := 0.0)
      { S7_GenerateENO := "TRUE" } Move(in := 0.0, out1 => "DB SECADEIRA3".REFERENCIAS.FINAL)
   END_RUNG
   RUNG wire#w1
      { S7_Templates := "SrcType := Real"; S7_GenerateENO := "TRUE" } Sub(in1 := "DB SECADEIRA3".REFERENCIAS.FINAL, in2 := "Tag_56", out => "Tag_58")
      { S7_Templates := "SrcType := Real" } GT_Contact(in1 := "Tag_58", in2 := -1.0)
      { S7_Templates := "SrcType := Real" } LT_Contact(in1 := "Tag_58", in2 := 1.0)
      { S7_GenerateENO := "TRUE" } Move(in := "Tag_56", out1 => "DB SECADEIRA3".REFERENCIAS.FINAL)
   END_RUNG
   RUNG wire#w1
      I_Contact( "DB SECADEIRA3".COMANDOS.DESBLOQUEIO_DRIVER )
      { S7_Templates := "SrcType := Real" } GE_Contact(in1 := "DB SECADEIRA3".REFERENCIAS.FINAL, in2 := "DB PRINCIPAL".REFERENCIAS.PASSO_DEC)
      { S7_GenerateENO := "TRUE" } Move(in := "DB PRINCIPAL".REFERENCIAS.PASSO_DEC, out1 => "DB SECADEIRA3".REFERENCIAS.FINAL)
   END_RUNG
   // the same network as SCL:
   // ENO of a box is taken as its EN; it also drops when the box reports an error
   IF "DB PRINCIPAL".AUXILIARES.SEMPRE_1 AND ("Tag_56" > "DB SECADEIRA3".REFERENCIAS.FINAL) THEN
       "DB SECADEIRA3".REFERENCIAS.FINAL := "DB SECADEIRA3".REFERENCIAS.FINAL + "DB PRINCIPAL".REFERENCIAS.PASSO_ACC;
   END_IF;
   #_w1 := "DB PRINCIPAL".AUXILIARES.SEMPRE_1 AND ("DB SECADEIRA3".REFERENCIAS.FINAL > "Tag_56");
   IF #_w1 THEN
       "DB SECADEIRA3".REFERENCIAS.FINAL := "DB SECADEIRA3".REFERENCIAS.FINAL - "DB PRINCIPAL".REFERENCIAS.PASSO_DEC;
   END_IF;
   IF #_w1 AND ("DB SECADEIRA3".REFERENCIAS.FINAL < 0.0) THEN
       "DB SECADEIRA3".REFERENCIAS.FINAL := 0.0;
   END_IF;
   IF "DB PRINCIPAL".AUXILIARES.SEMPRE_1 THEN
       "Tag_58" := "DB SECADEIRA3".REFERENCIAS.FINAL - "Tag_56";
   END_IF;
   IF "DB PRINCIPAL".AUXILIARES.SEMPRE_1 AND ("Tag_58" > (-1.0)) AND ("Tag_58" < 1.0) THEN
       "DB SECADEIRA3".REFERENCIAS.FINAL := "Tag_56";
   END_IF;
   IF "DB PRINCIPAL".AUXILIARES.SEMPRE_1 AND NOT "DB SECADEIRA3".COMANDOS.DESBLOQUEIO_DRIVER AND ("DB SECADEIRA3".REFERENCIAS.FINAL >= "DB PRINCIPAL".REFERENCIAS.PASSO_DEC) THEN
       "DB SECADEIRA3".REFERENCIAS.FINAL := "DB PRINCIPAL".REFERENCIAS.PASSO_DEC;
   END_IF;
END_REGION

REGION Network 13: DESBLOQUEIO DO INVERSOR DE FREQUÊNCIA
   // DESBLOQUEIO DO INVERSOR DE FREQUÊNCIA
   RUNG wire#powerrail
      Contact( "DB PRINCIPAL".AUXILIARES.SEMPRE_1 )
      wire#w1
      Contact( "DB SECADEIRA3".COMANDOS.JOG )
      wire#w2
      { S7_Templates := "SrcType := Real" } GE_Contact(in1 := "DB SECADEIRA3".REFERENCIAS.FINAL, in2 := "DB PRINCIPAL".REFERENCIAS.PASSO_DEC)
      Coil( "DB SECADEIRA3".COMANDOS.DESBLOQUEIO_DRIVER )
   END_RUNG
   RUNG wire#w1
      Contact( "DB SECADEIRA3".COMANDOS.MARCHA )
   END_RUNG wire#w2
   RUNG wire#w1
      Contact( "DB SECADEIRA3".COMANDOS.DESBLOQUEIO_DRIVER )
   END_RUNG wire#w2
   // the same network as SCL:
   "DB SECADEIRA3".COMANDOS.DESBLOQUEIO_DRIVER := "DB PRINCIPAL".AUXILIARES.SEMPRE_1 AND ("DB SECADEIRA3".COMANDOS.JOG OR "DB SECADEIRA3".COMANDOS.MARCHA OR "DB SECADEIRA3".COMANDOS.DESBLOQUEIO_DRIVER) AND ("DB SECADEIRA3".REFERENCIAS.FINAL >= "DB PRINCIPAL".REFERENCIAS.PASSO_DEC);
END_REGION

REGION Network 14 (STL): STATUS / CONTROLE - INVERSOR DE FREQUÊNCIA
   // DANFOSS FC300 PROFIBUS - TEX24626INV001
   // STATUS DO INVERSOR DE FREQUÊNCIA
         L     "Tag_39":P;
         T     "Tag_1";
         AN    "Tag_59";
         =     "DB SECADEIRA3".COMANDOS.STATUS_DRIVER;

   // CONTROLE DO INVERSOR DE FREQUÊNCIA
         L     1150;
         T     "Tag_1";
         A     "DB SECADEIRA3".COMANDOS.DESBLOQUEIO_DRIVER;
         =     "Tag_60";
         A     "T2";
         AN    "DB SECADEIRA3".COMANDOS.STATUS_DRIVER;
         =     "Tag_61";
         L     "Tag_1";
         T     "Tag_40":P;

   // REFERÊNCIA PARA O INVERSOR DE FREQUÊNCIA
         L     "DB SECADEIRA3".REFERENCIAS.FINAL;
         L     16384.0;
         *R;

         L     "DB SECADEIRA3".REFERENCIAS.VELOCIDADE_MAXIMA;
         /R;
         RND;
         T     "Tag_62";
         L     "Tag_62";
         T     "Tag_41":P;
END_REGION

REGION Network 15 (STL): INVERSOR RESERVA
         A     "DB PRINCIPAL".AUXILIARES.SEMPRE_1;
         =     %L24.0;
         A     %L24.0;
         A(;
         L     "DB PRINCIPAL".AUXILIARES1.INVERSOR_RESERVA1;
         L     14;
         ==I;
         );
         =     %L24.1;
         A     %L24.1;
         JNB   M00d;
         L     "DB SECADEIRA3".REFERENCIAS.FINAL;
         L     3.456;
         *R;
         T     #AUX_R;
         RND;
         T     "P_QW100":P;
   M00d: NOP   0;
         A     %L24.1;
         A     "I130";
         S     "DB PRINCIPAL".ALARME.INV_RESERVA1;
         A     %L24.1;
         A     "DB SECADEIRA3".COMANDOS.DESBLOQUEIO_DRIVER;
         S     "Q134";
         A     %L24.1;
         AN    "DB SECADEIRA3".COMANDOS.DESBLOQUEIO_DRIVER;
         R     "Q134";
         A     %L24.0;
         A(;
         L     "DB PRINCIPAL".AUXILIARES1.INVERSOR_RESERVA2;
         L     14;
         ==I;
         );
         =     %L24.1;
         A     %L24.1;
         JNB   M00e;
         L     "DB SECADEIRA3".REFERENCIAS.FINAL;
         L     3.456;
         *R;
         T     #AUX_R;
         RND;
         T     "P_QW102":P;
   M00e: NOP   0;
         A     %L24.1;
         A     "I132";
         S     "DB PRINCIPAL".ALARME.INV_RESERVA2;
         A     %L24.1;
         A     "DB SECADEIRA3".COMANDOS.DESBLOQUEIO_DRIVER;
         S     "Q135";
         A     %L24.1;
         AN    "DB SECADEIRA3".COMANDOS.DESBLOQUEIO_DRIVER;
         R     "Q135";
END_REGION
END_FUNCTION

FUNCTION "MT_SECADEIRA4" : Void   // FC24, LAD
TITLE = MÓDULO DE CONTROLE DA SECADEIRA 4
{ S7_Optimized_Access := 'FALSE' }
AUTHOR : THALLES
FAMILY : TRAÇÃO
NAME : LINHA1
VERSION : 0.1
// DATA BLOCK DE CONTROLE // DB24
// Automation Pack Automação Indl. e Com. Ltda.
// Cliente: Texima S/A Ind. de Máquinas
// Cliente Final: Cia. Fiação e Tecidos Santo Antonio.
// Máquina: LINHA 1 DENIN - O.S.: 24.626
   VAR_TEMP
      AUX_R : Real;
   END_VAR
   VAR_TEMP   // added for the SCL form of the ladder/FBD networks
      _w1 : Bool;
   END_VAR
BEGIN

REGION Network 1: ALARMES
   // RESET DOS ALARMES
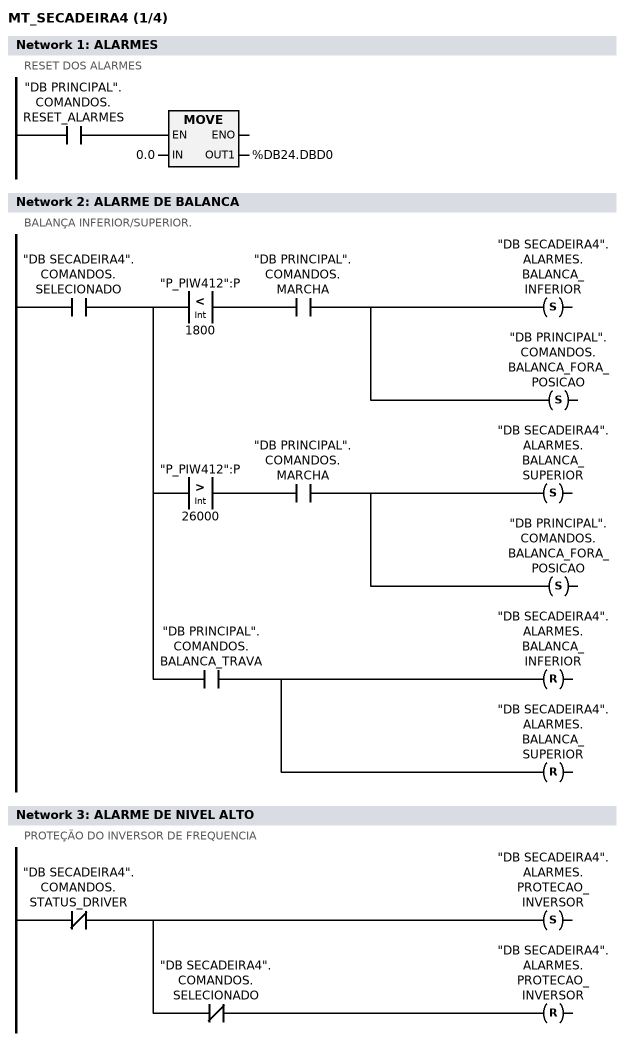
   RUNG wire#powerrail
      Contact( "DB PRINCIPAL".COMANDOS.RESET_ALARMES )
      { S7_GenerateENO := "TRUE" } Move(in := 0.0, out1 => %DB24.DBD0)
   END_RUNG
   // the same network as SCL:
   IF "DB PRINCIPAL".COMANDOS.RESET_ALARMES THEN %DB24.DBD0 := 0.0; END_IF;
END_REGION

REGION Network 2: ALARME DE BALANCA
   // BALANÇA INFERIOR/SUPERIOR.
   RUNG wire#powerrail
      Contact( "DB SECADEIRA4".COMANDOS.SELECIONADO )
      wire#w1
      { S7_Templates := "SrcType := Int" } LT_Contact(in1 := "P_PIW412":P, in2 := 1800)
      Contact( "DB PRINCIPAL".COMANDOS.MARCHA )
      wire#w2
      S_Coil( "DB SECADEIRA4".ALARMES.BALANCA_INFERIOR )
   END_RUNG
   RUNG wire#w2
      S_Coil( "DB PRINCIPAL".COMANDOS.BALANCA_FORA_POSICAO )
   END_RUNG
   RUNG wire#w1
      { S7_Templates := "SrcType := Int" } GT_Contact(in1 := "P_PIW412":P, in2 := 26000)
      Contact( "DB PRINCIPAL".COMANDOS.MARCHA )
      wire#w3
      S_Coil( "DB SECADEIRA4".ALARMES.BALANCA_SUPERIOR )
   END_RUNG
   RUNG wire#w3
      S_Coil( "DB PRINCIPAL".COMANDOS.BALANCA_FORA_POSICAO )
   END_RUNG
   RUNG wire#w1
      Contact( "DB PRINCIPAL".COMANDOS.BALANCA_TRAVA )
      wire#w4
      R_Coil( "DB SECADEIRA4".ALARMES.BALANCA_INFERIOR )
   END_RUNG
   RUNG wire#w4
      R_Coil( "DB SECADEIRA4".ALARMES.BALANCA_SUPERIOR )
   END_RUNG
   // the same network as SCL:
   IF "DB SECADEIRA4".COMANDOS.SELECIONADO AND ("P_PIW412":P < 1800) AND "DB PRINCIPAL".COMANDOS.MARCHA THEN
       "DB SECADEIRA4".ALARMES.BALANCA_INFERIOR := TRUE;
       "DB PRINCIPAL".COMANDOS.BALANCA_FORA_POSICAO := TRUE;
   END_IF;
   IF "DB SECADEIRA4".COMANDOS.SELECIONADO AND ("P_PIW412":P > 26000) AND "DB PRINCIPAL".COMANDOS.MARCHA THEN
       "DB SECADEIRA4".ALARMES.BALANCA_SUPERIOR := TRUE;
       "DB PRINCIPAL".COMANDOS.BALANCA_FORA_POSICAO := TRUE;
   END_IF;
   IF "DB SECADEIRA4".COMANDOS.SELECIONADO AND "DB PRINCIPAL".COMANDOS.BALANCA_TRAVA THEN
       "DB SECADEIRA4".ALARMES.BALANCA_INFERIOR := FALSE;
       "DB SECADEIRA4".ALARMES.BALANCA_SUPERIOR := FALSE;
   END_IF;
END_REGION

REGION Network 3: ALARME DE NIVEL ALTO
   // PROTEÇÃO DO INVERSOR DE FREQUENCIA
   RUNG wire#powerrail
      I_Contact( "DB SECADEIRA4".COMANDOS.STATUS_DRIVER )
      wire#w1
      S_Coil( "DB SECADEIRA4".ALARMES.PROTECAO_INVERSOR )
   END_RUNG
   RUNG wire#w1
      I_Contact( "DB SECADEIRA4".COMANDOS.SELECIONADO )
      R_Coil( "DB SECADEIRA4".ALARMES.PROTECAO_INVERSOR )
   END_RUNG
   // the same network as SCL:
   #_w1 := NOT "DB SECADEIRA4".COMANDOS.STATUS_DRIVER;
   IF #_w1 THEN "DB SECADEIRA4".ALARMES.PROTECAO_INVERSOR := TRUE; END_IF;
   IF #_w1 AND NOT "DB SECADEIRA4".COMANDOS.SELECIONADO THEN
       "DB SECADEIRA4".ALARMES.PROTECAO_INVERSOR := FALSE;
   END_IF;
END_REGION

REGION Network 4: ALARMES
   // ATIVAÇÃO DO BIT DE ALARME DE NIVEL ALTO
   // ATIVAÇÃO DO BIT DE ALARME DE NIVEL BAIXO
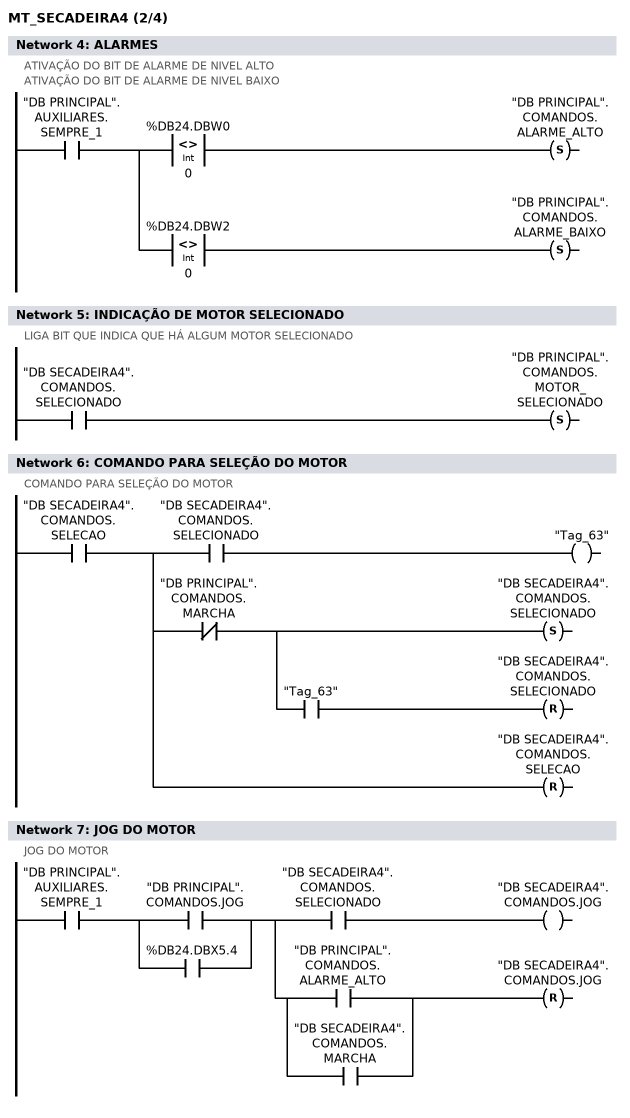
   RUNG wire#powerrail
      Contact( "DB PRINCIPAL".AUXILIARES.SEMPRE_1 )
      wire#w1
      { S7_Templates := "SrcType := Int" } NE_Contact(in1 := %DB24.DBW0, in2 := 0)
      S_Coil( "DB PRINCIPAL".COMANDOS.ALARME_ALTO )
   END_RUNG
   RUNG wire#w1
      { S7_Templates := "SrcType := Int" } NE_Contact(in1 := %DB24.DBW2, in2 := 0)
      S_Coil( "DB PRINCIPAL".COMANDOS.ALARME_BAIXO )
   END_RUNG
   // the same network as SCL:
   IF "DB PRINCIPAL".AUXILIARES.SEMPRE_1 AND (%DB24.DBW0 <> 0) THEN
       "DB PRINCIPAL".COMANDOS.ALARME_ALTO := TRUE;
   END_IF;
   IF "DB PRINCIPAL".AUXILIARES.SEMPRE_1 AND (%DB24.DBW2 <> 0) THEN
       "DB PRINCIPAL".COMANDOS.ALARME_BAIXO := TRUE;
   END_IF;
END_REGION

REGION Network 5: INDICAÇÃO DE MOTOR SELECIONADO
   // LIGA BIT QUE INDICA QUE HÁ ALGUM MOTOR SELECIONADO
   RUNG wire#powerrail
      Contact( "DB SECADEIRA4".COMANDOS.SELECIONADO )
      S_Coil( "DB PRINCIPAL".COMANDOS.MOTOR_SELECIONADO )
   END_RUNG
   // the same network as SCL:
   IF "DB SECADEIRA4".COMANDOS.SELECIONADO THEN "DB PRINCIPAL".COMANDOS.MOTOR_SELECIONADO := TRUE; END_IF;
END_REGION

REGION Network 6: COMANDO PARA SELEÇÃO DO MOTOR
   // COMANDO PARA SELEÇÃO DO MOTOR
   RUNG wire#powerrail
      Contact( "DB SECADEIRA4".COMANDOS.SELECAO )
      wire#w1
      Contact( "DB SECADEIRA4".COMANDOS.SELECIONADO )
      Coil( "Tag_63" )
   END_RUNG
   RUNG wire#w1
      I_Contact( "DB PRINCIPAL".COMANDOS.MARCHA )
      wire#w2
      S_Coil( "DB SECADEIRA4".COMANDOS.SELECIONADO )
   END_RUNG
   RUNG wire#w2
      Contact( "Tag_63" )
      R_Coil( "DB SECADEIRA4".COMANDOS.SELECIONADO )
   END_RUNG
   RUNG wire#w1
      R_Coil( "DB SECADEIRA4".COMANDOS.SELECAO )
   END_RUNG
   // the same network as SCL:
   "Tag_63" := "DB SECADEIRA4".COMANDOS.SELECAO AND "DB SECADEIRA4".COMANDOS.SELECIONADO;
   #_w1 := "DB SECADEIRA4".COMANDOS.SELECAO AND NOT "DB PRINCIPAL".COMANDOS.MARCHA;
   IF #_w1 THEN "DB SECADEIRA4".COMANDOS.SELECIONADO := TRUE; END_IF;
   IF #_w1 AND "Tag_63" THEN "DB SECADEIRA4".COMANDOS.SELECIONADO := FALSE; END_IF;
   IF "DB SECADEIRA4".COMANDOS.SELECAO THEN "DB SECADEIRA4".COMANDOS.SELECAO := FALSE; END_IF;
END_REGION

REGION Network 7: JOG DO MOTOR
   // JOG DO MOTOR
   RUNG wire#powerrail
      Contact( "DB PRINCIPAL".AUXILIARES.SEMPRE_1 )
      wire#w1
      Contact( "DB PRINCIPAL".COMANDOS.JOG )
      wire#w2
      Contact( "DB SECADEIRA4".COMANDOS.SELECIONADO )
      Coil( "DB SECADEIRA4".COMANDOS.JOG )
   END_RUNG
   RUNG wire#w1
      Contact( %DB24.DBX5.4 )
   END_RUNG wire#w2
   RUNG wire#w2
      Contact( "DB PRINCIPAL".COMANDOS.ALARME_ALTO )
      wire#w3
      R_Coil( "DB SECADEIRA4".COMANDOS.JOG )
   END_RUNG
   RUNG wire#w2
      Contact( "DB SECADEIRA4".COMANDOS.MARCHA )
   END_RUNG wire#w3
   // the same network as SCL:
   #_w1 := "DB PRINCIPAL".AUXILIARES.SEMPRE_1 AND ("DB PRINCIPAL".COMANDOS.JOG OR %DB24.DBX5.4);
   "DB SECADEIRA4".COMANDOS.JOG := #_w1 AND "DB SECADEIRA4".COMANDOS.SELECIONADO;
   IF #_w1 AND ("DB PRINCIPAL".COMANDOS.ALARME_ALTO OR "DB SECADEIRA4".COMANDOS.MARCHA) THEN
       "DB SECADEIRA4".COMANDOS.JOG := FALSE;
   END_IF;
END_REGION

REGION Network 8: COMANDO PARA LIBERAÇÃO DO MOTOR
   // COMANDO PARA LIBERAÇÃO DO MOTOR
